(* CODESYS project GraphicalTesting.project
   Company: ifm electronic
   Description: Project template with CR711S configured 2.25MByte Standard 2.25MByte Safety
   Version: 2.4.10.0
   Title: ifmCR711S_TemplateProject

Project tree, tasks and I/O mapping:
  SafetyPLC : CR711S SIL2, ifm electronic, order no. CR711S, version 3.2.0.0
    application Application
      libraries: ifmR360-3, * (ifm electronic)
      task Task (cyclic, interval t#10ms, priority 1, watchdog t#8ms x 1) calls PLC_PRG
      program PLC_PRG [ST]
      global variables EVL
    Communication : Communication, ifm electronic, version 3.2.0.0
      CAN : CAN, ifm electronic, version 3.2.0.0
      Ethernet : Ethernet, ifm electronic, version 3.2.0.0
    HMI : HMI, ifm electronic, version 3.2.0.0
      User_LEDs : User_LEDs, ifm electronic, version 3.2.0.0
          input  UserLED0_I : LED_IEC_B_INPUT_MAPPING_TYPE  // UserLED0_I
          input  UserLED1_I : LED_IEC_B_INPUT_MAPPING_TYPE  // UserLED1_I
          input  UserLED2_I : LED_IEC_B_INPUT_MAPPING_TYPE  // UserLED2_I
          input  UserLED3_I : LED_IEC_B_INPUT_MAPPING_TYPE  // UserLED3_I
          output UserLED0_Q : LED_IEC_B_OUTPUT_MAPPING_TYPE  // User LED 0
          output UserLED1_Q : LED_IEC_B_OUTPUT_MAPPING_TYPE  // User LED 1
          output UserLED2_Q : LED_IEC_B_OUTPUT_MAPPING_TYPE  // User LED 2
          output UserLED3_Q : LED_IEC_B_OUTPUT_MAPPING_TYPE  // User LED 3
    Local_IO : Local_IO, ifm electronic, version 3.2.0.0
      Inputs : Inputs, ifm electronic, version 3.2.0.0
          input  IN0100_I : IN_MULTIFUNCTION_A_INPUT_MAPPING_TYPE  // IN0100_I
          input  IN0101_I : IN_MULTIFUNCTION_A_INPUT_MAPPING_TYPE  // IN0101_I
          input  IN0102_I : IN_MULTIFUNCTION_A_INPUT_MAPPING_TYPE  // IN0102_I
          input  IN0103_I : IN_MULTIFUNCTION_A_INPUT_MAPPING_TYPE  // IN0103_I
          input  IN0200_I : IN_MULTIFUNCTION_A_INPUT_MAPPING_TYPE  // IN0200_I
          input  IN0201_I : IN_MULTIFUNCTION_A_INPUT_MAPPING_TYPE  // IN0201_I
          input  IN0202_I : IN_MULTIFUNCTION_A_INPUT_MAPPING_TYPE  // IN0202_I
          input  IN0203_I : IN_MULTIFUNCTION_A_INPUT_MAPPING_TYPE  // IN0203_I
          input  IN0600_I : IN_MULTIFUNCTION_A_INPUT_MAPPING_TYPE  // IN0600_I
          input  IN0601_I : IN_MULTIFUNCTION_A_INPUT_MAPPING_TYPE  // IN0601_I
          input  IN0602_I : IN_MULTIFUNCTION_A_INPUT_MAPPING_TYPE  // IN0602_I
          input  IN0603_I : IN_MULTIFUNCTION_A_INPUT_MAPPING_TYPE  // IN0603_I
          input  IN0700_I : IN_MULTIFUNCTION_A_INPUT_MAPPING_TYPE  // IN0700_I
          input  IN0701_I : IN_MULTIFUNCTION_A_INPUT_MAPPING_TYPE  // IN0701_I
          input  IN0702_I : IN_MULTIFUNCTION_A_INPUT_MAPPING_TYPE  // IN0702_I
          input  IN0703_I : IN_MULTIFUNCTION_A_INPUT_MAPPING_TYPE  // IN0703_I
          input  IN0400_I : IN_RESISTOR_A_INPUT_MAPPING_TYPE  // IN0400_I
          input  IN0401_I : IN_RESISTOR_A_INPUT_MAPPING_TYPE  // IN0401_I
          input  IN0900_I : IN_RESISTOR_A_INPUT_MAPPING_TYPE  // IN0900_I
          input  IN0901_I : IN_RESISTOR_A_INPUT_MAPPING_TYPE  // IN0901_I
          input  IN0300_I : IN_DIGITAL_B_INPUT_MAPPING_TYPE  // IN0300_I
          input  IN0301_I : IN_DIGITAL_B_INPUT_MAPPING_TYPE  // IN0301_I
          input  IN0800_I : IN_DIGITAL_B_INPUT_MAPPING_TYPE  // IN0800_I
          input  IN0801_I : IN_DIGITAL_B_INPUT_MAPPING_TYPE  // IN0801_I
          input  COM_RESET_I : IN_COMMUNICATION_RESET_INPUT_MAPPING_TYPE  // COM_RESET_I
          input  IN0000_I : IN_FREQUENCY_B_CHANNEL_A_INPUT_MAPPING_TYPE  // IN0000_I
          input  IN0002_I : IN_FREQUENCY_B_CHANNEL_A_INPUT_MAPPING_TYPE  // IN0002_I
          input  IN0500_I : IN_FREQUENCY_B_CHANNEL_A_INPUT_MAPPING_TYPE  // IN0500_I
          input  IN0502_I : IN_FREQUENCY_B_CHANNEL_A_INPUT_MAPPING_TYPE  // IN0502_I
          input  IN0001_I : IN_FREQUENCY_B_CHANNEL_B_INPUT_MAPPING_TYPE  // IN0001_I
          input  IN0003_I : IN_FREQUENCY_B_CHANNEL_B_INPUT_MAPPING_TYPE  // IN0003_I
          input  IN0501_I : IN_FREQUENCY_B_CHANNEL_B_INPUT_MAPPING_TYPE  // IN0501_I
          input  IN0503_I : IN_FREQUENCY_B_CHANNEL_B_INPUT_MAPPING_TYPE  // IN0503_I
      Outputs : Outputs, ifm electronic, version 3.2.0.0
          input  OUT0006_I : OUT_PWM_40_BRIDGE_A_INPUT_MAPPING_TYPE  // OUT0006_I
          input  OUT0106_I : OUT_PWM_40_BRIDGE_A_INPUT_MAPPING_TYPE  // OUT0106_I
          input  OUT0206_I : OUT_PWM_40_BRIDGE_A_INPUT_MAPPING_TYPE  // OUT0206_I
          input  OUT0008_I : OUT_PWM_40_A_INPUT_MAPPING_TYPE  // OUT0008_I
          input  OUT0108_I : OUT_PWM_40_A_INPUT_MAPPING_TYPE  // OUT0108_I
          input  OUT0208_I : OUT_PWM_40_A_INPUT_MAPPING_TYPE  // OUT0208_I
          input  OUT0000_I : OUT_PWM_25_A_INPUT_MAPPING_TYPE  // OUT0000_I
          input  OUT0002_I : OUT_PWM_25_A_INPUT_MAPPING_TYPE  // OUT0002_I
          input  OUT0004_I : OUT_PWM_25_A_INPUT_MAPPING_TYPE  // OUT0004_I
          input  OUT0100_I : OUT_PWM_25_A_INPUT_MAPPING_TYPE  // OUT0100_I
          input  OUT0102_I : OUT_PWM_25_A_INPUT_MAPPING_TYPE  // OUT0102_I
          input  OUT0104_I : OUT_PWM_25_A_INPUT_MAPPING_TYPE  // OUT0104_I
          input  OUT0200_I : OUT_PWM_25_A_INPUT_MAPPING_TYPE  // OUT0200_I
          input  OUT0202_I : OUT_PWM_25_A_INPUT_MAPPING_TYPE  // OUT0202_I
          input  OUT0204_I : OUT_PWM_25_A_INPUT_MAPPING_TYPE  // OUT0204_I
          input  OUT3001_I : OUT_VOLTAGE_A_INPUT_MAPPING_TYPE  // OUT3001_I
          input  OUT3000_I : OUT_SUPPLY_A_INPUT_MAPPING_TYPE  // OUT3000_I
          input  OUT0001_I : OUT_PWM_25_B_INPUT_MAPPING_TYPE  // OUT0001_I
          input  OUT0003_I : OUT_PWM_25_B_INPUT_MAPPING_TYPE  // OUT0003_I
          input  OUT0005_I : OUT_PWM_25_B_INPUT_MAPPING_TYPE  // OUT0005_I
          input  OUT0101_I : OUT_PWM_25_B_INPUT_MAPPING_TYPE  // OUT0101_I
          input  OUT0103_I : OUT_PWM_25_B_INPUT_MAPPING_TYPE  // OUT0103_I
          input  OUT0105_I : OUT_PWM_25_B_INPUT_MAPPING_TYPE  // OUT0105_I
          input  OUT0201_I : OUT_PWM_25_B_INPUT_MAPPING_TYPE  // OUT0201_I
          input  OUT0203_I : OUT_PWM_25_B_INPUT_MAPPING_TYPE  // OUT0203_I
          input  OUT0205_I : OUT_PWM_25_B_INPUT_MAPPING_TYPE  // OUT0205_I
          input  OUT0007_I : OUT_PWM_40_BRIDGE_A_INPUT_MAPPING_TYPE  // OUT0007_I
          input  OUT0107_I : OUT_PWM_40_BRIDGE_A_INPUT_MAPPING_TYPE  // OUT0107_I
          input  OUT0207_I : OUT_PWM_40_BRIDGE_A_INPUT_MAPPING_TYPE  // OUT0207_I
          output OUT0006_Q : OUT_PWM_40_BRIDGE_A_OUTPUT_MAPPING_TYPE  // OUT0006_Q
          output OUT0106_Q : OUT_PWM_40_BRIDGE_A_OUTPUT_MAPPING_TYPE  // OUT0106_Q
          output OUT0206_Q : OUT_PWM_40_BRIDGE_A_OUTPUT_MAPPING_TYPE  // OUT0206_Q
          output OUT0008_Q : OUT_PWM_40_A_OUTPUT_MAPPING_TYPE  // OUT0008_Q
          output OUT0108_Q : OUT_PWM_40_A_OUTPUT_MAPPING_TYPE  // OUT0108_Q
          output OUT0208_Q : OUT_PWM_40_A_OUTPUT_MAPPING_TYPE  // OUT0208_Q
          output OUT0000_Q : OUT_PWM_25_A_OUTPUT_MAPPING_TYPE  // OUT0000_Q
          output OUT0002_Q : OUT_PWM_25_A_OUTPUT_MAPPING_TYPE  // OUT0002_Q
          output OUT0004_Q : OUT_PWM_25_A_OUTPUT_MAPPING_TYPE  // OUT0004_Q
          output OUT0100_Q : OUT_PWM_25_A_OUTPUT_MAPPING_TYPE  // OUT0100_Q
          output OUT0102_Q : OUT_PWM_25_A_OUTPUT_MAPPING_TYPE  // OUT0102_Q
          output OUT0104_Q : OUT_PWM_25_A_OUTPUT_MAPPING_TYPE  // OUT0104_Q
          output OUT0200_Q : OUT_PWM_25_A_OUTPUT_MAPPING_TYPE  // OUT0200_Q
          output OUT0202_Q : OUT_PWM_25_A_OUTPUT_MAPPING_TYPE  // OUT0202_Q
          output OUT0204_Q : OUT_PWM_25_A_OUTPUT_MAPPING_TYPE  // OUT0204_Q
          output OUT3001_Q : OUT_VOLTAGE_A_OUTPUT_MAPPING_TYPE  // OUT3001_Q
          output OUT3000_Q : OUT_SUPPLY_A_OUTPUT_MAPPING_TYPE  // OUT3000_Q
          output OUT0001_Q : OUT_PWM_25_B_OUTPUT_MAPPING_TYPE  // OUT0001_Q
          output OUT0003_Q : OUT_PWM_25_B_OUTPUT_MAPPING_TYPE  // OUT0003_Q
          output OUT0005_Q : OUT_PWM_25_B_OUTPUT_MAPPING_TYPE  // OUT0005_Q
          output OUT0101_Q : OUT_PWM_25_B_OUTPUT_MAPPING_TYPE  // OUT0101_Q
          output OUT0103_Q : OUT_PWM_25_B_OUTPUT_MAPPING_TYPE  // OUT0103_Q
          output OUT0105_Q : OUT_PWM_25_B_OUTPUT_MAPPING_TYPE  // OUT0105_Q
          output OUT0201_Q : OUT_PWM_25_B_OUTPUT_MAPPING_TYPE  // OUT0201_Q
          output OUT0203_Q : OUT_PWM_25_B_OUTPUT_MAPPING_TYPE  // OUT0203_Q
          output OUT0205_Q : OUT_PWM_25_B_OUTPUT_MAPPING_TYPE  // OUT0205_Q
          output OUT0007_Q : OUT_PWM_40_BRIDGE_A_OUTPUT_MAPPING_TYPE  // OUT0007_Q
          output OUT0107_Q : OUT_PWM_40_BRIDGE_A_OUTPUT_MAPPING_TYPE  // OUT0107_Q
          output OUT0207_Q : OUT_PWM_40_BRIDGE_A_OUTPUT_MAPPING_TYPE  // OUT0207_Q
      System_Inputs : System_Inputs, ifm electronic, version 3.2.0.0
          input  VBB30 : IN_SYSTEM_VOLTAGE_INPUT_MAPPING_TYPE  // VBB30
          input  VBB15 : IN_SYSTEM_VOLTAGE_INPUT_MAPPING_TYPE  // VBB15
          input  TemperatureBoard0 : IN_TEMPERATURE_INPUT_MAPPING_TYPE  // TemperatureBoard0
          input  TemperatureChip0 : IN_TEMPERATURE_INPUT_MAPPING_TYPE  // TemperatureChip0
      System_Outputs : System_Outputs, ifm electronic, version 3.2.0.0
          input  VBB0_SW_I : OUT_GROUP_SWITCH_INPUT_MAPPING_TYPE  // VBB0_SW_I
          input  VBB1_SW_I : OUT_GROUP_SWITCH_INPUT_MAPPING_TYPE  // VBB1_SW_I
          input  VBB2_SW_I : OUT_GROUP_SWITCH_INPUT_MAPPING_TYPE  // VBB2_SW_I
          output VBB0_SW_Q : OUT_GROUP_SWITCH_OUTPUT_MAPPING_TYPE  // VBB0_SW_Q
          output VBB1_SW_Q : OUT_GROUP_SWITCH_OUTPUT_MAPPING_TYPE  // VBB1_SW_Q
          output VBB2_SW_Q : OUT_GROUP_SWITCH_OUTPUT_MAPPING_TYPE  // VBB2_SW_Q
          output SUPPLY_SWITCH_Q : OUT_SYS_SWITCH_OUTPUT_MAPPING_TYPE  // SUPPLY_SWITCH_Q
  StandardPLC : CR711S Standard, ifm electronic, order no. CR711S, version 3.2.0.0
    application Application
      libraries: ifmR360-3, 1.1.1.0 (ifm electronic); Util, * (System); Standard, * (System); CR711S IOWrapper, 1.0.4.9 (ifm electronic); CAA CiA 405, 3.5.8.0 (CAA Technical Workgroup)
      task Main (cyclic, interval t#20ms, priority 1, watchdog t#18ms x 1) calls PLC_PRG, _CAN_MAIN
      EVC
      global variables PersistentVars
      program SFC_TEST [SFC]
      program FB_TESTING [FBD]: PleaseIhaveKids
      program LD_TEST [LD]
      visualisation Visualization
    Communication : Communication, ifm electronic, version 3.2.0.0
      CAN : CAN, ifm electronic, version 3.2.0.0
        CANbus_1 : CANbus, ifm electronic, version 1.0.1.1
            settings: NetID = 1
          J1939_Manager : J1939_Manager, 3S - Smart Software Solutions GmbH, order no. 
      , version 3.5.16.0
            Engine_Receiver : J1939_ECU, 3S - Smart Software Solutions GmbH, version 3.5.9.0
                settings: NAME = 16#0000000000000000; Communication Watchog Enabled = TRUE; Communication Watchdog Timeout Period = 16#05DC ms; Activated PGs = 13; PG Offline Data.Name = "EEC2"; PG Offline Data.Description = "Electronic Engine Controller 2"; PG Online Data.PGN = 61443; PG Online Data.Length (Bytes) = 8; PG Transmission Settings.Destination Address = 255; PG Transmission Settings.CycleTimeFactor = 1; Signal Offline Data.SPN = 558; Signal Offline Data.Name = "Accelerator Pedal 1 Low Idle Switch"; Signal Offline Data.Unit = "bit"; Signal Offline Data.Min = 0; Signal Offline Data.Max = 3; Signal Online Data.BitSize = 2; Signal Online Data.BitPosition = 0; Convert Data.Flags = 3; Convert Data.pSigValue = 0; Convert Data.Scaling = 4607182418800017408; Convert Data.Offset = 0; Signal Offline Data.SPN = 559; Signal Offline Data.Name = "Accelerator Pedal Kickdown Switch"; Signal Offline Data.Unit = "bit"; Signal Offline Data.Min = 0; Signal Offline Data.Max = 3; Signal Online Data.BitSize = 2; Signal Online Data.BitPosition = 2; Convert Data.Flags = 3; Convert Data.pSigValue = 0; Convert Data.Scaling = 4607182418800017408; Convert Data.Offset = 0; Signal Offline Data.SPN = 1437; Signal Offline Data.Name = "Road Speed Limit Status"; Signal Offline Data.Unit = "bit"; Signal Offline Data.Min = 0; Signal Offline Data.Max = 3; Signal Online Data.BitSize = 2; Signal Online Data.BitPosition = 4; Convert Data.Flags = 3;
                  Convert Data.pSigValue = 0; Convert Data.Scaling = 4607182418800017408; Convert Data.Offset = 0; Signal Offline Data.SPN = 2970; Signal Offline Data.Name = "Accelerator Pedal 2 Low Idle Switch"; Signal Offline Data.Unit = "bit"; Signal Offline Data.Min = 0; Signal Offline Data.Max = 3; Signal Online Data.BitSize = 2; Signal Online Data.BitPosition = 6; Convert Data.Flags = 3; Convert Data.pSigValue = 0; Convert Data.Scaling = 4607182418800017408; Convert Data.Offset = 0; Signal Offline Data.SPN = 91; Signal Offline Data.Name = "Accelerator Pedal Position 1"; Signal Offline Data.Unit = "%"; Signal Offline Data.Min = 0; Signal Offline Data.Max = 100; Signal Online Data.BitSize = 8; Signal Online Data.BitPosition = 8; Convert Data.Flags = 3; Convert Data.pSigValue = 0; Convert Data.Scaling = 4600877379321698714; Convert Data.Offset = 0; Signal Offline Data.SPN = 92; Signal Offline Data.Name = "Engine Percent Load At Current Speed"; Signal Offline Data.Unit = "%"; Signal Offline Data.Min = 0; Signal Offline Data.Max = 250; Signal Online Data.BitSize = 8; Signal Online Data.BitPosition = 16; Convert Data.Flags = 3; Convert Data.pSigValue = 0; Convert Data.Scaling = 4607182418800017408; Convert Data.Offset = 0; Signal Offline Data.SPN = 974; Signal Offline Data.Name = "Remote Accelerator Pedal Position"; Signal Offline Data.Unit = "%"; Signal Offline Data.Min = 0;
                  Signal Offline Data.Max = 100; Signal Online Data.BitSize = 8; Signal Online Data.BitPosition = 24; Convert Data.Flags = 3; Convert Data.pSigValue = 0; Convert Data.Scaling = 4600877379321698714; Convert Data.Offset = 0; Signal Offline Data.SPN = 29; Signal Offline Data.Name = "Accelerator Pedal Position 2"; Signal Offline Data.Unit = "%"; Signal Offline Data.Min = 0; Signal Offline Data.Max = 100; Signal Online Data.BitSize = 8; Signal Online Data.BitPosition = 32; Convert Data.Flags = 3; Convert Data.pSigValue = 0; Convert Data.Scaling = 4600877379321698714; Convert Data.Offset = 0; Signal Offline Data.SPN = 2979; Signal Offline Data.Name = "Vehicle Acceleration Rate Limit Status"; Signal Offline Data.Unit = "bit"; Signal Offline Data.Min = 0; Signal Offline Data.Max = 3; Signal Online Data.BitSize = 2; Signal Online Data.BitPosition = 40; Convert Data.Flags = 3; Convert Data.pSigValue = 0; Convert Data.Scaling = 4607182418800017408; Convert Data.Offset = 0; Signal Offline Data.SPN = 5021; Signal Offline Data.Name = "Momentary Engine Maximum Power Enable Feedback"; Signal Offline Data.Unit = "bit"; Signal Offline Data.Min = 0; Signal Offline Data.Max = 3; Signal Online Data.BitSize = 2; Signal Online Data.BitPosition = 42; Convert Data.Flags = 3; Convert Data.pSigValue = 0; Convert Data.Scaling = 4607182418800017408; Convert Data.Offset = 0;
                  Signal Offline Data.SPN = 5399; Signal Offline Data.Name = "DPF Thermal Management Active"; Signal Offline Data.Unit = "bit"; Signal Offline Data.Min = 0; Signal Offline Data.Max = 3; Signal Online Data.BitSize = 2; Signal Online Data.BitPosition = 44; Convert Data.Flags = 3; Convert Data.pSigValue = 0; Convert Data.Scaling = 4607182418800017408; Convert Data.Offset = 0; Signal Offline Data.SPN = 5400; Signal Offline Data.Name = "SCR Thermal Management Active"; Signal Offline Data.Unit = "bit"; Signal Offline Data.Min = 0; Signal Offline Data.Max = 3; Signal Online Data.BitSize = 2; Signal Online Data.BitPosition = 46; Convert Data.Flags = 3; Convert Data.pSigValue = 0; Convert Data.Scaling = 4607182418800017408; Convert Data.Offset = 0; Signal Offline Data.SPN = 3357; Signal Offline Data.Name = "Actual Maximum Available Engine - Percent Torque"; Signal Offline Data.Unit = "%"; Signal Offline Data.Min = 0; Signal Offline Data.Max = 100; Signal Online Data.BitSize = 8; Signal Online Data.BitPosition = 48; Convert Data.Flags = 3; Convert Data.pSigValue = 0; Convert Data.Scaling = 4600877379321698714; Convert Data.Offset = 0; Signal Offline Data.SPN = 5398; Signal Offline Data.Name = "Estimated Pumping - Percent Torque"; Signal Offline Data.Unit = "%"; Signal Offline Data.Min = -125; Signal Offline Data.Max = 125; Signal Online Data.BitSize = 8; Signal Online Data.BitPosition = 56;
                  Convert Data.Flags = 3; Convert Data.pSigValue = 0; Convert Data.Scaling = 4607182418800017408; Convert Data.Offset = 13861868546813853696; PG Offline Data.Name = "EEC1"; PG Offline Data.Description = "Electronic Engine Controller 1"; PG Online Data.PGN = 61444; PG Online Data.Length (Bytes) = 8; PG Transmission Settings.Destination Address = 255; PG Transmission Settings.CycleTimeFactor = 1; Signal Offline Data.SPN = 899; Signal Offline Data.Name = "Engine Torque Mode"; Signal Offline Data.Unit = "bit"; Signal Offline Data.Min = 0; Signal Offline Data.Max = 15; Signal Online Data.BitSize = 4; Signal Online Data.BitPosition = 0; Convert Data.Flags = 3; Convert Data.pSigValue = 0; Convert Data.Scaling = 4607182418800017408; Convert Data.Offset = 0; Signal Offline Data.SPN = 4154; Signal Offline Data.Name = "Actual Engine - Percent Torque High Resolution"; Signal Offline Data.Unit = "%"; Signal Offline Data.Min = 0; Signal Offline Data.Max = 0.875; Signal Online Data.BitSize = 4; Signal Online Data.BitPosition = 4; Convert Data.Flags = 3; Convert Data.pSigValue = 0; Convert Data.Scaling = 4593671619917905920; Convert Data.Offset = 0; Signal Offline Data.SPN = 512; Signal Offline Data.Name = "Driver$'s Demand Engine - Percent Torque"; Signal Offline Data.Unit = "%"; Signal Offline Data.Min = -125; Signal Offline Data.Max = 125; Signal Online Data.BitSize = 8; Signal Online Data.BitPosition = 8; Convert Data.Flags = 3;
                  Convert Data.pSigValue = 0; Convert Data.Scaling = 4607182418800017408; Convert Data.Offset = 13861868546813853696; Signal Offline Data.SPN = 513; Signal Offline Data.Name = "Actual Engine - Percent Torque"; Signal Offline Data.Unit = "%"; Signal Offline Data.Min = -125; Signal Offline Data.Max = 125; Signal Online Data.BitSize = 8; Signal Online Data.BitPosition = 16; Convert Data.Flags = 3; Convert Data.pSigValue = 0; Convert Data.Scaling = 4607182418800017408; Convert Data.Offset = 13861868546813853696; Signal Offline Data.SPN = 190; Signal Offline Data.Name = "Engine Speed"; Signal Offline Data.Unit = "rpm"; Signal Offline Data.Min = 0; Signal Offline Data.Max = 8031.875; Signal Online Data.BitSize = 16; Signal Online Data.BitPosition = 24; Convert Data.Flags = 3; Convert Data.pSigValue = 0; Convert Data.Scaling = 4593671619917905920; Convert Data.Offset = 0; Signal Offline Data.SPN = 1483; Signal Offline Data.Name = "Source Address of Controlling Device for Engine Control"; Signal Offline Data.Unit = "SA"; Signal Offline Data.Min = 0; Signal Offline Data.Max = 255; Signal Online Data.BitSize = 8; Signal Online Data.BitPosition = 40; Convert Data.Flags = 3; Convert Data.pSigValue = 0; Convert Data.Scaling = 4607182418800017408; Convert Data.Offset = 0; Signal Offline Data.SPN = 1675; Signal Offline Data.Name = "Engine Starter Mode"; Signal Offline Data.Unit = "bit"; Signal Offline Data.Min = 0;
                  Signal Offline Data.Max = 15; Signal Online Data.BitSize = 4; Signal Online Data.BitPosition = 48; Convert Data.Flags = 3; Convert Data.pSigValue = 0; Convert Data.Scaling = 4607182418800017408; Convert Data.Offset = 0; Signal Offline Data.SPN = 2432; Signal Offline Data.Name = "Engine Demand – Percent Torque"; Signal Offline Data.Unit = "%"; Signal Offline Data.Min = -125; Signal Offline Data.Max = 125; Signal Online Data.BitSize = 8; Signal Online Data.BitPosition = 56; Convert Data.Flags = 3; Convert Data.pSigValue = 0; Convert Data.Scaling = 4607182418800017408; Convert Data.Offset = 13861868546813853696; PG Offline Data.Name = "HOURS"; PG Offline Data.Description = "Engine Hours, Revolutions"; PG Online Data.PGN = 65253; PG Online Data.Length (Bytes) = 8; PG Transmission Settings.Destination Address = 255; PG Transmission Settings.CycleTimeFactor = 1; Signal Offline Data.SPN = 247; Signal Offline Data.Name = "Engine Total Hours of Operation"; Signal Offline Data.Description = "Accumulated time of operation of engine."; Signal Offline Data.Unit = "hr"; Signal Offline Data.Min = 0; Signal Offline Data.Max = 210554060.75; Signal Online Data.BitSize = 32; Signal Online Data.BitPosition = 0; Convert Data.Flags = 3; Convert Data.pSigValue = 0; Convert Data.Scaling = 4587366580439587226; Convert Data.Offset = 0; Signal Offline Data.SPN = 249; Signal Offline Data.Name = "Engine Total Revolutions"; Signal Offline Data.Description = "Accumulated number of revolutions of engine crankshaft during its operation."; Signal Offline Data.Unit = "r";
                  Signal Offline Data.Min = 0; Signal Offline Data.Max = 4211081215000; Signal Online Data.BitSize = 32; Signal Online Data.BitPosition = 32; Convert Data.Flags = 3; Convert Data.pSigValue = 0; Convert Data.Scaling = 4652007308841189376; Convert Data.Offset = 0; PG Offline Data.Name = "ET1"; PG Offline Data.Description = "Engine Temperature 1"; PG Online Data.PGN = 65262; PG Online Data.Length (Bytes) = 8; PG Transmission Settings.Destination Address = 255; PG Transmission Settings.CycleTimeFactor = 1; Signal Offline Data.SPN = 110; Signal Offline Data.Name = "Engine Coolant Temperature"; Signal Offline Data.Description = "Temperature of liquid found in engine cooling system."; Signal Offline Data.Unit = "C"; Signal Offline Data.Min = -40; Signal Offline Data.Max = 210; Signal Online Data.BitSize = 8; Signal Online Data.BitPosition = 0; Convert Data.Flags = 3; Convert Data.pSigValue = 0; Convert Data.Scaling = 4607182418800017408; Convert Data.Offset = 13854198353698488320; Signal Offline Data.SPN = 174; Signal Offline Data.Name = "Engine Fuel Temperature 1"; Signal Offline Data.Unit = "C"; Signal Offline Data.Min = -40; Signal Offline Data.Max = 210; Signal Online Data.BitSize = 8; Signal Online Data.BitPosition = 8; Convert Data.Flags = 3; Convert Data.pSigValue = 0; Convert Data.Scaling = 4607182418800017408; Convert Data.Offset = 13854198353698488320; Signal Offline Data.SPN = 175; Signal Offline Data.Name = "Engine Oil Temperature 1"; Signal Offline Data.Description = "Temperature of the engine lubricant.";
                  Signal Offline Data.Unit = "C"; Signal Offline Data.Min = -273; Signal Offline Data.Max = 1734.96875; Signal Online Data.BitSize = 16; Signal Online Data.BitPosition = 16; Convert Data.Flags = 3; Convert Data.pSigValue = 0; Convert Data.Scaling = 4584664420663164928; Convert Data.Offset = 13866882319836512256; Signal Offline Data.SPN = 176; Signal Offline Data.Name = "Engine Turbocharger Oil Temperature"; Signal Offline Data.Description = "Temperature of the turbocharger lubricant."; Signal Offline Data.Unit = "C"; Signal Offline Data.Min = -273; Signal Offline Data.Max = 1734.96875; Signal Online Data.BitSize = 16; Signal Online Data.BitPosition = 32; Convert Data.Flags = 3; Convert Data.pSigValue = 0; Convert Data.Scaling = 4584664420663164928; Convert Data.Offset = 13866882319836512256; Signal Offline Data.SPN = 52; Signal Offline Data.Name = "Engine Intercooler Temperature"; Signal Offline Data.Description = "Temperature of liquid found in the intercooler located after the turbocharger."; Signal Offline Data.Unit = "C"; Signal Offline Data.Min = -40; Signal Offline Data.Max = 210; Signal Online Data.BitSize = 8; Signal Online Data.BitPosition = 48; Convert Data.Flags = 3; Convert Data.pSigValue = 0; Convert Data.Scaling = 4607182418800017408; Convert Data.Offset = 13854198353698488320; Signal Offline Data.SPN = 1134; Signal Offline Data.Name = "Engine Intercooler Thermostat Opening"; Signal Offline Data.Unit = "%"; Signal Offline Data.Min = 0; Signal Offline Data.Max = 100; Signal Online Data.BitSize = 8; Signal Online Data.BitPosition = 56;
                  Convert Data.Flags = 3; Convert Data.pSigValue = 0; Convert Data.Scaling = 4600877379321698714; Convert Data.Offset = 0; PG Offline Data.Name = "EFL/P1"; PG Offline Data.Description = "Engine Fluid Level/Pressure 1"; PG Online Data.PGN = 65263; PG Online Data.Length (Bytes) = 8; PG Transmission Settings.Destination Address = 255; PG Transmission Settings.CycleTimeFactor = 1; Signal Offline Data.SPN = 94; Signal Offline Data.Name = "Engine Fuel Delivery Pressure"; Signal Offline Data.Unit = "kPa"; Signal Offline Data.Min = 0; Signal Offline Data.Max = 1000; Signal Online Data.BitSize = 8; Signal Online Data.BitPosition = 0; Convert Data.Flags = 3; Convert Data.pSigValue = 0; Convert Data.Scaling = 4616189618054758400; Convert Data.Offset = 0; Signal Offline Data.SPN = 22; Signal Offline Data.Name = "Engine Extended Crankcase Blow-by Pressure"; Signal Offline Data.Unit = "kPa"; Signal Offline Data.Min = 0; Signal Offline Data.Max = 12.5; Signal Online Data.BitSize = 8; Signal Online Data.BitPosition = 8; Convert Data.Flags = 3; Convert Data.pSigValue = 0; Convert Data.Scaling = 4587366580439587226; Convert Data.Offset = 0; Signal Offline Data.SPN = 98; Signal Offline Data.Name = "Engine Oil Level"; Signal Offline Data.Description = "Ratio of current volume of engine sump oil to maximum required volume."; Signal Offline Data.Unit = "%"; Signal Offline Data.Min = 0; Signal Offline Data.Max = 100; Signal Online Data.BitSize = 8; Signal Online Data.BitPosition = 16;
                  Convert Data.Flags = 3; Convert Data.pSigValue = 0; Convert Data.Scaling = 4600877379321698714; Convert Data.Offset = 0; Signal Offline Data.SPN = 100; Signal Offline Data.Name = "Engine Oil Pressure"; Signal Offline Data.Description = "Gage pressure of oil in engine lubrication system as provided by oil pump."; Signal Offline Data.Unit = "kPa"; Signal Offline Data.Min = 0; Signal Offline Data.Max = 1000; Signal Online Data.BitSize = 8; Signal Online Data.BitPosition = 24; Convert Data.Flags = 3; Convert Data.pSigValue = 0; Convert Data.Scaling = 4616189618054758400; Convert Data.Offset = 0; Signal Offline Data.SPN = 101; Signal Offline Data.Name = "Engine Crankcase Pressure"; Signal Offline Data.Description = "Gage pressure inside engine crankcase."; Signal Offline Data.Unit = "kPa"; Signal Offline Data.Min = -250; Signal Offline Data.Max = 251.99; Signal Online Data.BitSize = 16; Signal Online Data.BitPosition = 32; Convert Data.Flags = 3; Convert Data.pSigValue = 0; Convert Data.Scaling = 4575657221408423936; Convert Data.Offset = 13866372146441224192; Signal Offline Data.SPN = 109; Signal Offline Data.Name = "Engine Coolant Pressure"; Signal Offline Data.Description = "Gage pressure of liquid found in engine cooling system.$r$n$r$nSee SPN 20 for alternate SLOT."; Signal Offline Data.Unit = "kPa"; Signal Offline Data.Min = 0; Signal Offline Data.Max = 500; Signal Online Data.BitSize = 8; Signal Online Data.BitPosition = 48; Convert Data.Flags = 3; Convert Data.pSigValue = 0; Convert Data.Scaling = 4611686018427387904; Convert Data.Offset = 0;
                  Signal Offline Data.SPN = 111; Signal Offline Data.Name = "Engine Coolant Level"; Signal Offline Data.Unit = "%"; Signal Offline Data.Min = 0; Signal Offline Data.Max = 100; Signal Online Data.BitSize = 8; Signal Online Data.BitPosition = 56; Convert Data.Flags = 3; Convert Data.pSigValue = 0; Convert Data.Scaling = 4600877379321698714; Convert Data.Offset = 0; PG Offline Data.Name = "LFE1"; PG Offline Data.Description = "Fuel Economy (Liquid)"; PG Online Data.PGN = 65266; PG Online Data.Length (Bytes) = 8; PG Transmission Settings.Destination Address = 255; PG Transmission Settings.CycleTimeFactor = 1; Signal Offline Data.SPN = 183; Signal Offline Data.Name = "Engine Fuel Rate"; Signal Offline Data.Description = "Amount of fuel consumed by engine per unit of time.$r$n$r$nNOTE - See SPN 1600 for alternate resolution."; Signal Offline Data.Unit = "l/h"; Signal Offline Data.Min = 0; Signal Offline Data.Max = 3212.75; Signal Online Data.BitSize = 16; Signal Online Data.BitPosition = 0; Convert Data.Flags = 3; Convert Data.pSigValue = 0; Convert Data.Scaling = 4587366580439587226; Convert Data.Offset = 0; Signal Offline Data.SPN = 184; Signal Offline Data.Name = "Engine Instantaneous Fuel Economy"; Signal Offline Data.Description = "Current fuel economy at current vehicle velocity.$r$n$r$n0xFB00 = Infinite (for example, during engine motoring)"; Signal Offline Data.Unit = "km/L"; Signal Offline Data.Min = 0; Signal Offline Data.Max = 125.498046875; Signal Online Data.BitSize = 16; Signal Online Data.BitPosition = 16; Convert Data.Flags = 3; Convert Data.pSigValue = 0; Convert Data.Scaling = 4566650022153682944;
                  Convert Data.Offset = 0; Signal Offline Data.SPN = 185; Signal Offline Data.Name = "Engine Average Fuel Economy"; Signal Offline Data.Description = "Average of instantaneous fuel economy for that segment of vehicle operation of interest."; Signal Offline Data.Unit = "km/L"; Signal Offline Data.Min = 0; Signal Offline Data.Max = 125.498046875; Signal Online Data.BitSize = 16; Signal Online Data.BitPosition = 32; Convert Data.Flags = 3; Convert Data.pSigValue = 0; Convert Data.Scaling = 4566650022153682944; Convert Data.Offset = 0; Signal Offline Data.SPN = 51; Signal Offline Data.Name = "Engine Throttle Valve 1 Position"; Signal Offline Data.Unit = "%"; Signal Offline Data.Min = 0; Signal Offline Data.Max = 100; Signal Online Data.BitSize = 8; Signal Online Data.BitPosition = 48; Convert Data.Flags = 3; Convert Data.pSigValue = 0; Convert Data.Scaling = 4600877379321698714; Convert Data.Offset = 0; Signal Offline Data.SPN = 3673; Signal Offline Data.Name = "Engine Throttle Valve 2 Position"; Signal Offline Data.Unit = "%"; Signal Offline Data.Min = 0; Signal Offline Data.Max = 100; Signal Online Data.BitSize = 8; Signal Online Data.BitPosition = 56; Convert Data.Flags = 3; Convert Data.pSigValue = 0; Convert Data.Scaling = 4600877379321698714; Convert Data.Offset = 0; PG Offline Data.Name = "IC1"; PG Offline Data.Description = "Intake/Exhaust Conditions 1"; PG Online Data.PGN = 65270; PG Online Data.Length (Bytes) = 8; PG Transmission Settings.Destination Address = 255;
                  PG Transmission Settings.CycleTimeFactor = 1; Signal Offline Data.SPN = 81; Signal Offline Data.Name = "Engine Diesel Particulate Filter Intake Pressure"; Signal Offline Data.Unit = "kPa"; Signal Offline Data.Min = 0; Signal Offline Data.Max = 125; Signal Online Data.BitSize = 8; Signal Online Data.BitPosition = 0; Convert Data.Flags = 3; Convert Data.pSigValue = 0; Convert Data.Scaling = 4602678819172646912; Convert Data.Offset = 0; Signal Offline Data.SPN = 102; Signal Offline Data.Name = "Engine Intake Manifold #1 Pressure"; Signal Offline Data.Unit = "kPa"; Signal Offline Data.Min = 0; Signal Offline Data.Max = 500; Signal Online Data.BitSize = 8; Signal Online Data.BitPosition = 8; Convert Data.Flags = 3; Convert Data.pSigValue = 0; Convert Data.Scaling = 4611686018427387904; Convert Data.Offset = 0; Signal Offline Data.SPN = 105; Signal Offline Data.Name = "Engine Intake Manifold 1 Temperature"; Signal Offline Data.Description = "Temperature of pre-combustion air found in intake manifold of engine air supply system."; Signal Offline Data.Unit = "C"; Signal Offline Data.Min = -40; Signal Offline Data.Max = 210; Signal Online Data.BitSize = 8; Signal Online Data.BitPosition = 16; Convert Data.Flags = 3; Convert Data.pSigValue = 0; Convert Data.Scaling = 4607182418800017408; Convert Data.Offset = 13854198353698488320; Signal Offline Data.SPN = 106; Signal Offline Data.Name = "Engine Air Intake Pressure"; Signal Offline Data.Description = "Absolute air pressure at input port to intake manifold or air box."; Signal Offline Data.Unit = "kPa"; Signal Offline Data.Min = 0;
                  Signal Offline Data.Max = 500; Signal Online Data.BitSize = 8; Signal Online Data.BitPosition = 24; Convert Data.Flags = 3; Convert Data.pSigValue = 0; Convert Data.Scaling = 4611686018427387904; Convert Data.Offset = 0; Signal Offline Data.SPN = 107; Signal Offline Data.Name = "Engine Air Filter 1 Differential Pressure"; Signal Offline Data.Unit = "kPa"; Signal Offline Data.Min = 0; Signal Offline Data.Max = 12.5; Signal Online Data.BitSize = 8; Signal Online Data.BitPosition = 32; Convert Data.Flags = 3; Convert Data.pSigValue = 0; Convert Data.Scaling = 4587366580439587226; Convert Data.Offset = 0; Signal Offline Data.SPN = 173; Signal Offline Data.Name = "Engine Exhaust Gas Temperature"; Signal Offline Data.Unit = "C"; Signal Offline Data.Min = -273; Signal Offline Data.Max = 1734.96875; Signal Online Data.BitSize = 16; Signal Online Data.BitPosition = 40; Convert Data.Flags = 3; Convert Data.pSigValue = 0; Convert Data.Scaling = 4584664420663164928; Convert Data.Offset = 13866882319836512256; Signal Offline Data.SPN = 112; Signal Offline Data.Name = "Engine Coolant Filter Differential Pressure"; Signal Offline Data.Unit = "kPa"; Signal Offline Data.Min = 0; Signal Offline Data.Max = 125; Signal Online Data.BitSize = 8; Signal Online Data.BitPosition = 56; Convert Data.Flags = 3; Convert Data.pSigValue = 0; Convert Data.Scaling = 4602678819172646912; Convert Data.Offset = 0;
                  PG Offline Data.Name = "VEP1"; PG Offline Data.Description = "Vehicle Electrical Power 1"; PG Online Data.PGN = 65271; PG Online Data.Length (Bytes) = 8; PG Transmission Settings.Destination Address = 255; PG Transmission Settings.CycleTimeFactor = 1; Signal Offline Data.SPN = 114; Signal Offline Data.Name = "Net Battery Current"; Signal Offline Data.Description = "Net flow of electrical current into/out of the battery or batteries."; Signal Offline Data.Unit = "Amps"; Signal Offline Data.Min = -125; Signal Offline Data.Max = 125; Signal Online Data.BitSize = 8; Signal Online Data.BitPosition = 0; Convert Data.Flags = 3; Convert Data.pSigValue = 0; Convert Data.Scaling = 4607182418800017408; Convert Data.Offset = 13861868546813853696; Signal Offline Data.SPN = 115; Signal Offline Data.Name = "Alternator Current"; Signal Offline Data.Unit = "Amps"; Signal Offline Data.Min = 0; Signal Offline Data.Max = 250; Signal Online Data.BitSize = 8; Signal Online Data.BitPosition = 8; Convert Data.Flags = 3; Convert Data.pSigValue = 0; Convert Data.Scaling = 4607182418800017408; Convert Data.Offset = 0; Signal Offline Data.SPN = 167; Signal Offline Data.Name = "Charging System Potential (Voltage)"; Signal Offline Data.Unit = "Volts"; Signal Offline Data.Min = 0; Signal Offline Data.Max = 3212.75; Signal Online Data.BitSize = 16; Signal Online Data.BitPosition = 16; Convert Data.Flags = 3; Convert Data.pSigValue = 0; Convert Data.Scaling = 4587366580439587226; Convert Data.Offset = 0;
                  Signal Offline Data.SPN = 168; Signal Offline Data.Name = "Battery Potential / Power Input 1"; Signal Offline Data.Unit = "Volts"; Signal Offline Data.Min = 0; Signal Offline Data.Max = 3212.75; Signal Online Data.BitSize = 16; Signal Online Data.BitPosition = 32; Convert Data.Flags = 3; Convert Data.pSigValue = 0; Convert Data.Scaling = 4587366580439587226; Convert Data.Offset = 0; Signal Offline Data.SPN = 158; Signal Offline Data.Name = "Keyswitch Battery Potential"; Signal Offline Data.Unit = "Volts"; Signal Offline Data.Min = 0; Signal Offline Data.Max = 3212.75; Signal Online Data.BitSize = 16; Signal Online Data.BitPosition = 48; Convert Data.Flags = 3; Convert Data.pSigValue = 0; Convert Data.Scaling = 4587366580439587226; Convert Data.Offset = 0; PG Offline Data.Name = "EC1"; PG Offline Data.Description = "Engine Configuration 1"; PG Online Data.PGN = 65251; PG Online Data.Length (Bytes) = 39; PG Transmission Settings.Destination Address = 255; PG Transmission Settings.CycleTimeFactor = 1; Signal Offline Data.SPN = 188; Signal Offline Data.Name = "Engine Speed At Idle, Point 1 (Engine Configuration)"; Signal Offline Data.Unit = "rpm"; Signal Offline Data.Min = 0; Signal Offline Data.Max = 8031.875; Signal Online Data.BitSize = 16; Signal Online Data.BitPosition = 0; Convert Data.Flags = 3; Convert Data.pSigValue = 0; Convert Data.Scaling = 4593671619917905920; Convert Data.Offset = 0; Signal Offline Data.SPN = 539;
                  Signal Offline Data.Name = "Engine Percent Torque At Idle, Point 1 (Engine Configuration)"; Signal Offline Data.Unit = "%"; Signal Offline Data.Min = -125; Signal Offline Data.Max = 125; Signal Online Data.BitSize = 8; Signal Online Data.BitPosition = 16; Convert Data.Flags = 3; Convert Data.pSigValue = 0; Convert Data.Scaling = 4607182418800017408; Convert Data.Offset = 13861868546813853696; Signal Offline Data.SPN = 528; Signal Offline Data.Name = "Engine Speed At Point 2 (Engine Configuration)"; Signal Offline Data.Unit = "rpm"; Signal Offline Data.Min = 0; Signal Offline Data.Max = 8031.875; Signal Online Data.BitSize = 16; Signal Online Data.BitPosition = 24; Convert Data.Flags = 3; Convert Data.pSigValue = 0; Convert Data.Scaling = 4593671619917905920; Convert Data.Offset = 0; Signal Offline Data.SPN = 540; Signal Offline Data.Name = "Engine Percent Torque At Point 2 (Engine Configuration)"; Signal Offline Data.Unit = "%"; Signal Offline Data.Min = -125; Signal Offline Data.Max = 125; Signal Online Data.BitSize = 8; Signal Online Data.BitPosition = 40; Convert Data.Flags = 3; Convert Data.pSigValue = 0; Convert Data.Scaling = 4607182418800017408; Convert Data.Offset = 13861868546813853696; Signal Offline Data.SPN = 529; Signal Offline Data.Name = "Engine Speed At Point 3 (Engine Configuration)"; Signal Offline Data.Unit = "rpm"; Signal Offline Data.Min = 0; Signal Offline Data.Max = 8031.875; Signal Online Data.BitSize = 16; Signal Online Data.BitPosition = 48; Convert Data.Flags = 3;
                  Convert Data.pSigValue = 0; Convert Data.Scaling = 4593671619917905920; Convert Data.Offset = 0; Signal Offline Data.SPN = 541; Signal Offline Data.Name = "Engine Percent Torque At Point 3 (Engine Configuration)"; Signal Offline Data.Unit = "%"; Signal Offline Data.Min = -125; Signal Offline Data.Max = 125; Signal Online Data.BitSize = 8; Signal Online Data.BitPosition = 64; Convert Data.Flags = 3; Convert Data.pSigValue = 0; Convert Data.Scaling = 4607182418800017408; Convert Data.Offset = 13861868546813853696; Signal Offline Data.SPN = 530; Signal Offline Data.Name = "Engine Speed At Point 4 (Engine Configuration)"; Signal Offline Data.Unit = "rpm"; Signal Offline Data.Min = 0; Signal Offline Data.Max = 8031.875; Signal Online Data.BitSize = 16; Signal Online Data.BitPosition = 72; Convert Data.Flags = 3; Convert Data.pSigValue = 0; Convert Data.Scaling = 4593671619917905920; Convert Data.Offset = 0; Signal Offline Data.SPN = 542; Signal Offline Data.Name = "Engine Percent Torque At Point 4 (Engine Configuration)"; Signal Offline Data.Unit = "%"; Signal Offline Data.Min = -125; Signal Offline Data.Max = 125; Signal Online Data.BitSize = 8; Signal Online Data.BitPosition = 88; Convert Data.Flags = 3; Convert Data.pSigValue = 0; Convert Data.Scaling = 4607182418800017408; Convert Data.Offset = 13861868546813853696; Signal Offline Data.SPN = 531; Signal Offline Data.Name = "Engine Speed At Point 5 (Engine Configuration)"; Signal Offline Data.Unit = "rpm"; Signal Offline Data.Min = 0;
                  Signal Offline Data.Max = 8031.875; Signal Online Data.BitSize = 16; Signal Online Data.BitPosition = 96; Convert Data.Flags = 3; Convert Data.pSigValue = 0; Convert Data.Scaling = 4593671619917905920; Convert Data.Offset = 0; Signal Offline Data.SPN = 543; Signal Offline Data.Name = "Engine Percent Torque At Point 5 (Engine Configuration)"; Signal Offline Data.Unit = "%"; Signal Offline Data.Min = -125; Signal Offline Data.Max = 125; Signal Online Data.BitSize = 8; Signal Online Data.BitPosition = 112; Convert Data.Flags = 3; Convert Data.pSigValue = 0; Convert Data.Scaling = 4607182418800017408; Convert Data.Offset = 13861868546813853696; Signal Offline Data.SPN = 532; Signal Offline Data.Name = "Engine Speed At High Idle, Point 6 (Engine Configuration)"; Signal Offline Data.Unit = "rpm"; Signal Offline Data.Min = 0; Signal Offline Data.Max = 8031.875; Signal Online Data.BitSize = 16; Signal Online Data.BitPosition = 120; Convert Data.Flags = 3; Convert Data.pSigValue = 0; Convert Data.Scaling = 4593671619917905920; Convert Data.Offset = 0; Signal Offline Data.SPN = 545; Signal Offline Data.Name = "Engine Gain (Kp) Of The Endspeed Governor (Engine Configuration)"; Signal Offline Data.Unit = "%/rpm"; Signal Offline Data.Min = 0; Signal Offline Data.Max = 50.2; Signal Online Data.BitSize = 16; Signal Online Data.BitPosition = 136; Convert Data.Flags = 3; Convert Data.pSigValue = 0; Convert Data.Scaling = 4560344982675364250; Convert Data.Offset = 0;
                  Signal Offline Data.SPN = 544; Signal Offline Data.Name = "Engine Reference Torque (Engine Configuration)"; Signal Offline Data.Unit = "Nm"; Signal Offline Data.Min = 0; Signal Offline Data.Max = 64255; Signal Online Data.BitSize = 16; Signal Online Data.BitPosition = 152; Convert Data.Flags = 3; Convert Data.pSigValue = 0; Convert Data.Scaling = 4607182418800017408; Convert Data.Offset = 0; Signal Offline Data.SPN = 533; Signal Offline Data.Name = "Engine Maximum Momentary Override Speed, Point 7 (Engine Configuration)"; Signal Offline Data.Unit = "rpm"; Signal Offline Data.Min = 0; Signal Offline Data.Max = 8031.875; Signal Online Data.BitSize = 16; Signal Online Data.BitPosition = 168; Convert Data.Flags = 3; Convert Data.pSigValue = 0; Convert Data.Scaling = 4593671619917905920; Convert Data.Offset = 0; Signal Offline Data.SPN = 534; Signal Offline Data.Name = "Engine Maximum Momentary Override Time Limit (Engine Configuration)"; Signal Offline Data.Description = "The maximum time limit allowed to override the engine$'s high idle speed."; Signal Offline Data.Unit = "Seconds"; Signal Offline Data.Min = 0; Signal Offline Data.Max = 25; Signal Online Data.BitSize = 8; Signal Online Data.BitPosition = 184; Convert Data.Flags = 3; Convert Data.pSigValue = 0; Convert Data.Scaling = 4591870180066957722; Convert Data.Offset = 0; Signal Offline Data.SPN = 535; Signal Offline Data.Name = "Engine Requested Speed Control Range Lower Limit (Engine Configuration)"; Signal Offline Data.Description = "The minimum engine speed that the engine will allow when operating in a speed control/limit mode."; Signal Offline Data.Unit = "rpm"; Signal Offline Data.Min = 0; Signal Offline Data.Max = 2500;
                  Signal Online Data.BitSize = 8; Signal Online Data.BitPosition = 192; Convert Data.Flags = 3; Convert Data.pSigValue = 0; Convert Data.Scaling = 4621819117588971520; Convert Data.Offset = 0; Signal Offline Data.SPN = 536; Signal Offline Data.Name = "Engine Requested Speed Control Range Upper Limit (Engine Configuration)"; Signal Offline Data.Unit = "rpm"; Signal Offline Data.Min = 0; Signal Offline Data.Max = 2500; Signal Online Data.BitSize = 8; Signal Online Data.BitPosition = 200; Convert Data.Flags = 3; Convert Data.pSigValue = 0; Convert Data.Scaling = 4621819117588971520; Convert Data.Offset = 0; Signal Offline Data.SPN = 537; Signal Offline Data.Name = "Engine Requested Torque Control Range Lower Limit (Engine Configuration)"; Signal Offline Data.Description = "The minimum engine torque that the engine will allow when operating in a torque control/limit mode."; Signal Offline Data.Unit = "%"; Signal Offline Data.Min = -125; Signal Offline Data.Max = 125; Signal Online Data.BitSize = 8; Signal Online Data.BitPosition = 208; Convert Data.Flags = 3; Convert Data.pSigValue = 0; Convert Data.Scaling = 4607182418800017408; Convert Data.Offset = 13861868546813853696; Signal Offline Data.SPN = 538; Signal Offline Data.Name = "Engine Requested Torque Control Range Upper Limit (Engine Configuration)"; Signal Offline Data.Description = "The maximum engine torque that the engine will allow when operating in a torque control/limit mode."; Signal Offline Data.Unit = "%"; Signal Offline Data.Min = -125; Signal Offline Data.Max = 125; Signal Online Data.BitSize = 8; Signal Online Data.BitPosition = 216; Convert Data.Flags = 3; Convert Data.pSigValue = 0; Convert Data.Scaling = 4607182418800017408;
                  Convert Data.Offset = 13861868546813853696; Signal Offline Data.SPN = 1712; Signal Offline Data.Name = "Engine Extended Range Requested Speed Control Range Upper Limit (Engine configuration)"; Signal Offline Data.Unit = "rpm"; Signal Offline Data.Min = 0; Signal Offline Data.Max = 8031.875; Signal Online Data.BitSize = 16; Signal Online Data.BitPosition = 224; Convert Data.Flags = 3; Convert Data.pSigValue = 0; Convert Data.Scaling = 4593671619917905920; Convert Data.Offset = 0; Signal Offline Data.SPN = 1794; Signal Offline Data.Name = "Engine Moment of Inertia"; Signal Offline Data.Unit = "kg/m²"; Signal Offline Data.Min = 0; Signal Offline Data.Max = 257.02; Signal Online Data.BitSize = 16; Signal Online Data.BitPosition = 240; Convert Data.Flags = 3; Convert Data.pSigValue = 0; Convert Data.Scaling = 4571261708172110332; Convert Data.Offset = 0; Signal Offline Data.SPN = 1846; Signal Offline Data.Name = "Engine Default Torque Limit"; Signal Offline Data.Unit = "Nm"; Signal Offline Data.Min = 0; Signal Offline Data.Max = 64255; Signal Online Data.BitSize = 16; Signal Online Data.BitPosition = 256; Convert Data.Flags = 3; Convert Data.pSigValue = 0; Convert Data.Scaling = 4607182418800017408; Convert Data.Offset = 0; Signal Offline Data.SPN = 3344; Signal Offline Data.Name = "Support Variable Rate TSC1 Message"; Signal Offline Data.Unit = "bit"; Signal Offline Data.Min = 0; Signal Offline Data.Max = 255; Signal Online Data.BitSize = 8;
                  Signal Online Data.BitPosition = 272; Convert Data.Flags = 3; Convert Data.pSigValue = 0; Convert Data.Scaling = 4607182418800017408; Convert Data.Offset = 0; Signal Offline Data.SPN = 3345; Signal Offline Data.Name = "Support TSC1 Control Purpose Group 1"; Signal Offline Data.Unit = "bit"; Signal Offline Data.Min = 0; Signal Offline Data.Max = 255; Signal Online Data.BitSize = 8; Signal Online Data.BitPosition = 280; Convert Data.Flags = 3; Convert Data.pSigValue = 0; Convert Data.Scaling = 4607182418800017408; Convert Data.Offset = 0; Signal Offline Data.SPN = 3346; Signal Offline Data.Name = "Support TSC1 Control Purpose Group 2"; Signal Offline Data.Unit = "bit"; Signal Offline Data.Min = 0; Signal Offline Data.Max = 255; Signal Online Data.BitSize = 8; Signal Online Data.BitPosition = 288; Convert Data.Flags = 3; Convert Data.pSigValue = 0; Convert Data.Scaling = 4607182418800017408; Convert Data.Offset = 0; Signal Offline Data.SPN = 3347; Signal Offline Data.Name = "Support TSC1 Control Purpose Group 3"; Signal Offline Data.Unit = "bit"; Signal Offline Data.Min = 0; Signal Offline Data.Max = 255; Signal Online Data.BitSize = 8; Signal Online Data.BitPosition = 296; Convert Data.Flags = 3; Convert Data.pSigValue = 0; Convert Data.Scaling = 4607182418800017408; Convert Data.Offset = 0; Signal Offline Data.SPN = 3348; Signal Offline Data.Name = "Support TSC1 Control Purpose Group 4";
                  Signal Offline Data.Unit = "bit"; Signal Offline Data.Min = 0; Signal Offline Data.Max = 255; Signal Online Data.BitSize = 8; Signal Online Data.BitPosition = 304; Convert Data.Flags = 3; Convert Data.pSigValue = 0; Convert Data.Scaling = 4607182418800017408; Convert Data.Offset = 0; PG Offline Data.Name = "EEC3"; PG Offline Data.Description = "Electronic Engine Controller 3"; PG Online Data.PGN = 65247; PG Online Data.Length (Bytes) = 8; PG Transmission Settings.Destination Address = 255; PG Transmission Settings.CycleTimeFactor = 1; Signal Offline Data.SPN = 514; Signal Offline Data.Name = "Nominal Friction - Percent Torque"; Signal Offline Data.Unit = "%"; Signal Offline Data.Min = -125; Signal Offline Data.Max = 125; Signal Online Data.BitSize = 8; Signal Online Data.BitPosition = 0; Convert Data.Flags = 3; Convert Data.pSigValue = 0; Convert Data.Scaling = 4607182418800017408; Convert Data.Offset = 13861868546813853696; Signal Offline Data.SPN = 515; Signal Offline Data.Name = "Engine$'s Desired Operating Speed"; Signal Offline Data.Unit = "rpm"; Signal Offline Data.Min = 0; Signal Offline Data.Max = 8031.875; Signal Online Data.BitSize = 16; Signal Online Data.BitPosition = 8; Convert Data.Flags = 3; Convert Data.pSigValue = 0; Convert Data.Scaling = 4593671619917905920; Convert Data.Offset = 0; Signal Offline Data.SPN = 519; Signal Offline Data.Name = "Engine$'s Desired Operating Speed Asymmetry Adjustment"; Signal Offline Data.Unit = "Ratio";
                  Signal Offline Data.Min = 0; Signal Offline Data.Max = 250; Signal Online Data.BitSize = 8; Signal Online Data.BitPosition = 24; Convert Data.Flags = 3; Convert Data.pSigValue = 0; Convert Data.Scaling = 4607182418800017408; Convert Data.Offset = 0; Signal Offline Data.SPN = 2978; Signal Offline Data.Name = "Estimated Engine Parasitic Losses - Percent Torque"; Signal Offline Data.Unit = "%"; Signal Offline Data.Min = -125; Signal Offline Data.Max = 125; Signal Online Data.BitSize = 8; Signal Online Data.BitPosition = 32; Convert Data.Flags = 3; Convert Data.pSigValue = 0; Convert Data.Scaling = 4607182418800017408; Convert Data.Offset = 13861868546813853696; Signal Offline Data.SPN = 3236; Signal Offline Data.Name = "Aftertreatment 1 Exhaust Gas Mass Flow"; Signal Offline Data.Description = "Measured/calculated exhaust gas mass upstream of the aftertreatment system in exhaust bank 1 and 2."; Signal Offline Data.Unit = "kg/h"; Signal Offline Data.Min = 0; Signal Offline Data.Max = 12851; Signal Online Data.BitSize = 16; Signal Online Data.BitPosition = 40; Convert Data.Flags = 3; Convert Data.pSigValue = 0; Convert Data.Scaling = 4596373779694328218; Convert Data.Offset = 0; Signal Offline Data.SPN = 3237; Signal Offline Data.Name = "Aftertreatment 1 Intake Dew Point"; Signal Offline Data.Unit = "bit"; Signal Offline Data.Min = 0; Signal Offline Data.Max = 3; Signal Online Data.BitSize = 2; Signal Online Data.BitPosition = 56; Convert Data.Flags = 3; Convert Data.pSigValue = 0;
                  Convert Data.Scaling = 4607182418800017408; Convert Data.Offset = 0; Signal Offline Data.SPN = 3238; Signal Offline Data.Name = "Aftertreatment 1 Exhaust Dew Point"; Signal Offline Data.Unit = "bit"; Signal Offline Data.Min = 0; Signal Offline Data.Max = 3; Signal Online Data.BitSize = 2; Signal Online Data.BitPosition = 58; Convert Data.Flags = 3; Convert Data.pSigValue = 0; Convert Data.Scaling = 4607182418800017408; Convert Data.Offset = 0; Signal Offline Data.SPN = 3239; Signal Offline Data.Name = "Aftertreatment 2 Intake Dew Point"; Signal Offline Data.Unit = "bit"; Signal Offline Data.Min = 0; Signal Offline Data.Max = 3; Signal Online Data.BitSize = 2; Signal Online Data.BitPosition = 60; Convert Data.Flags = 3; Convert Data.pSigValue = 0; Convert Data.Scaling = 4607182418800017408; Convert Data.Offset = 0; Signal Offline Data.SPN = 3240; Signal Offline Data.Name = "Aftertreatment 2 Exhaust Dew Point"; Signal Offline Data.Unit = "bit"; Signal Offline Data.Min = 0; Signal Offline Data.Max = 3; Signal Online Data.BitSize = 2; Signal Online Data.BitPosition = 62; Convert Data.Flags = 3; Convert Data.pSigValue = 0; Convert Data.Scaling = 4607182418800017408; Convert Data.Offset = 0; PG Offline Data.Name = "AAI"; PG Offline Data.Description = "Auxiliary Analog Information"; PG Online Data.PGN = 65164; PG Online Data.Length (Bytes) = 8; PG Transmission Settings.Destination Address = 255;
                  PG Transmission Settings.CycleTimeFactor = 1; Signal Offline Data.SPN = 441; Signal Offline Data.Name = "Auxiliary Temperature 1"; Signal Offline Data.Description = "Temperature measured by auxiliary temperature sensor #1.  Not to be used in place of existing SPNs."; Signal Offline Data.Unit = "C"; Signal Offline Data.Min = -40; Signal Offline Data.Max = 210; Signal Online Data.BitSize = 8; Signal Online Data.BitPosition = 0; Convert Data.Flags = 3; Convert Data.pSigValue = 0; Convert Data.Scaling = 4607182418800017408; Convert Data.Offset = 13854198353698488320; Signal Offline Data.SPN = 1387; Signal Offline Data.Name = "Auxiliary Pressure #1"; Signal Offline Data.Description = "Pressure measured by auxiliary pressure sensor #1.  Not to be used in place of existing SPNs."; Signal Offline Data.Unit = "kPa"; Signal Offline Data.Min = 0; Signal Offline Data.Max = 4000; Signal Online Data.BitSize = 8; Signal Online Data.BitPosition = 16; Convert Data.Flags = 3; Convert Data.pSigValue = 0; Convert Data.Scaling = 4625196817309499392; Convert Data.Offset = 0; PG Offline Data.Name = "SHUTDN"; PG Offline Data.Description = "Shutdown"; PG Online Data.PGN = 65252; PG Online Data.Length (Bytes) = 8; PG Transmission Settings.Destination Address = 255; PG Transmission Settings.CycleTimeFactor = 1; Signal Offline Data.SPN = 593; Signal Offline Data.Name = "Engine Idle Shutdown has Shutdown Engine"; Signal Offline Data.Unit = "bit"; Signal Offline Data.Min = 0; Signal Offline Data.Max = 3; Signal Online Data.BitSize = 2; Signal Online Data.BitPosition = 0; Convert Data.Flags = 3; Convert Data.pSigValue = 0;
                  Convert Data.Scaling = 4607182418800017408; Convert Data.Offset = 0; Signal Offline Data.SPN = 594; Signal Offline Data.Name = "Engine Idle Shutdown Driver Alert Mode"; Signal Offline Data.Unit = "bit"; Signal Offline Data.Min = 0; Signal Offline Data.Max = 3; Signal Online Data.BitSize = 2; Signal Online Data.BitPosition = 2; Convert Data.Flags = 3; Convert Data.pSigValue = 0; Convert Data.Scaling = 4607182418800017408; Convert Data.Offset = 0; Signal Offline Data.SPN = 592; Signal Offline Data.Name = "Engine Idle Shutdown Timer Override"; Signal Offline Data.Unit = "bit"; Signal Offline Data.Min = 0; Signal Offline Data.Max = 3; Signal Online Data.BitSize = 2; Signal Online Data.BitPosition = 4; Convert Data.Flags = 3; Convert Data.pSigValue = 0; Convert Data.Scaling = 4607182418800017408; Convert Data.Offset = 0; Signal Offline Data.SPN = 590; Signal Offline Data.Name = "Engine Idle Shutdown Timer State"; Signal Offline Data.Unit = "bit"; Signal Offline Data.Min = 0; Signal Offline Data.Max = 3; Signal Online Data.BitSize = 2; Signal Online Data.BitPosition = 6; Convert Data.Flags = 3; Convert Data.pSigValue = 0; Convert Data.Scaling = 4607182418800017408; Convert Data.Offset = 0; Signal Offline Data.SPN = 591; Signal Offline Data.Name = "Engine Idle Shutdown Timer Function"; Signal Offline Data.Unit = "bit"; Signal Offline Data.Min = 0; Signal Offline Data.Max = 3;
                  Signal Online Data.BitSize = 2; Signal Online Data.BitPosition = 14; Convert Data.Flags = 3; Convert Data.pSigValue = 0; Convert Data.Scaling = 4607182418800017408; Convert Data.Offset = 0; Signal Offline Data.SPN = 985; Signal Offline Data.Name = "A/C High Pressure Fan Switch"; Signal Offline Data.Unit = "bit"; Signal Offline Data.Min = 0; Signal Offline Data.Max = 3; Signal Online Data.BitSize = 2; Signal Online Data.BitPosition = 16; Convert Data.Flags = 3; Convert Data.pSigValue = 0; Convert Data.Scaling = 4607182418800017408; Convert Data.Offset = 0; Signal Offline Data.SPN = 875; Signal Offline Data.Name = "Refrigerant Low Pressure Switch"; Signal Offline Data.Unit = "bit"; Signal Offline Data.Min = 0; Signal Offline Data.Max = 3; Signal Online Data.BitSize = 2; Signal Online Data.BitPosition = 18; Convert Data.Flags = 3; Convert Data.pSigValue = 0; Convert Data.Scaling = 4607182418800017408; Convert Data.Offset = 0; Signal Offline Data.SPN = 605; Signal Offline Data.Name = "Refrigerant High Pressure Switch"; Signal Offline Data.Unit = "bit"; Signal Offline Data.Min = 0; Signal Offline Data.Max = 3; Signal Online Data.BitSize = 2; Signal Online Data.BitPosition = 20; Convert Data.Flags = 3; Convert Data.pSigValue = 0; Convert Data.Scaling = 4607182418800017408; Convert Data.Offset = 0; Signal Offline Data.SPN = 1081;
                  Signal Offline Data.Name = "Engine Wait to Start Lamp"; Signal Offline Data.Unit = "bit"; Signal Offline Data.Min = 0; Signal Offline Data.Max = 3; Signal Online Data.BitSize = 2; Signal Online Data.BitPosition = 24; Convert Data.Flags = 3; Convert Data.pSigValue = 0; Convert Data.Scaling = 4607182418800017408; Convert Data.Offset = 0; Signal Offline Data.SPN = 1110; Signal Offline Data.Name = "Engine Protection System has Shutdown Engine"; Signal Offline Data.Unit = "bit"; Signal Offline Data.Min = 0; Signal Offline Data.Max = 3; Signal Online Data.BitSize = 2; Signal Online Data.BitPosition = 32; Convert Data.Flags = 3; Convert Data.pSigValue = 0; Convert Data.Scaling = 4607182418800017408; Convert Data.Offset = 0; Signal Offline Data.SPN = 1109; Signal Offline Data.Name = "Engine Protection System Approaching Shutdown"; Signal Offline Data.Unit = "bit"; Signal Offline Data.Min = 0; Signal Offline Data.Max = 3; Signal Online Data.BitSize = 2; Signal Online Data.BitPosition = 34; Convert Data.Flags = 3; Convert Data.pSigValue = 0; Convert Data.Scaling = 4607182418800017408; Convert Data.Offset = 0; Signal Offline Data.SPN = 1108; Signal Offline Data.Name = "Engine Protection System Timer Override"; Signal Offline Data.Unit = "bit"; Signal Offline Data.Min = 0; Signal Offline Data.Max = 3; Signal Online Data.BitSize = 2; Signal Online Data.BitPosition = 36; Convert Data.Flags = 3;
                  Convert Data.pSigValue = 0; Convert Data.Scaling = 4607182418800017408; Convert Data.Offset = 0; Signal Offline Data.SPN = 1107; Signal Offline Data.Name = "Engine Protection System Timer State"; Signal Offline Data.Unit = "bit"; Signal Offline Data.Min = 0; Signal Offline Data.Max = 3; Signal Online Data.BitSize = 2; Signal Online Data.BitPosition = 38; Convert Data.Flags = 3; Convert Data.pSigValue = 0; Convert Data.Scaling = 4607182418800017408; Convert Data.Offset = 0; Signal Offline Data.SPN = 1111; Signal Offline Data.Name = "Engine Protection System Configuration"; Signal Offline Data.Unit = "bit"; Signal Offline Data.Min = 0; Signal Offline Data.Max = 3; Signal Online Data.BitSize = 2; Signal Online Data.BitPosition = 46; Convert Data.Flags = 3; Convert Data.pSigValue = 0; Convert Data.Scaling = 4607182418800017408; Convert Data.Offset = 0; Signal Offline Data.SPN = 2815; Signal Offline Data.Name = "Engine Alarm Acknowledge"; Signal Offline Data.Unit = "bit"; Signal Offline Data.Min = 0; Signal Offline Data.Max = 3; Signal Online Data.BitSize = 2; Signal Online Data.BitPosition = 48; Convert Data.Flags = 3; Convert Data.pSigValue = 0; Convert Data.Scaling = 4607182418800017408; Convert Data.Offset = 0; Signal Offline Data.SPN = 2814; Signal Offline Data.Name = "Engine Alarm Output Command Status"; Signal Offline Data.Unit = "bit"; Signal Offline Data.Min = 0;
                  Signal Offline Data.Max = 3; Signal Online Data.BitSize = 2; Signal Online Data.BitPosition = 50; Convert Data.Flags = 3; Convert Data.pSigValue = 0; Convert Data.Scaling = 4607182418800017408; Convert Data.Offset = 0; Signal Offline Data.SPN = 2813; Signal Offline Data.Name = "Engine Air Shutoff Command Status"; Signal Offline Data.Unit = "bit"; Signal Offline Data.Min = 0; Signal Offline Data.Max = 3; Signal Online Data.BitSize = 2; Signal Online Data.BitPosition = 52; Convert Data.Flags = 3; Convert Data.pSigValue = 0; Convert Data.Scaling = 4607182418800017408; Convert Data.Offset = 0; Signal Offline Data.SPN = 2812; Signal Offline Data.Name = "Engine Overspeed Test"; Signal Offline Data.Unit = "bit"; Signal Offline Data.Min = 0; Signal Offline Data.Max = 3; Signal Online Data.BitSize = 2; Signal Online Data.BitPosition = 54; Convert Data.Flags = 3; Convert Data.pSigValue = 0; Convert Data.Scaling = 4607182418800017408; Convert Data.Offset = 0; Signal Offline Data.SPN = 3667; Signal Offline Data.Name = "Engine Air Shutoff Status"; Signal Offline Data.Unit = "bit"; Signal Offline Data.Min = 0; Signal Offline Data.Max = 3; Signal Online Data.BitSize = 2; Signal Online Data.BitPosition = 56; Convert Data.Flags = 3; Convert Data.pSigValue = 0; Convert Data.Scaling = 4607182418800017408; Convert Data.Offset = 0;
                  Signal Offline Data.SPN = 5404; Signal Offline Data.Name = "PTO Shutdown has Shutdown Engine"; Signal Offline Data.Unit = "bit"; Signal Offline Data.Min = 0; Signal Offline Data.Max = 3; Signal Online Data.BitSize = 2; Signal Online Data.BitPosition = 58; Convert Data.Flags = 3; Convert Data.pSigValue = 0; Convert Data.Scaling = 4607182418800017408; Convert Data.Offset = 0; Signal Offline Data.SPN = 5566; Signal Offline Data.Name = "Coolant Level Engine Protection Shutdown Status"; Signal Offline Data.Unit = "bit"; Signal Offline Data.Min = 0; Signal Offline Data.Max = 3; Signal Online Data.BitSize = 2; Signal Online Data.BitPosition = 60; Convert Data.Flags = 3; Convert Data.pSigValue = 0; Convert Data.Scaling = 4607182418800017408; Convert Data.Offset = 0; PG Offline Data.Name = "DM01"; PG Offline Data.Description = "Active Diagnostic Trouble Codes"; PG Online Data.PGN = 65226; PG Online Data.Length (Bytes) = 1785; PG Transmission Settings.Destination Address = 255; PG Transmission Settings.CycleTimeFactor = 1; Signal Offline Data.SPN = 987; Signal Offline Data.Name = "Protect Lamp"; Signal Offline Data.Unit = "bit"; Signal Offline Data.Min = 0; Signal Offline Data.Max = 3; Signal Online Data.BitSize = 2; Signal Online Data.BitPosition = 0; Convert Data.Flags = 3; Convert Data.pSigValue = 0; Convert Data.Scaling = 4607182418800017408; Convert Data.Offset = 0; Signal Offline Data.SPN = 624;
                  Signal Offline Data.Name = "Amber Warning Lamp"; Signal Offline Data.Unit = "bit"; Signal Offline Data.Min = 0; Signal Offline Data.Max = 3; Signal Online Data.BitSize = 2; Signal Online Data.BitPosition = 2; Convert Data.Flags = 3; Convert Data.pSigValue = 0; Convert Data.Scaling = 4607182418800017408; Convert Data.Offset = 0; Signal Offline Data.SPN = 623; Signal Offline Data.Name = "Red Stop Lamp"; Signal Offline Data.Unit = "bit"; Signal Offline Data.Min = 0; Signal Offline Data.Max = 3; Signal Online Data.BitSize = 2; Signal Online Data.BitPosition = 4; Convert Data.Flags = 3; Convert Data.pSigValue = 0; Convert Data.Scaling = 4607182418800017408; Convert Data.Offset = 0; Signal Offline Data.SPN = 1213; Signal Offline Data.Name = "Malfunction Indicator Lamp"; Signal Offline Data.Unit = "bit"; Signal Offline Data.Min = 0; Signal Offline Data.Max = 3; Signal Online Data.BitSize = 2; Signal Online Data.BitPosition = 6; Convert Data.Flags = 3; Convert Data.pSigValue = 0; Convert Data.Scaling = 4607182418800017408; Convert Data.Offset = 0; Signal Offline Data.SPN = 3041; Signal Offline Data.Name = "Flash Protect Lamp"; Signal Offline Data.Unit = "bit"; Signal Offline Data.Min = 0; Signal Offline Data.Max = 3; Signal Online Data.BitSize = 2; Signal Online Data.BitPosition = 8; Convert Data.Flags = 3;
                  Convert Data.pSigValue = 0; Convert Data.Scaling = 4607182418800017408; Convert Data.Offset = 0; Signal Offline Data.SPN = 3040; Signal Offline Data.Name = "Flash Amber Warning Lamp (AWL)"; Signal Offline Data.Unit = "bit"; Signal Offline Data.Min = 0; Signal Offline Data.Max = 3; Signal Online Data.BitSize = 2; Signal Online Data.BitPosition = 10; Convert Data.Flags = 3; Convert Data.pSigValue = 0; Convert Data.Scaling = 4607182418800017408; Convert Data.Offset = 0; Signal Offline Data.SPN = 3039; Signal Offline Data.Name = "Flash Red Stop Lamp (RSL)"; Signal Offline Data.Unit = "bit"; Signal Offline Data.Min = 0; Signal Offline Data.Max = 3; Signal Online Data.BitSize = 2; Signal Online Data.BitPosition = 12; Convert Data.Flags = 3; Convert Data.pSigValue = 0; Convert Data.Scaling = 4607182418800017408; Convert Data.Offset = 0; Signal Offline Data.SPN = 3038; Signal Offline Data.Name = "Flash Malfunction Indicator Lamp (MIL)"; Signal Offline Data.Unit = "bit"; Signal Offline Data.Min = 0; Signal Offline Data.Max = 3; Signal Online Data.BitSize = 2; Signal Online Data.BitPosition = 14; Convert Data.Flags = 3; Convert Data.pSigValue = 0; Convert Data.Scaling = 4607182418800017408; Convert Data.Offset = 0; Signal Offline Data.SPN = 1214; Signal Offline Data.Name = "Suspect Parameter Number"; Signal Offline Data.Unit = "binary"; Signal Offline Data.Min = 0;
                  Signal Offline Data.Max = 524287; Signal Online Data.BitSize = 19; Signal Online Data.BitPosition = 16; Convert Data.Flags = 3; Convert Data.pSigValue = 0; Convert Data.Scaling = 4607182418800017408; Convert Data.Offset = 0; Signal Offline Data.SPN = 1215; Signal Offline Data.Name = "Failure Mode Identifier"; Signal Offline Data.Unit = "binary"; Signal Offline Data.Min = 0; Signal Offline Data.Max = 31; Signal Online Data.BitSize = 5; Signal Online Data.BitPosition = 32; Convert Data.Flags = 3; Convert Data.pSigValue = 0; Convert Data.Scaling = 4607182418800017408; Convert Data.Offset = 0; Signal Offline Data.SPN = 1216; Signal Offline Data.Name = "Occurrence Count"; Signal Offline Data.Unit = "binary"; Signal Offline Data.Min = 0; Signal Offline Data.Max = 127; Signal Online Data.BitSize = 7; Signal Online Data.BitPosition = 40; Convert Data.Flags = 3; Convert Data.pSigValue = 0; Convert Data.Scaling = 4607182418800017408; Convert Data.Offset = 0; Signal Offline Data.SPN = 1706; Signal Offline Data.Name = "SPN Conversion Method"; Signal Offline Data.Unit = "bit"; Signal Offline Data.Min = 0; Signal Offline Data.Max = 1; Signal Online Data.BitSize = 1; Signal Online Data.BitPosition = 47; Convert Data.Flags = 3; Convert Data.pSigValue = 0; Convert Data.Scaling = 4607182418800017408; Convert Data.Offset = 0;
                  Activated PGs = 0
                input  Engine_Load_at_Current_Speed : USINT  // Engine Percent Load At Current Speed
                input  Engine_Speed : REAL  // Engine Speed
                input  Engine_Load_Percent_Torque : BYTE  // Engine Demand – Percent Torque
                input  Engine_Total_Hours_of_Operation : REAL  // Engine Total Hours of Operation
                input  Engine_Total_Revolutions : localTypes:TByteArray4  // Engine Total Revolutions
                input  Engine_Coolant_Temperature : INT  // Engine Coolant Temperature
                input  Engine_Fuel_Temperature : INT  // Engine Fuel Temperature 1
                input  Engine_Oil_Temperature : REAL  // Engine Oil Temperature 1
                input  Eninge_Intercooler_Temperature : INT  // Engine Intercooler Temperature
                input  Engine_Oil_Level : REAL  // Engine Oil Level
                input  Engine_Oil_Pressure : UINT  // Engine Oil Pressure
                input  Engine_Coolant_Pressure : UINT  // Engine Coolant Pressure
                input  Engine_Coolant_Level : REAL  // Engine Coolant Level
                input  Engine_Fuel_Rate : REAL  // Engine Fuel Rate
                input  Engine_Inlet_Temperature : INT  // Engine Intake Manifold 1 Temperature
                input  Engine_Intake_Pressure : UINT  // Engine Air Intake Pressure
                input  Engine_Exhaust_Gas_Temperature : REAL  // Engine Exhaust Gas Temperature
                input  Battery_Potential_Voltage : REAL  // Battery Potential / Power Input 1
                input  Keyswitch_Battery_Potential : REAL  // Keyswitch Battery Potential
                input  Engine_Speed_At_Low_Idle : localTypes:TByteArray2  // Engine Speed At Idle, Point 1 (Engine Configuration)
                input  Engine_Percent_Torque_At_Idle_Point_1_Engine_Configuration_ : BYTE  // Engine Percent Torque At Idle, Point 1 (Engine Configuration)
                input  Engine_Speed_At_Point_2_Engine_Configuration_ : localTypes:TByteArray2  // Engine Speed At Point 2 (Engine Configuration)
                input  Engine_Percent_Torque_At_Point_2_Engine_Configuration_ : BYTE  // Engine Percent Torque At Point 2 (Engine Configuration)
                input  Engine_Speed_At_Point_3_Engine_Configuration_ : localTypes:TByteArray2  // Engine Speed At Point 3 (Engine Configuration)
                input  Engine_Percent_Torque_At_Point_3_Engine_Configuration_ : BYTE  // Engine Percent Torque At Point 3 (Engine Configuration)
                input  Engine_Speed_At_Point_4_Engine_Configuration_ : localTypes:TByteArray2  // Engine Speed At Point 4 (Engine Configuration)
                input  Engine_Percent_Torque_At_Point_4_Engine_Configuration_ : BYTE  // Engine Percent Torque At Point 4 (Engine Configuration)
                input  Engine_Speed_At_Point_5_Engine_Configuration_ : localTypes:TByteArray2  // Engine Speed At Point 5 (Engine Configuration)
                input  Engine_Percent_Torque_At_Point_5_Engine_Configuration_ : BYTE  // Engine Percent Torque At Point 5 (Engine Configuration)
                input  Engine_Speed_At_High_Idle : localTypes:TByteArray2  // Engine Speed At High Idle, Point 6 (Engine Configuration)
                input  Engine_Gain_Kp_Of_The_Endspeed_Governor_Engine_Configuration_ : localTypes:TByteArray2  // Engine Gain (Kp) Of The Endspeed Governor (Engine Configuration)
                input  Engine_Reference_Torque_Engine_Configuration_ : localTypes:TByteArray2  // Engine Reference Torque (Engine Configuration)
                input  Engine_Maximum_Momentary_Override_Speed_Point_7_Engine_Configuration_ : localTypes:TByteArray2  // Engine Maximum Momentary Override Speed, Point 7 (Engine Configuration)
                input  Engine_Maximum_Momentary_Override_Time_Limit_Engine_Configuration_ : BYTE  // Engine Maximum Momentary Override Time Limit (Engine Configuration)
                input  Engine_Requested_Speed_Control_Range_Lower_Limit_Engine_Configuration_ : BYTE  // Engine Requested Speed Control Range Lower Limit (Engine Configuration)
                input  Engine_Requested_Speed_Control_Range_Upper_Limit_Engine_Configuration_ : BYTE  // Engine Requested Speed Control Range Upper Limit (Engine Configuration)
                input  Engine_Requested_Torque_Control_Range_Lower_Limit_Engine_Configuration_ : BYTE  // Engine Requested Torque Control Range Lower Limit (Engine Configuration)
                input  Engine_Requested_Torque_Control_Range_Upper_Limit_Engine_Configuration_ : BYTE  // Engine Requested Torque Control Range Upper Limit (Engine Configuration)
                input  Engine_Extended_Range_Requested_Speed_Control_Range_Upper_Limit_Engine_configuration_ : localTypes:TByteArray2  // Engine Extended Range Requested Speed Control Range Upper Limit (Engine configuration)
                input  Engine_Moment_of_Inertia : localTypes:TByteArray2  // Engine Moment of Inertia
                input  Engine_Default_Torque_Limit : localTypes:TByteArray2  // Engine Default Torque Limit
                input  Support_Variable_Rate_TSC1_Message : BYTE  // Support Variable Rate TSC1 Message
                input  Support_TSC1_Control_Purpose_Group_1 : BYTE  // Support TSC1 Control Purpose Group 1
                input  Support_TSC1_Control_Purpose_Group_2 : BYTE  // Support TSC1 Control Purpose Group 2
                input  Support_TSC1_Control_Purpose_Group_3 : BYTE  // Support TSC1 Control Purpose Group 3
                input  Support_TSC1_Control_Purpose_Group_4 : BYTE  // Support TSC1 Control Purpose Group 4
                input  Nominal_Friction_Percent_Torque : BYTE  // Nominal Friction - Percent Torque
                input  Engine_Desired_Operating_Speed : localTypes:TByteArray2  // Engine's Desired Operating Speed
                input  Auxiliary_Temperature_1 : BYTE  // Auxiliary Temperature 1
                input  Auxiliary_Pressure_1 : BYTE  // Auxiliary Pressure #1
                input  Engine_Idle_Shutdown_has_Shutdown_Engine : BYTE  // Engine Idle Shutdown has Shutdown Engine
                input  Engine_Idle_Shutdown_Driver_Alert_Mode : BYTE  // Engine Idle Shutdown Driver Alert Mode
                input  Engine_Idle_Shutdown_Timer_Override : BYTE  // Engine Idle Shutdown Timer Override
                input  Engine_Idle_Shutdown_Timer_State : BYTE  // Engine Idle Shutdown Timer State
                input  Engine_Idle_Shutdown_Timer_Function : BYTE  // Engine Idle Shutdown Timer Function
                input  A_C_High_Pressure_Fan_Switch : BYTE  // A/C High Pressure Fan Switch
                input  Refrigerant_Low_Pressure_Switch : BYTE  // Refrigerant Low Pressure Switch
                input  Refrigerant_High_Pressure_Switch : BYTE  // Refrigerant High Pressure Switch
                input  Engine_Wait_to_Start_Lamp : USINT  // Engine Wait to Start Lamp
                input  Engine_Protection_System_has_Shutdown_Engine : BYTE  // Engine Protection System has Shutdown Engine
                input  Engine_Protection_System_Approaching_Shutdown : BYTE  // Engine Protection System Approaching Shutdown
                input  Engine_Protection_System_Timer_Override : BYTE  // Engine Protection System Timer Override
                input  Engine_Protection_System_Timer_State : BYTE  // Engine Protection System Timer State
                input  Engine_Protection_System_Configuration : BYTE  // Engine Protection System Configuration
                input  Engine_Alarm_Acknowledge : BYTE  // Engine Alarm Acknowledge
                input  Engine_Alarm_Output_Command_Status : BYTE  // Engine Alarm Output Command Status
                input  Engine_Air_Shutoff_Command_Status : BYTE  // Engine Air Shutoff Command Status
                input  Engine_Overspeed_Test : BYTE  // Engine Overspeed Test
                input  Engine_Air_Shutoff_Status : BYTE  // Engine Air Shutoff Status
                input  PTO_Shutdown_has_Shutdown_Engine : BYTE  // PTO Shutdown has Shutdown Engine
                input  Coolant_Level_Engine_Protection_Shutdown_Status : BYTE  // Coolant Level Engine Protection Shutdown Status
                input  Protect_Lamp_1 : USINT  // Protect Lamp
                input  Amber_Warning_Lamp_1 : USINT  // Amber Warning Lamp
                input  Red_Stop_Lamp_1 : USINT  // Red Stop Lamp
                input  Malfunction_Indicator_Lamp_1 : BYTE  // Malfunction Indicator Lamp
                input  Flash_Protect_Lamp_1 : BYTE  // Flash Protect Lamp
                input  Flash_Amber_Warning_Lamp_AWL_1 : BYTE  // Flash Amber Warning Lamp (AWL)
                input  Flash_Red_Stop_Lamp_RSL_1 : BYTE  // Flash Red Stop Lamp (RSL)
                input  Flash_Malfunction_Indicator_Lamp_MIL_1 : BYTE  // Flash Malfunction Indicator Lamp (MIL)
                input  Suspect_Parameter_Number_1 : UDINT  // Suspect Parameter Number
                input  Failure_Mode_Identifier_1 : USINT  // Failure Mode Identifier
                input  Occurrence_Count_1 : USINT  // Occurrence Count
                input  SPN_Conversion_Method_1 : BIT  // SPN Conversion Method
                unmapped channels: Accelerator Pedal 1 Low Idle Switch, Accelerator Pedal Kickdown Switch, Road Speed Limit Status, Accelerator Pedal 2 Low Idle Switch, Accelerator Pedal Position 1, Remote Accelerator Pedal Position, Accelerator Pedal Position 2, Vehicle Acceleration Rate Limit Status, Momentary Engine Maximum Power Enable Feedback, DPF Thermal Management Active, SCR Thermal Management Active, Actual Maximum Available Engine - Percent Torque, Estimated Pumping - Percent Torque, Engine Torque Mode, Actual Engine - Percent Torque High Resolution, Driver's Demand Engine - Percent Torque, Actual Engine - Percent Torque, Source Address of Controlling Device for Engine Control, Engine Starter Mode, Engine Turbocharger Oil Temperature, Engine Intercooler Thermostat Opening, Engine Fuel Delivery Pressure, Engine Extended Crankcase Blow-by Pressure, Engine Crankcase Pressure, Engine Instantaneous Fuel Economy, Engine Average Fuel Economy, Engine Throttle Valve 1 Position, Engine Throttle Valve 2 Position, Engine Diesel Particulate Filter Intake Pressure, Engine Intake Manifold #1 Pressure, Engine Air Filter 1 Differential Pressure, Engine Coolant Filter Differential Pressure, Net Battery Current, Alternator Current, Charging System Potential (Voltage), Engine's Desired Operating Speed Asymmetry Adjustment, Estimated Engine Parasitic Losses - Percent Torque, Aftertreatment 1 Exhaust Gas Mass Flow, Aftertreatment 1 Intake Dew Point, Aftertreatment 1 Exhaust Dew Point,
                  Aftertreatment 2 Intake Dew Point, Aftertreatment 2 Exhaust Dew Point
        CANbus_0 : CANbus, ifm electronic, version 1.0.1.1
          CANopen_Manager : CANopen_Manager, 3S - Smart Software Solutions GmbH, version 3.5.10.0
              settings: Sync CycleTime in Microseconds = 100000; Enable Sync generation = TRUE; Synchronous Window Length = 120000; Heartbeat Node ID = 1; CANopen NodeID = 1; ConfigVersion = 50659584
            CDJCAN_CO_3_X : CDJCAN_XYZW_AXIS, Frenzel + Berg Elektronik, order no. CO4013, version Revision=16#00000001, FileVersion=1.0, File=CDJCAN_XYZW_AXIS.eds
                settings: General Options.Create all SDOs = TRUE; General Options.Optional Device = TRUE; General Options.Reset Node = FALSE; NODEIDSAVED = 14; SDO Timeout = 1000000; PDO_Autoconfig = FALSE; EXPERTSETTINGS = True; Emergency-General Parameters.Emergency COBID = 16#0000008E; Heartbeat-Producer Time = 200; PDO 16#1400.COBID = 16#0000020E; PDO 16#1400.Transmission Type = 16#00; Process by CANopenManager = TRUE; PDO 16#1800.COBID = 16#0000018E; Process by CANopenManager = TRUE; PDO 16#1801.COBID = 16#0000028E; Process by CANopenManager = TRUE; Write Output Byte_1.Subindex = 16#01; DigInput8_0.Subindex = 16#01; DigInput8_1.Subindex = 16#02; DigInput8_2.Subindex = 16#03; Joystick X Axis.Subindex = 16#01; Joystick Y Axis.Subindex = 16#02; Joystick Z Axis.Subindex = 16#03; SDO List.Set COB-ID sync.Index = 16#1005; SDO List.Set COB-ID sync.Subindex = 16#00; SDO List.Set COB-ID sync.Value = 16#00000080; SDO List.Set COB-ID sync.Size = 32; SDO List.Set COB-ID sync.AbortIfError = FALSE; SDO List.Set COB-ID sync.JumpToLine = FALSE; SDO List.Set COB-ID sync.Line = 0; SDO List.Set Guardtime.Index = 16#100C; SDO List.Set Guardtime.Subindex = 16#00; SDO List.Set Guardtime.Value = 16#00000000; SDO List.Set Guardtime.Size = 16; SDO List.Set Guardtime.AbortIfError = FALSE; SDO List.Set Guardtime.JumpToLine = FALSE; SDO List.Set Guardtime.Line = 0; SDO List.Set Lifetime.Index = 16#100D; SDO List.Set Lifetime.Subindex = 16#00; SDO List.Set Lifetime.Value = 16#00000000;
                  SDO List.Set Lifetime.Size = 8; SDO List.Set Lifetime.AbortIfError = FALSE; SDO List.Set Lifetime.JumpToLine = FALSE; SDO List.Set Lifetime.Line = 0; SDO List.Disable Emcy CobID.Index = 16#1014; SDO List.Disable Emcy CobID.Subindex = 16#00; SDO List.Disable Emcy CobID.Value = 16#8000008E; SDO List.Disable Emcy CobID.Size = 32; SDO List.Disable Emcy CobID.AbortIfError = FALSE; SDO List.Disable Emcy CobID.JumpToLine = FALSE; SDO List.Disable Emcy CobID.Line = 0; SDO List.Set Emcy CobID.Index = 16#1014; SDO List.Set Emcy CobID.Subindex = 16#00; SDO List.Set Emcy CobID.Value = 16#0000008E; SDO List.Set Emcy CobID.Size = 32; SDO List.Set Emcy CobID.AbortIfError = FALSE; SDO List.Set Emcy CobID.JumpToLine = FALSE; SDO List.Set Emcy CobID.Line = 0; SDO List.Set Heartbeat Producer.Index = 16#1017; SDO List.Set Heartbeat Producer.Subindex = 16#00; SDO List.Set Heartbeat Producer.Value = 16#000000C8; SDO List.Set Heartbeat Producer.Size = 16; SDO List.Set Heartbeat Producer.AbortIfError = FALSE; SDO List.Set Heartbeat Producer.JumpToLine = FALSE; SDO List.Set Heartbeat Producer.Line = 0; SDO List.Disable PDO.Index = 16#1400; SDO List.Disable PDO.Subindex = 16#01; SDO List.Disable PDO.Value = 16#8000020E; SDO List.Disable PDO.Size = 32; SDO List.Disable PDO.AbortIfError = FALSE; SDO List.Disable PDO.JumpToLine = FALSE; SDO List.Disable PDO.Line = 0; SDO List.Set transmission type.Index = 16#1400; SDO List.Set transmission type.Subindex = 16#02; SDO List.Set transmission type.Value = 16#00; SDO List.Set transmission type.Size = 8; SDO List.Set transmission type.AbortIfError = FALSE; SDO List.Set transmission type.JumpToLine = FALSE; SDO List.Set transmission type.Line = 0; SDO List.Clear pdo mapping.Index = 16#1600;
                  SDO List.Clear pdo mapping.Subindex = 16#00; SDO List.Clear pdo mapping.Value = 16#0; SDO List.Clear pdo mapping.Size = 8; SDO List.Clear pdo mapping.AbortIfError = FALSE; SDO List.Clear pdo mapping.JumpToLine = FALSE; SDO List.Clear pdo mapping.Line = 0; SDO List.Set Mapping.Index = 16#1600; SDO List.Set Mapping.Subindex = 16#01; SDO List.Set Mapping.Value = 16#62000108; SDO List.Set Mapping.Size = 32; SDO List.Set Mapping.AbortIfError = FALSE; SDO List.Set Mapping.JumpToLine = FALSE; SDO List.Set Mapping.Line = 0; SDO List.Set number of mappings.Index = 16#1600; SDO List.Set number of mappings.Subindex = 16#00; SDO List.Set number of mappings.Value = 16#01; SDO List.Set number of mappings.Size = 8; SDO List.Set number of mappings.AbortIfError = FALSE; SDO List.Set number of mappings.JumpToLine = FALSE; SDO List.Set number of mappings.Line = 0; SDO List.Set and enable COB-ID.Index = 16#1400; SDO List.Set and enable COB-ID.Subindex = 16#01; SDO List.Set and enable COB-ID.Value = 16#0000020E; SDO List.Set and enable COB-ID.Size = 32; SDO List.Set and enable COB-ID.AbortIfError = FALSE; SDO List.Set and enable COB-ID.JumpToLine = FALSE; SDO List.Set and enable COB-ID.Line = 0; SDO List.Disable PDO.Index = 16#1800; SDO List.Disable PDO.Subindex = 16#01; SDO List.Disable PDO.Value = 16#8000018E; SDO List.Disable PDO.Size = 32; SDO List.Disable PDO.AbortIfError = FALSE; SDO List.Disable PDO.JumpToLine = FALSE; SDO List.Disable PDO.Line = 0; SDO List.Set transmission type.Index = 16#1800; SDO List.Set transmission type.Subindex = 16#02; SDO List.Set transmission type.Value = 16#FF; SDO List.Set transmission type.Size = 8; SDO List.Set transmission type.AbortIfError = FALSE; SDO List.Set transmission type.JumpToLine = FALSE;
                  SDO List.Set transmission type.Line = 0; SDO List.Set inhibit time.Index = 16#1800; SDO List.Set inhibit time.Subindex = 16#03; SDO List.Set inhibit time.Value = 16#0000; SDO List.Set inhibit time.Size = 16; SDO List.Set inhibit time.AbortIfError = FALSE; SDO List.Set inhibit time.JumpToLine = FALSE; SDO List.Set inhibit time.Line = 0; SDO List.Set event time.Index = 16#1800; SDO List.Set event time.Subindex = 16#05; SDO List.Set event time.Value = 16#0000; SDO List.Set event time.Size = 16; SDO List.Set event time.AbortIfError = FALSE; SDO List.Set event time.JumpToLine = FALSE; SDO List.Set event time.Line = 0; SDO List.Clear pdo mapping.Index = 16#1A00; SDO List.Clear pdo mapping.Subindex = 16#00; SDO List.Clear pdo mapping.Value = 16#0; SDO List.Clear pdo mapping.Size = 8; SDO List.Clear pdo mapping.AbortIfError = FALSE; SDO List.Clear pdo mapping.JumpToLine = FALSE; SDO List.Clear pdo mapping.Line = 0; SDO List.Set Mapping.Index = 16#1A00; SDO List.Set Mapping.Subindex = 16#01; SDO List.Set Mapping.Value = 16#60000108; SDO List.Set Mapping.Size = 32; SDO List.Set Mapping.AbortIfError = FALSE; SDO List.Set Mapping.JumpToLine = FALSE; SDO List.Set Mapping.Line = 0; SDO List.Set Mapping.Index = 16#1A00; SDO List.Set Mapping.Subindex = 16#02; SDO List.Set Mapping.Value = 16#60000208; SDO List.Set Mapping.Size = 32; SDO List.Set Mapping.AbortIfError = FALSE; SDO List.Set Mapping.JumpToLine = FALSE; SDO List.Set Mapping.Line = 0; SDO List.Set Mapping.Index = 16#1A00; SDO List.Set Mapping.Subindex = 16#03; SDO List.Set Mapping.Value = 16#60000308; SDO List.Set Mapping.Size = 32;
                  SDO List.Set Mapping.AbortIfError = FALSE; SDO List.Set Mapping.JumpToLine = FALSE; SDO List.Set Mapping.Line = 0; SDO List.Set number of mappings.Index = 16#1A00; SDO List.Set number of mappings.Subindex = 16#00; SDO List.Set number of mappings.Value = 16#03; SDO List.Set number of mappings.Size = 8; SDO List.Set number of mappings.AbortIfError = FALSE; SDO List.Set number of mappings.JumpToLine = FALSE; SDO List.Set number of mappings.Line = 0; SDO List.Set and enable COB-ID.Index = 16#1800; SDO List.Set and enable COB-ID.Subindex = 16#01; SDO List.Set and enable COB-ID.Value = 16#0000018E; SDO List.Set and enable COB-ID.Size = 32; SDO List.Set and enable COB-ID.AbortIfError = FALSE; SDO List.Set and enable COB-ID.JumpToLine = FALSE; SDO List.Set and enable COB-ID.Line = 0; SDO List.Disable PDO.Index = 16#1801; SDO List.Disable PDO.Subindex = 16#01; SDO List.Disable PDO.Value = 16#8000028E; SDO List.Disable PDO.Size = 32; SDO List.Disable PDO.AbortIfError = FALSE; SDO List.Disable PDO.JumpToLine = FALSE; SDO List.Disable PDO.Line = 0; SDO List.Set transmission type.Index = 16#1801; SDO List.Set transmission type.Subindex = 16#02; SDO List.Set transmission type.Value = 16#FF; SDO List.Set transmission type.Size = 8; SDO List.Set transmission type.AbortIfError = FALSE; SDO List.Set transmission type.JumpToLine = FALSE; SDO List.Set transmission type.Line = 0; SDO List.Set inhibit time.Index = 16#1801; SDO List.Set inhibit time.Subindex = 16#03; SDO List.Set inhibit time.Value = 16#0000; SDO List.Set inhibit time.Size = 16; SDO List.Set inhibit time.AbortIfError = FALSE; SDO List.Set inhibit time.JumpToLine = FALSE; SDO List.Set inhibit time.Line = 0; SDO List.Set event time.Index = 16#1801; SDO List.Set event time.Subindex = 16#05;
                  SDO List.Set event time.Value = 16#0000; SDO List.Set event time.Size = 16; SDO List.Set event time.AbortIfError = FALSE; SDO List.Set event time.JumpToLine = FALSE; SDO List.Set event time.Line = 0; SDO List.Clear pdo mapping.Index = 16#1A01; SDO List.Clear pdo mapping.Subindex = 16#00; SDO List.Clear pdo mapping.Value = 16#0; SDO List.Clear pdo mapping.Size = 8; SDO List.Clear pdo mapping.AbortIfError = FALSE; SDO List.Clear pdo mapping.JumpToLine = FALSE; SDO List.Clear pdo mapping.Line = 0; SDO List.Set Mapping.Index = 16#1A01; SDO List.Set Mapping.Subindex = 16#01; SDO List.Set Mapping.Value = 16#64010110; SDO List.Set Mapping.Size = 32; SDO List.Set Mapping.AbortIfError = FALSE; SDO List.Set Mapping.JumpToLine = FALSE; SDO List.Set Mapping.Line = 0; SDO List.Set Mapping.Index = 16#1A01; SDO List.Set Mapping.Subindex = 16#02; SDO List.Set Mapping.Value = 16#64010210; SDO List.Set Mapping.Size = 32; SDO List.Set Mapping.AbortIfError = FALSE; SDO List.Set Mapping.JumpToLine = FALSE; SDO List.Set Mapping.Line = 0; SDO List.Set Mapping.Index = 16#1A01; SDO List.Set Mapping.Subindex = 16#03; SDO List.Set Mapping.Value = 16#64010310; SDO List.Set Mapping.Size = 32; SDO List.Set Mapping.AbortIfError = FALSE; SDO List.Set Mapping.JumpToLine = FALSE; SDO List.Set Mapping.Line = 0; SDO List.Set number of mappings.Index = 16#1A01; SDO List.Set number of mappings.Subindex = 16#00; SDO List.Set number of mappings.Value = 16#03; SDO List.Set number of mappings.Size = 8; SDO List.Set number of mappings.AbortIfError = FALSE; SDO List.Set number of mappings.JumpToLine = FALSE; SDO List.Set number of mappings.Line = 0;
                  SDO List.Set and enable COB-ID.Index = 16#1801; SDO List.Set and enable COB-ID.Subindex = 16#01; SDO List.Set and enable COB-ID.Value = 16#0000028E; SDO List.Set and enable COB-ID.Size = 32; SDO List.Set and enable COB-ID.AbortIfError = FALSE; SDO List.Set and enable COB-ID.JumpToLine = FALSE; SDO List.Set and enable COB-ID.Line = 0; SDO List.Global Interrupt Enable Digital In.Index = 16#6005; SDO List.Global Interrupt Enable Digital In.Subindex = 16#00; SDO List.Global Interrupt Enable Digital In.Value = 16#FF; SDO List.Global Interrupt Enable Digital In.Size = 8; SDO List.Global Interrupt Enable Digital In.AbortIfError = FALSE; SDO List.Global Interrupt Enable Digital In.JumpToLine = FALSE; SDO List.Global Interrupt Enable Digital In.Line = 0; SDO List.Analog Input Interrupt Enable.Index = 16#6423; SDO List.Analog Input Interrupt Enable.Subindex = 16#00; SDO List.Analog Input Interrupt Enable.Value = 1; SDO List.Analog Input Interrupt Enable.Size = 8; SDO List.Analog Input Interrupt Enable.AbortIfError = FALSE; SDO List.Analog Input Interrupt Enable.JumpToLine = FALSE; SDO List.Analog Input Interrupt Enable.Line = 0; SDO List.CAN Restart Delay.Index = 16#2180; SDO List.CAN Restart Delay.Subindex = 16#00; SDO List.CAN Restart Delay.Value = 0; SDO List.CAN Restart Delay.Size = 16; SDO List.CAN Restart Delay.AbortIfError = FALSE; SDO List.CAN Restart Delay.JumpToLine = FALSE; SDO List.CAN Restart Delay.Line = 0; SDO List.Debounce Time digital Input1.Index = 16#5003; SDO List.Debounce Time digital Input1.Subindex = 16#01; SDO List.Debounce Time digital Input1.Value = 40; SDO List.Debounce Time digital Input1.Size = 8; SDO List.Debounce Time digital Input1.AbortIfError = FALSE; SDO List.Debounce Time digital Input1.JumpToLine = FALSE; SDO List.Debounce Time digital Input1.Line = 0; SDO List.Debounce Time digital Input2.Index = 16#5003; SDO List.Debounce Time digital Input2.Subindex = 16#02; SDO List.Debounce Time digital Input2.Value = 40; SDO List.Debounce Time digital Input2.Size = 8; SDO List.Debounce Time digital Input2.AbortIfError = FALSE;
                  SDO List.Debounce Time digital Input2.JumpToLine = FALSE; SDO List.Debounce Time digital Input2.Line = 0; SDO List.Debounce Time digital Input3.Index = 16#5003; SDO List.Debounce Time digital Input3.Subindex = 16#03; SDO List.Debounce Time digital Input3.Value = 40; SDO List.Debounce Time digital Input3.Size = 8; SDO List.Debounce Time digital Input3.AbortIfError = FALSE; SDO List.Debounce Time digital Input3.JumpToLine = FALSE; SDO List.Debounce Time digital Input3.Line = 0; SDO List.Debounce Time digital Input4.Index = 16#5003; SDO List.Debounce Time digital Input4.Subindex = 16#04; SDO List.Debounce Time digital Input4.Value = 40; SDO List.Debounce Time digital Input4.Size = 8; SDO List.Debounce Time digital Input4.AbortIfError = FALSE; SDO List.Debounce Time digital Input4.JumpToLine = FALSE; SDO List.Debounce Time digital Input4.Line = 0; SDO List.Debounce Time digital Input5.Index = 16#5003; SDO List.Debounce Time digital Input5.Subindex = 16#05; SDO List.Debounce Time digital Input5.Value = 40; SDO List.Debounce Time digital Input5.Size = 8; SDO List.Debounce Time digital Input5.AbortIfError = FALSE; SDO List.Debounce Time digital Input5.JumpToLine = FALSE; SDO List.Debounce Time digital Input5.Line = 0; SDO List.Debounce Time digital Input6.Index = 16#5003; SDO List.Debounce Time digital Input6.Subindex = 16#06; SDO List.Debounce Time digital Input6.Value = 40; SDO List.Debounce Time digital Input6.Size = 8; SDO List.Debounce Time digital Input6.AbortIfError = FALSE; SDO List.Debounce Time digital Input6.JumpToLine = FALSE; SDO List.Debounce Time digital Input6.Line = 0; SDO List.Debounce Time digital Input7.Index = 16#5003; SDO List.Debounce Time digital Input7.Subindex = 16#07; SDO List.Debounce Time digital Input7.Value = 40; SDO List.Debounce Time digital Input7.Size = 8; SDO List.Debounce Time digital Input7.AbortIfError = FALSE; SDO List.Debounce Time digital Input7.JumpToLine = FALSE; SDO List.Debounce Time digital Input7.Line = 0; SDO List.Debounce Time digital Input8.Index = 16#5003; SDO List.Debounce Time digital Input8.Subindex = 16#08; SDO List.Debounce Time digital Input8.Value = 40;
                  SDO List.Debounce Time digital Input8.Size = 8; SDO List.Debounce Time digital Input8.AbortIfError = FALSE; SDO List.Debounce Time digital Input8.JumpToLine = FALSE; SDO List.Debounce Time digital Input8.Line = 0; SDO List.Debounce Time digital Input9.Index = 16#5003; SDO List.Debounce Time digital Input9.Subindex = 16#09; SDO List.Debounce Time digital Input9.Value = 40; SDO List.Debounce Time digital Input9.Size = 8; SDO List.Debounce Time digital Input9.AbortIfError = FALSE; SDO List.Debounce Time digital Input9.JumpToLine = FALSE; SDO List.Debounce Time digital Input9.Line = 0; SDO List.Debounce Time digital Input10.Index = 16#5003; SDO List.Debounce Time digital Input10.Subindex = 16#0A; SDO List.Debounce Time digital Input10.Value = 40; SDO List.Debounce Time digital Input10.Size = 8; SDO List.Debounce Time digital Input10.AbortIfError = FALSE; SDO List.Debounce Time digital Input10.JumpToLine = FALSE; SDO List.Debounce Time digital Input10.Line = 0; SDO List.Debounce Time digital Input11.Index = 16#5003; SDO List.Debounce Time digital Input11.Subindex = 16#0B; SDO List.Debounce Time digital Input11.Value = 40; SDO List.Debounce Time digital Input11.Size = 8; SDO List.Debounce Time digital Input11.AbortIfError = FALSE; SDO List.Debounce Time digital Input11.JumpToLine = FALSE; SDO List.Debounce Time digital Input11.Line = 0; SDO List.Debounce Time digital Input12.Index = 16#5003; SDO List.Debounce Time digital Input12.Subindex = 16#0C; SDO List.Debounce Time digital Input12.Value = 40; SDO List.Debounce Time digital Input12.Size = 8; SDO List.Debounce Time digital Input12.AbortIfError = FALSE; SDO List.Debounce Time digital Input12.JumpToLine = FALSE; SDO List.Debounce Time digital Input12.Line = 0; SDO List.Debounce Time digital Input13.Index = 16#5003; SDO List.Debounce Time digital Input13.Subindex = 16#0D; SDO List.Debounce Time digital Input13.Value = 40; SDO List.Debounce Time digital Input13.Size = 8; SDO List.Debounce Time digital Input13.AbortIfError = FALSE; SDO List.Debounce Time digital Input13.JumpToLine = FALSE; SDO List.Debounce Time digital Input13.Line = 0; SDO List.Debounce Time digital Input14.Index = 16#5003;
                  SDO List.Debounce Time digital Input14.Subindex = 16#0E; SDO List.Debounce Time digital Input14.Value = 40; SDO List.Debounce Time digital Input14.Size = 8; SDO List.Debounce Time digital Input14.AbortIfError = FALSE; SDO List.Debounce Time digital Input14.JumpToLine = FALSE; SDO List.Debounce Time digital Input14.Line = 0; SDO List.Debounce Time digital Input15.Index = 16#5003; SDO List.Debounce Time digital Input15.Subindex = 16#0F; SDO List.Debounce Time digital Input15.Value = 40; SDO List.Debounce Time digital Input15.Size = 8; SDO List.Debounce Time digital Input15.AbortIfError = FALSE; SDO List.Debounce Time digital Input15.JumpToLine = FALSE; SDO List.Debounce Time digital Input15.Line = 0; SDO List.Debounce Time digital Input16.Index = 16#5003; SDO List.Debounce Time digital Input16.Subindex = 16#10; SDO List.Debounce Time digital Input16.Value = 40; SDO List.Debounce Time digital Input16.Size = 8; SDO List.Debounce Time digital Input16.AbortIfError = FALSE; SDO List.Debounce Time digital Input16.JumpToLine = FALSE; SDO List.Debounce Time digital Input16.Line = 0; SDO List.Debounce Time digital Input17.Index = 16#5003; SDO List.Debounce Time digital Input17.Subindex = 16#11; SDO List.Debounce Time digital Input17.Value = 40; SDO List.Debounce Time digital Input17.Size = 8; SDO List.Debounce Time digital Input17.AbortIfError = FALSE; SDO List.Debounce Time digital Input17.JumpToLine = FALSE; SDO List.Debounce Time digital Input17.Line = 0; SDO List.Debounce Time digital Input18.Index = 16#5003; SDO List.Debounce Time digital Input18.Subindex = 16#12; SDO List.Debounce Time digital Input18.Value = 40; SDO List.Debounce Time digital Input18.Size = 8; SDO List.Debounce Time digital Input18.AbortIfError = FALSE; SDO List.Debounce Time digital Input18.JumpToLine = FALSE; SDO List.Debounce Time digital Input18.Line = 0; SDO List.Debounce Time digital Input19.Index = 16#5003; SDO List.Debounce Time digital Input19.Subindex = 16#13; SDO List.Debounce Time digital Input19.Value = 40; SDO List.Debounce Time digital Input19.Size = 8; SDO List.Debounce Time digital Input19.AbortIfError = FALSE; SDO List.Debounce Time digital Input19.JumpToLine = FALSE;
                  SDO List.Debounce Time digital Input19.Line = 0; SDO List.Debounce Time digital Input20.Index = 16#5003; SDO List.Debounce Time digital Input20.Subindex = 16#14; SDO List.Debounce Time digital Input20.Value = 40; SDO List.Debounce Time digital Input20.Size = 8; SDO List.Debounce Time digital Input20.AbortIfError = FALSE; SDO List.Debounce Time digital Input20.JumpToLine = FALSE; SDO List.Debounce Time digital Input20.Line = 0; SDO List.Debounce Time digital Input21.Index = 16#5003; SDO List.Debounce Time digital Input21.Subindex = 16#15; SDO List.Debounce Time digital Input21.Value = 40; SDO List.Debounce Time digital Input21.Size = 8; SDO List.Debounce Time digital Input21.AbortIfError = FALSE; SDO List.Debounce Time digital Input21.JumpToLine = FALSE; SDO List.Debounce Time digital Input21.Line = 0; SDO List.Debounce Time digital Input22.Index = 16#5003; SDO List.Debounce Time digital Input22.Subindex = 16#16; SDO List.Debounce Time digital Input22.Value = 40; SDO List.Debounce Time digital Input22.Size = 8; SDO List.Debounce Time digital Input22.AbortIfError = FALSE; SDO List.Debounce Time digital Input22.JumpToLine = FALSE; SDO List.Debounce Time digital Input22.Line = 0; SDO List.Debounce Time digital Input23.Index = 16#5003; SDO List.Debounce Time digital Input23.Subindex = 16#17; SDO List.Debounce Time digital Input23.Value = 40; SDO List.Debounce Time digital Input23.Size = 8; SDO List.Debounce Time digital Input23.AbortIfError = FALSE; SDO List.Debounce Time digital Input23.JumpToLine = FALSE; SDO List.Debounce Time digital Input23.Line = 0; SDO List.Debounce Time digital Input24.Index = 16#5003; SDO List.Debounce Time digital Input24.Subindex = 16#18; SDO List.Debounce Time digital Input24.Value = 40; SDO List.Debounce Time digital Input24.Size = 8; SDO List.Debounce Time digital Input24.AbortIfError = FALSE; SDO List.Debounce Time digital Input24.JumpToLine = FALSE; SDO List.Debounce Time digital Input24.Line = 0; SDO List.Debounce Time digital Input25.Index = 16#5003; SDO List.Debounce Time digital Input25.Subindex = 16#19; SDO List.Debounce Time digital Input25.Value = 40; SDO List.Debounce Time digital Input25.Size = 8;
                  SDO List.Debounce Time digital Input25.AbortIfError = FALSE; SDO List.Debounce Time digital Input25.JumpToLine = FALSE; SDO List.Debounce Time digital Input25.Line = 0; SDO List.Debounce Time digital Input26.Index = 16#5003; SDO List.Debounce Time digital Input26.Subindex = 16#1A; SDO List.Debounce Time digital Input26.Value = 40; SDO List.Debounce Time digital Input26.Size = 8; SDO List.Debounce Time digital Input26.AbortIfError = FALSE; SDO List.Debounce Time digital Input26.JumpToLine = FALSE; SDO List.Debounce Time digital Input26.Line = 0; SDO List.Debounce Time digital Input27.Index = 16#5003; SDO List.Debounce Time digital Input27.Subindex = 16#1B; SDO List.Debounce Time digital Input27.Value = 40; SDO List.Debounce Time digital Input27.Size = 8; SDO List.Debounce Time digital Input27.AbortIfError = FALSE; SDO List.Debounce Time digital Input27.JumpToLine = FALSE; SDO List.Debounce Time digital Input27.Line = 0; SDO List.Debounce Time digital Input28.Index = 16#5003; SDO List.Debounce Time digital Input28.Subindex = 16#1C; SDO List.Debounce Time digital Input28.Value = 40; SDO List.Debounce Time digital Input28.Size = 8; SDO List.Debounce Time digital Input28.AbortIfError = FALSE; SDO List.Debounce Time digital Input28.JumpToLine = FALSE; SDO List.Debounce Time digital Input28.Line = 0; SDO List.Debounce Time digital Input29.Index = 16#5003; SDO List.Debounce Time digital Input29.Subindex = 16#1D; SDO List.Debounce Time digital Input29.Value = 40; SDO List.Debounce Time digital Input29.Size = 8; SDO List.Debounce Time digital Input29.AbortIfError = FALSE; SDO List.Debounce Time digital Input29.JumpToLine = FALSE; SDO List.Debounce Time digital Input29.Line = 0; SDO List.Debounce Time digital Input30.Index = 16#5003; SDO List.Debounce Time digital Input30.Subindex = 16#1E; SDO List.Debounce Time digital Input30.Value = 40; SDO List.Debounce Time digital Input30.Size = 8; SDO List.Debounce Time digital Input30.AbortIfError = FALSE; SDO List.Debounce Time digital Input30.JumpToLine = FALSE; SDO List.Debounce Time digital Input30.Line = 0; SDO List.Debounce Time digital Input31.Index = 16#5003; SDO List.Debounce Time digital Input31.Subindex = 16#1F;
                  SDO List.Debounce Time digital Input31.Value = 40; SDO List.Debounce Time digital Input31.Size = 8; SDO List.Debounce Time digital Input31.AbortIfError = FALSE; SDO List.Debounce Time digital Input31.JumpToLine = FALSE; SDO List.Debounce Time digital Input31.Line = 0; SDO List.Debounce Time digital Input32.Index = 16#5003; SDO List.Debounce Time digital Input32.Subindex = 16#20; SDO List.Debounce Time digital Input32.Value = 40; SDO List.Debounce Time digital Input32.Size = 8; SDO List.Debounce Time digital Input32.AbortIfError = FALSE; SDO List.Debounce Time digital Input32.JumpToLine = FALSE; SDO List.Debounce Time digital Input32.Line = 0; SDO List.Minimum Value Axis1.Index = 16#5401; SDO List.Minimum Value Axis1.Subindex = 16#01; SDO List.Minimum Value Axis1.Value = 16#00001000; SDO List.Minimum Value Axis1.Size = 16; SDO List.Minimum Value Axis1.AbortIfError = FALSE; SDO List.Minimum Value Axis1.JumpToLine = FALSE; SDO List.Minimum Value Axis1.Line = 0; SDO List.Minimum Value Axis2.Index = 16#5401; SDO List.Minimum Value Axis2.Subindex = 16#02; SDO List.Minimum Value Axis2.Value = 16#00001000; SDO List.Minimum Value Axis2.Size = 16; SDO List.Minimum Value Axis2.AbortIfError = FALSE; SDO List.Minimum Value Axis2.JumpToLine = FALSE; SDO List.Minimum Value Axis2.Line = 0; SDO List.Minimum Value Axis3.Index = 16#5401; SDO List.Minimum Value Axis3.Subindex = 16#03; SDO List.Minimum Value Axis3.Value = 16#00001000; SDO List.Minimum Value Axis3.Size = 16; SDO List.Minimum Value Axis3.AbortIfError = FALSE; SDO List.Minimum Value Axis3.JumpToLine = FALSE; SDO List.Minimum Value Axis3.Line = 0; SDO List.Minimum Value Axis4.Index = 16#5401; SDO List.Minimum Value Axis4.Subindex = 16#04; SDO List.Minimum Value Axis4.Value = 16#00001000; SDO List.Minimum Value Axis4.Size = 16; SDO List.Minimum Value Axis4.AbortIfError = FALSE; SDO List.Minimum Value Axis4.JumpToLine = FALSE; SDO List.Minimum Value Axis4.Line = 0;
                  SDO List.Polarity Input 8 bit Byte_0.Index = 16#6002; SDO List.Polarity Input 8 bit Byte_0.Subindex = 16#01; SDO List.Polarity Input 8 bit Byte_0.Value = 0; SDO List.Polarity Input 8 bit Byte_0.Size = 8; SDO List.Polarity Input 8 bit Byte_0.AbortIfError = FALSE; SDO List.Polarity Input 8 bit Byte_0.JumpToLine = FALSE; SDO List.Polarity Input 8 bit Byte_0.Line = 0; SDO List.Polarity Input 8 bit Byte_1.Index = 16#6002; SDO List.Polarity Input 8 bit Byte_1.Subindex = 16#02; SDO List.Polarity Input 8 bit Byte_1.Value = 0; SDO List.Polarity Input 8 bit Byte_1.Size = 8; SDO List.Polarity Input 8 bit Byte_1.AbortIfError = FALSE; SDO List.Polarity Input 8 bit Byte_1.JumpToLine = FALSE; SDO List.Polarity Input 8 bit Byte_1.Line = 0; SDO List.Polarity Input 8 bit Byte_2.Index = 16#6002; SDO List.Polarity Input 8 bit Byte_2.Subindex = 16#03; SDO List.Polarity Input 8 bit Byte_2.Value = 0; SDO List.Polarity Input 8 bit Byte_2.Size = 8; SDO List.Polarity Input 8 bit Byte_2.AbortIfError = FALSE; SDO List.Polarity Input 8 bit Byte_2.JumpToLine = FALSE; SDO List.Polarity Input 8 bit Byte_2.Line = 0; SDO List.Irq Mask Any Change Byte_1.Index = 16#6006; SDO List.Irq Mask Any Change Byte_1.Subindex = 16#01; SDO List.Irq Mask Any Change Byte_1.Value = 16#FF; SDO List.Irq Mask Any Change Byte_1.Size = 8; SDO List.Irq Mask Any Change Byte_1.AbortIfError = FALSE; SDO List.Irq Mask Any Change Byte_1.JumpToLine = FALSE; SDO List.Irq Mask Any Change Byte_1.Line = 0; SDO List.Irq Mask Any Change Byte_2.Index = 16#6006; SDO List.Irq Mask Any Change Byte_2.Subindex = 16#02; SDO List.Irq Mask Any Change Byte_2.Value = 16#FF; SDO List.Irq Mask Any Change Byte_2.Size = 8; SDO List.Irq Mask Any Change Byte_2.AbortIfError = FALSE; SDO List.Irq Mask Any Change Byte_2.JumpToLine = FALSE; SDO List.Irq Mask Any Change Byte_2.Line = 0; SDO List.Irq Mask Any Change Byte_3.Index = 16#6006; SDO List.Irq Mask Any Change Byte_3.Subindex = 16#03; SDO List.Irq Mask Any Change Byte_3.Value = 16#FF; SDO List.Irq Mask Any Change Byte_3.Size = 8; SDO List.Irq Mask Any Change Byte_3.AbortIfError = FALSE;
                  SDO List.Irq Mask Any Change Byte_3.JumpToLine = FALSE; SDO List.Irq Mask Any Change Byte_3.Line = 0; SDO List.Irq Mask Rising Edge Byte_1.Index = 16#6007; SDO List.Irq Mask Rising Edge Byte_1.Subindex = 16#01; SDO List.Irq Mask Rising Edge Byte_1.Value = 0; SDO List.Irq Mask Rising Edge Byte_1.Size = 8; SDO List.Irq Mask Rising Edge Byte_1.AbortIfError = FALSE; SDO List.Irq Mask Rising Edge Byte_1.JumpToLine = FALSE; SDO List.Irq Mask Rising Edge Byte_1.Line = 0; SDO List.Irq Mask Rising Edge Byte_2.Index = 16#6007; SDO List.Irq Mask Rising Edge Byte_2.Subindex = 16#02; SDO List.Irq Mask Rising Edge Byte_2.Value = 0; SDO List.Irq Mask Rising Edge Byte_2.Size = 8; SDO List.Irq Mask Rising Edge Byte_2.AbortIfError = FALSE; SDO List.Irq Mask Rising Edge Byte_2.JumpToLine = FALSE; SDO List.Irq Mask Rising Edge Byte_2.Line = 0; SDO List.Irq Mask Rising Edge Byte_3.Index = 16#6007; SDO List.Irq Mask Rising Edge Byte_3.Subindex = 16#03; SDO List.Irq Mask Rising Edge Byte_3.Value = 0; SDO List.Irq Mask Rising Edge Byte_3.Size = 8; SDO List.Irq Mask Rising Edge Byte_3.AbortIfError = FALSE; SDO List.Irq Mask Rising Edge Byte_3.JumpToLine = FALSE; SDO List.Irq Mask Rising Edge Byte_3.Line = 0; SDO List.Irq Mask Falling Edge Byte_1.Index = 16#6008; SDO List.Irq Mask Falling Edge Byte_1.Subindex = 16#01; SDO List.Irq Mask Falling Edge Byte_1.Value = 0; SDO List.Irq Mask Falling Edge Byte_1.Size = 8; SDO List.Irq Mask Falling Edge Byte_1.AbortIfError = FALSE; SDO List.Irq Mask Falling Edge Byte_1.JumpToLine = FALSE; SDO List.Irq Mask Falling Edge Byte_1.Line = 0; SDO List.Irq Mask Falling Edge Byte_2.Index = 16#6008; SDO List.Irq Mask Falling Edge Byte_2.Subindex = 16#02; SDO List.Irq Mask Falling Edge Byte_2.Value = 0; SDO List.Irq Mask Falling Edge Byte_2.Size = 8; SDO List.Irq Mask Falling Edge Byte_2.AbortIfError = FALSE; SDO List.Irq Mask Falling Edge Byte_2.JumpToLine = FALSE; SDO List.Irq Mask Falling Edge Byte_2.Line = 0; SDO List.Irq Mask Falling Edge Byte_3.Index = 16#6008; SDO List.Irq Mask Falling Edge Byte_3.Subindex = 16#03; SDO List.Irq Mask Falling Edge Byte_3.Value = 0;
                  SDO List.Irq Mask Falling Edge Byte_3.Size = 8; SDO List.Irq Mask Falling Edge Byte_3.AbortIfError = FALSE; SDO List.Irq Mask Falling Edge Byte_3.JumpToLine = FALSE; SDO List.Irq Mask Falling Edge Byte_3.Line = 0; SDO List.Change Polarity Output Byte_1.Index = 16#6202; SDO List.Change Polarity Output Byte_1.Subindex = 16#01; SDO List.Change Polarity Output Byte_1.Value = 0; SDO List.Change Polarity Output Byte_1.Size = 8; SDO List.Change Polarity Output Byte_1.AbortIfError = FALSE; SDO List.Change Polarity Output Byte_1.JumpToLine = FALSE; SDO List.Change Polarity Output Byte_1.Line = 0; SDO List.Error Mode Output Byte_1.Index = 16#6206; SDO List.Error Mode Output Byte_1.Subindex = 16#01; SDO List.Error Mode Output Byte_1.Value = 16#FF; SDO List.Error Mode Output Byte_1.Size = 8; SDO List.Error Mode Output Byte_1.AbortIfError = FALSE; SDO List.Error Mode Output Byte_1.JumpToLine = FALSE; SDO List.Error Mode Output Byte_1.Line = 0; SDO List.Error State Output Byte_1.Index = 16#6207; SDO List.Error State Output Byte_1.Subindex = 16#01; SDO List.Error State Output Byte_1.Value = 0; SDO List.Error State Output Byte_1.Size = 8; SDO List.Error State Output Byte_1.AbortIfError = FALSE; SDO List.Error State Output Byte_1.JumpToLine = FALSE; SDO List.Error State Output Byte_1.Line = 0; SDO List.Analog Input Trigger Selection1.Index = 16#6421; SDO List.Analog Input Trigger Selection1.Subindex = 16#01; SDO List.Analog Input Trigger Selection1.Value = 7; SDO List.Analog Input Trigger Selection1.Size = 8; SDO List.Analog Input Trigger Selection1.AbortIfError = FALSE; SDO List.Analog Input Trigger Selection1.JumpToLine = FALSE; SDO List.Analog Input Trigger Selection1.Line = 0; SDO List.Analog Input Trigger Selection2.Index = 16#6421; SDO List.Analog Input Trigger Selection2.Subindex = 16#02; SDO List.Analog Input Trigger Selection2.Value = 7; SDO List.Analog Input Trigger Selection2.Size = 8; SDO List.Analog Input Trigger Selection2.AbortIfError = FALSE; SDO List.Analog Input Trigger Selection2.JumpToLine = FALSE; SDO List.Analog Input Trigger Selection2.Line = 0; SDO List.Analog Input Trigger Selection3.Index = 16#6421;
                  SDO List.Analog Input Trigger Selection3.Subindex = 16#03; SDO List.Analog Input Trigger Selection3.Value = 7; SDO List.Analog Input Trigger Selection3.Size = 8; SDO List.Analog Input Trigger Selection3.AbortIfError = FALSE; SDO List.Analog Input Trigger Selection3.JumpToLine = FALSE; SDO List.Analog Input Trigger Selection3.Line = 0; SDO List.Analog Input Trigger Selection4.Index = 16#6421; SDO List.Analog Input Trigger Selection4.Subindex = 16#04; SDO List.Analog Input Trigger Selection4.Value = 7; SDO List.Analog Input Trigger Selection4.Size = 8; SDO List.Analog Input Trigger Selection4.AbortIfError = FALSE; SDO List.Analog Input Trigger Selection4.JumpToLine = FALSE; SDO List.Analog Input Trigger Selection4.Line = 0; SDO List.Analog Input Interrupt Upper Limit1.Index = 16#6424; SDO List.Analog Input Interrupt Upper Limit1.Subindex = 16#01; SDO List.Analog Input Interrupt Upper Limit1.Value = 16#00000000; SDO List.Analog Input Interrupt Upper Limit1.Size = 32; SDO List.Analog Input Interrupt Upper Limit1.AbortIfError = FALSE; SDO List.Analog Input Interrupt Upper Limit1.JumpToLine = FALSE; SDO List.Analog Input Interrupt Upper Limit1.Line = 0; SDO List.Analog Input Interrupt Upper Limit2.Index = 16#6424; SDO List.Analog Input Interrupt Upper Limit2.Subindex = 16#02; SDO List.Analog Input Interrupt Upper Limit2.Value = 16#00000000; SDO List.Analog Input Interrupt Upper Limit2.Size = 32; SDO List.Analog Input Interrupt Upper Limit2.AbortIfError = FALSE; SDO List.Analog Input Interrupt Upper Limit2.JumpToLine = FALSE; SDO List.Analog Input Interrupt Upper Limit2.Line = 0; SDO List.Analog Input Interrupt Upper Limit3.Index = 16#6424; SDO List.Analog Input Interrupt Upper Limit3.Subindex = 16#03; SDO List.Analog Input Interrupt Upper Limit3.Value = 16#00000000; SDO List.Analog Input Interrupt Upper Limit3.Size = 32; SDO List.Analog Input Interrupt Upper Limit3.AbortIfError = FALSE; SDO List.Analog Input Interrupt Upper Limit3.JumpToLine = FALSE; SDO List.Analog Input Interrupt Upper Limit3.Line = 0; SDO List.Analog Input Interrupt Upper Limit4.Index = 16#6424; SDO List.Analog Input Interrupt Upper Limit4.Subindex = 16#04; SDO List.Analog Input Interrupt Upper Limit4.Value = 16#00000000; SDO List.Analog Input Interrupt Upper Limit4.Size = 32; SDO List.Analog Input Interrupt Upper Limit4.AbortIfError = FALSE; SDO List.Analog Input Interrupt Upper Limit4.JumpToLine = FALSE;
                  SDO List.Analog Input Interrupt Upper Limit4.Line = 0; SDO List.Analog Input Interrupt Lower Limit1.Index = 16#6425; SDO List.Analog Input Interrupt Lower Limit1.Subindex = 16#01; SDO List.Analog Input Interrupt Lower Limit1.Value = 16#00000000; SDO List.Analog Input Interrupt Lower Limit1.Size = 32; SDO List.Analog Input Interrupt Lower Limit1.AbortIfError = FALSE; SDO List.Analog Input Interrupt Lower Limit1.JumpToLine = FALSE; SDO List.Analog Input Interrupt Lower Limit1.Line = 0; SDO List.Analog Input Interrupt Lower Limit2.Index = 16#6425; SDO List.Analog Input Interrupt Lower Limit2.Subindex = 16#02; SDO List.Analog Input Interrupt Lower Limit2.Value = 16#00000000; SDO List.Analog Input Interrupt Lower Limit2.Size = 32; SDO List.Analog Input Interrupt Lower Limit2.AbortIfError = FALSE; SDO List.Analog Input Interrupt Lower Limit2.JumpToLine = FALSE; SDO List.Analog Input Interrupt Lower Limit2.Line = 0; SDO List.Analog Input Interrupt Lower Limit3.Index = 16#6425; SDO List.Analog Input Interrupt Lower Limit3.Subindex = 16#03; SDO List.Analog Input Interrupt Lower Limit3.Value = 16#00000000; SDO List.Analog Input Interrupt Lower Limit3.Size = 32; SDO List.Analog Input Interrupt Lower Limit3.AbortIfError = FALSE; SDO List.Analog Input Interrupt Lower Limit3.JumpToLine = FALSE; SDO List.Analog Input Interrupt Lower Limit3.Line = 0; SDO List.Analog Input Interrupt Lower Limit4.Index = 16#6425; SDO List.Analog Input Interrupt Lower Limit4.Subindex = 16#04; SDO List.Analog Input Interrupt Lower Limit4.Value = 16#00000000; SDO List.Analog Input Interrupt Lower Limit4.Size = 32; SDO List.Analog Input Interrupt Lower Limit4.AbortIfError = FALSE; SDO List.Analog Input Interrupt Lower Limit4.JumpToLine = FALSE; SDO List.Analog Input Interrupt Lower Limit4.Line = 0; SDO List.Analog Input Interrupt Delta1.Index = 16#6426; SDO List.Analog Input Interrupt Delta1.Subindex = 16#01; SDO List.Analog Input Interrupt Delta1.Value = 16#00000000; SDO List.Analog Input Interrupt Delta1.Size = 32; SDO List.Analog Input Interrupt Delta1.AbortIfError = FALSE; SDO List.Analog Input Interrupt Delta1.JumpToLine = FALSE; SDO List.Analog Input Interrupt Delta1.Line = 0; SDO List.Analog Input Interrupt Delta2.Index = 16#6426; SDO List.Analog Input Interrupt Delta2.Subindex = 16#02; SDO List.Analog Input Interrupt Delta2.Value = 16#00000000; SDO List.Analog Input Interrupt Delta2.Size = 32;
                  SDO List.Analog Input Interrupt Delta2.AbortIfError = FALSE; SDO List.Analog Input Interrupt Delta2.JumpToLine = FALSE; SDO List.Analog Input Interrupt Delta2.Line = 0; SDO List.Analog Input Interrupt Delta3.Index = 16#6426; SDO List.Analog Input Interrupt Delta3.Subindex = 16#03; SDO List.Analog Input Interrupt Delta3.Value = 16#00000000; SDO List.Analog Input Interrupt Delta3.Size = 32; SDO List.Analog Input Interrupt Delta3.AbortIfError = FALSE; SDO List.Analog Input Interrupt Delta3.JumpToLine = FALSE; SDO List.Analog Input Interrupt Delta3.Line = 0; SDO List.Analog Input Interrupt Delta4.Index = 16#6426; SDO List.Analog Input Interrupt Delta4.Subindex = 16#04; SDO List.Analog Input Interrupt Delta4.Value = 16#00000000; SDO List.Analog Input Interrupt Delta4.Size = 32; SDO List.Analog Input Interrupt Delta4.AbortIfError = FALSE; SDO List.Analog Input Interrupt Delta4.JumpToLine = FALSE; SDO List.Analog Input Interrupt Delta4.Line = 0; SDO List.Analog Input Interrupt Negative Delta1.Index = 16#6427; SDO List.Analog Input Interrupt Negative Delta1.Subindex = 16#01; SDO List.Analog Input Interrupt Negative Delta1.Value = 16#00000000; SDO List.Analog Input Interrupt Negative Delta1.Size = 32; SDO List.Analog Input Interrupt Negative Delta1.AbortIfError = FALSE; SDO List.Analog Input Interrupt Negative Delta1.JumpToLine = FALSE; SDO List.Analog Input Interrupt Negative Delta1.Line = 0; SDO List.Analog Input Interrupt Negative Delta2.Index = 16#6427; SDO List.Analog Input Interrupt Negative Delta2.Subindex = 16#02; SDO List.Analog Input Interrupt Negative Delta2.Value = 16#00000000; SDO List.Analog Input Interrupt Negative Delta2.Size = 32; SDO List.Analog Input Interrupt Negative Delta2.AbortIfError = FALSE; SDO List.Analog Input Interrupt Negative Delta2.JumpToLine = FALSE; SDO List.Analog Input Interrupt Negative Delta2.Line = 0; SDO List.Analog Input Interrupt Negative Delta3.Index = 16#6427; SDO List.Analog Input Interrupt Negative Delta3.Subindex = 16#03; SDO List.Analog Input Interrupt Negative Delta3.Value = 16#00000000; SDO List.Analog Input Interrupt Negative Delta3.Size = 32; SDO List.Analog Input Interrupt Negative Delta3.AbortIfError = FALSE; SDO List.Analog Input Interrupt Negative Delta3.JumpToLine = FALSE; SDO List.Analog Input Interrupt Negative Delta3.Line = 0; SDO List.Analog Input Interrupt Negative Delta4.Index = 16#6427; SDO List.Analog Input Interrupt Negative Delta4.Subindex = 16#04;
                  SDO List.Analog Input Interrupt Negative Delta4.Value = 16#00000000; SDO List.Analog Input Interrupt Negative Delta4.Size = 32; SDO List.Analog Input Interrupt Negative Delta4.AbortIfError = FALSE; SDO List.Analog Input Interrupt Negative Delta4.JumpToLine = FALSE; SDO List.Analog Input Interrupt Negative Delta4.Line = 0; SDO List.Analog Input Interrupt Positive Delta1.Index = 16#6428; SDO List.Analog Input Interrupt Positive Delta1.Subindex = 16#01; SDO List.Analog Input Interrupt Positive Delta1.Value = 16#00000000; SDO List.Analog Input Interrupt Positive Delta1.Size = 32; SDO List.Analog Input Interrupt Positive Delta1.AbortIfError = FALSE; SDO List.Analog Input Interrupt Positive Delta1.JumpToLine = FALSE; SDO List.Analog Input Interrupt Positive Delta1.Line = 0; SDO List.Analog Input Interrupt Positive Delta2.Index = 16#6428; SDO List.Analog Input Interrupt Positive Delta2.Subindex = 16#02; SDO List.Analog Input Interrupt Positive Delta2.Value = 16#00000000; SDO List.Analog Input Interrupt Positive Delta2.Size = 32; SDO List.Analog Input Interrupt Positive Delta2.AbortIfError = FALSE; SDO List.Analog Input Interrupt Positive Delta2.JumpToLine = FALSE; SDO List.Analog Input Interrupt Positive Delta2.Line = 0; SDO List.Analog Input Interrupt Positive Delta3.Index = 16#6428; SDO List.Analog Input Interrupt Positive Delta3.Subindex = 16#03; SDO List.Analog Input Interrupt Positive Delta3.Value = 16#00000000; SDO List.Analog Input Interrupt Positive Delta3.Size = 32; SDO List.Analog Input Interrupt Positive Delta3.AbortIfError = FALSE; SDO List.Analog Input Interrupt Positive Delta3.JumpToLine = FALSE; SDO List.Analog Input Interrupt Positive Delta3.Line = 0; SDO List.Analog Input Interrupt Positive Delta4.Index = 16#6428; SDO List.Analog Input Interrupt Positive Delta4.Subindex = 16#04; SDO List.Analog Input Interrupt Positive Delta4.Value = 16#00000000; SDO List.Analog Input Interrupt Positive Delta4.Size = 32; SDO List.Analog Input Interrupt Positive Delta4.AbortIfError = FALSE; SDO List.Analog Input Interrupt Positive Delta4.JumpToLine = FALSE; SDO List.Analog Input Interrupt Positive Delta4.Line = 0; SDO List.Analog Input Offset1.Index = 16#6431; SDO List.Analog Input Offset1.Subindex = 16#01; SDO List.Analog Input Offset1.Value = 16#00000000; SDO List.Analog Input Offset1.Size = 32; SDO List.Analog Input Offset1.AbortIfError = FALSE; SDO List.Analog Input Offset1.JumpToLine = FALSE; SDO List.Analog Input Offset1.Line = 0;
                  SDO List.Analog Input Offset2.Index = 16#6431; SDO List.Analog Input Offset2.Subindex = 16#02; SDO List.Analog Input Offset2.Value = 16#00000000; SDO List.Analog Input Offset2.Size = 32; SDO List.Analog Input Offset2.AbortIfError = FALSE; SDO List.Analog Input Offset2.JumpToLine = FALSE; SDO List.Analog Input Offset2.Line = 0; SDO List.Analog Input Offset3.Index = 16#6431; SDO List.Analog Input Offset3.Subindex = 16#03; SDO List.Analog Input Offset3.Value = 16#00000000; SDO List.Analog Input Offset3.Size = 32; SDO List.Analog Input Offset3.AbortIfError = FALSE; SDO List.Analog Input Offset3.JumpToLine = FALSE; SDO List.Analog Input Offset3.Line = 0; SDO List.Analog Input Offset4.Index = 16#6431; SDO List.Analog Input Offset4.Subindex = 16#04; SDO List.Analog Input Offset4.Value = 16#00000000; SDO List.Analog Input Offset4.Size = 32; SDO List.Analog Input Offset4.AbortIfError = FALSE; SDO List.Analog Input Offset4.JumpToLine = FALSE; SDO List.Analog Input Offset4.Line = 0; ConfigVersion = 50659584
                input  Application.JOYSTICK_INPUT_MAPPING.xRawSwitch1 : BOOL  // DigInput8_2.Bit0
                input  Application.JOYSTICK_INPUT_MAPPING.xRawSwitch2 : BOOL  // DigInput8_2.Bit1
                input  Application.JOYSTICK_INPUT_MAPPING.xRawSwitch3 : BOOL  // DigInput8_2.Bit2
                input  Application.JOYSTICK_INPUT_MAPPING.xRawSwitch4 : BOOL  // DigInput8_2.Bit3
                input  Application.JOYSTICK_INPUT_MAPPING.xRawPersonPresent : BOOL  // DigInput8_2.Bit7
                input  Application.JOYSTICK_INPUT_MAPPING.iRawAxisX : INT  // Joystick X Axis
                input  Application.JOYSTICK_INPUT_MAPPING.iRawAxisY : INT  // Joystick Y Axis
                input  Application.JOYSTICK_INPUT_MAPPING.iRawAxisZ : INT  // Joystick Z Axis
                unmapped channels: Write Output Byte_1, DigInput8_0, DigInput8_1, DigInput8_2
            System_R360_I_O_CompactModule_CR2052_V020014 : System R360: I/O CompactModule CR2052_V020013, ifm electronic gmbh, order no. CR2052, version Revision=16#00000000, FileVersion=1.1
                settings: General Options.Create all SDOs = TRUE; General Options.Optional Device = TRUE; General Options.Reset Node = FALSE; NODEIDSAVED = 20; SDO Timeout = 1000000; PDO_Autoconfig = FALSE; EXPERTSETTINGS = True; Sync-General Parameters.Sync-COBID = 16#00000080; Sync-General Parameters.Communication Cycle Period = 16#000186A0 usec; Emergency-General Parameters.Emergency COBID = 16#00000094; Heartbeat-Producer Time = 200; PDO 16#1400.COBID = 16#00000214; PDO 16#1400.Transmission Type = 16#01; Process by CANopenManager = TRUE; PDO 16#1401.COBID = 16#00000314; PDO 16#1401.Transmission Type = 16#01; Process by CANopenManager = TRUE; PDO 16#1402.COBID = 16#00000414; PDO 16#1402.Transmission Type = 16#01; Process by CANopenManager = TRUE; PDO 16#1800.COBID = 16#00000194; PDO 16#1800.Transmission Type = 16#01; Process by CANopenManager = TRUE; PDO 16#1801.COBID = 16#00000294; PDO 16#1801.Transmission Type = 16#01; Process by CANopenManager = TRUE; PDO 16#1802.COBID = 16#00000394; PDO 16#1802.Transmission Type = 16#01; Process by CANopenManager = TRUE; PDO 16#1803.COBID = 16#00000494; PDO 16#1803.Transmission Type = 16#01; Process by CANopenManager = TRUE; PDO 16#1804.COBID = 16#00000195; PDO 16#1804.Transmission Type = 16#01; Process by CANopenManager = TRUE; PDO 16#1805.COBID = 16#00000295; PDO 16#1805.Transmission Type = 16#01; Process by CANopenManager = TRUE; PDO 16#1806.COBID = 16#00000395; PDO 16#1806.Transmission Type = 16#01;
                  Process by CANopenManager = TRUE; PDO 16#1807.COBID = 16#00000495; PDO 16#1807.Transmission Type = 16#01; Process by CANopenManager = TRUE; PDO 16#1808.COBID = 16#00000196; PDO 16#1808.Transmission Type = 16#01; Process by CANopenManager = TRUE; PDO 16#1809.COBID = 16#00000296; PDO 16#1809.Transmission Type = 16#01; Process by CANopenManager = TRUE; PDO 16#180a.COBID = 16#00000396; PDO 16#180a.Transmission Type = 16#01; Process by CANopenManager = TRUE; Heartbeat-Consuming1.Heartbeat-Time = 300 ms; Binary Outputs OUT 0 - OUT 7.Subindex = 16#01; Analog Output OUT 0.Subindex = 16#01; Analog Output OUT 1.Subindex = 16#02; Analog Output OUT 2.Subindex = 16#03; Analog Output OUT 3.Subindex = 16#04; Analog Output OUT 4.Subindex = 16#05; Analog Output OUT 5.Subindex = 16#06; Analog Output OUT 6.Subindex = 16#07; Analog Output OUT 7.Subindex = 16#08; Binary Inputs IN 0 - IN 7.Subindex = 16#01; BrakeShort Inputs IN 0 - IN 7.Subindex = 16#01; BrakeLoss Inputs IN 0 - IN 7.Subindex = 16#01; OverCurrent Inputs IN 0/IN 1/IN 4/IN 5.Subindex = 16#01; BrakeShort Outputs OUT 0 - OUT 7.Subindex = 16#01; BrakeLoss Outputs OUT 0 - OUT 7.Subindex = 16#01; Overload Outputs OUT 0 - OUT 7.Subindex = 16#01; Analog Input IN 0.Subindex = 16#01; Analog Input IN 1.Subindex = 16#02; Analog Input IN 4.Subindex = 16#03; Analog Input IN 5.Subindex = 16#04; Resistance Input IN 2.Subindex = 16#01; Resistance Input IN 3.Subindex = 16#02; Resistance Input IN 6.Subindex = 16#03; Resistance Input IN 7.Subindex = 16#04; Period Inputs IN 0.Subindex = 16#01; Period Inputs IN 1.Subindex = 16#02;
                  Period Inputs IN 4.Subindex = 16#03; Period Inputs IN 5.Subindex = 16#04; Ratio IN 0.Subindex = 16#01; Ratio IN 1.Subindex = 16#02; Ratio IN 4.Subindex = 16#03; Ratio IN 5.Subindex = 16#04; Frequency IN 0.Subindex = 16#01; Frequency IN 1.Subindex = 16#02; Frequency IN 4.Subindex = 16#03; Frequency IN 5.Subindex = 16#04; Current value OUT 0.Subindex = 16#01; Current value OUT 1.Subindex = 16#02; Current value OUT 2.Subindex = 16#03; Current value OUT 3.Subindex = 16#04; Current value OUT 4.Subindex = 16#05; Current value OUT 5.Subindex = 16#06; Current value OUT 6.Subindex = 16#07; Current value OUT 7.Subindex = 16#08; VBBS System voltage.Subindex = 16#01; VBB2 Supply voltage.Subindex = 16#01; Temperature.Subindex = 16#00; SDO List.Set COB-ID sync.Index = 16#1005; SDO List.Set COB-ID sync.Subindex = 16#00; SDO List.Set COB-ID sync.Value = 16#00000080; SDO List.Set COB-ID sync.Size = 32; SDO List.Set COB-ID sync.AbortIfError = FALSE; SDO List.Set COB-ID sync.JumpToLine = FALSE; SDO List.Set COB-ID sync.Line = 0; SDO List.Set communication cycle period.Index = 16#1006; SDO List.Set communication cycle period.Subindex = 16#00; SDO List.Set communication cycle period.Value = 16#000186A0; SDO List.Set communication cycle period.Size = 32; SDO List.Set communication cycle period.AbortIfError = FALSE; SDO List.Set communication cycle period.JumpToLine = FALSE; SDO List.Set communication cycle period.Line = 0; SDO List.Disable Emcy CobID.Index = 16#1014; SDO List.Disable Emcy CobID.Subindex = 16#00; SDO List.Disable Emcy CobID.Value = 16#80000094; SDO List.Disable Emcy CobID.Size = 32; SDO List.Disable Emcy CobID.AbortIfError = FALSE;
                  SDO List.Disable Emcy CobID.JumpToLine = FALSE; SDO List.Disable Emcy CobID.Line = 0; SDO List.Set Emcy CobID.Index = 16#1014; SDO List.Set Emcy CobID.Subindex = 16#00; SDO List.Set Emcy CobID.Value = 16#00000094; SDO List.Set Emcy CobID.Size = 32; SDO List.Set Emcy CobID.AbortIfError = FALSE; SDO List.Set Emcy CobID.JumpToLine = FALSE; SDO List.Set Emcy CobID.Line = 0; SDO List.Set Heartbeat Consumer.Index = 16#1016; SDO List.Set Heartbeat Consumer.Subindex = 16#01; SDO List.Set Heartbeat Consumer.Value = 16#0001012C; SDO List.Set Heartbeat Consumer.Size = 32; SDO List.Set Heartbeat Consumer.AbortIfError = FALSE; SDO List.Set Heartbeat Consumer.JumpToLine = FALSE; SDO List.Set Heartbeat Consumer.Line = 0; SDO List.Set Heartbeat Producer.Index = 16#1017; SDO List.Set Heartbeat Producer.Subindex = 16#00; SDO List.Set Heartbeat Producer.Value = 16#000000C8; SDO List.Set Heartbeat Producer.Size = 16; SDO List.Set Heartbeat Producer.AbortIfError = FALSE; SDO List.Set Heartbeat Producer.JumpToLine = FALSE; SDO List.Set Heartbeat Producer.Line = 0; SDO List.Disable PDO.Index = 16#1400; SDO List.Disable PDO.Subindex = 16#01; SDO List.Disable PDO.Value = 16#80000214; SDO List.Disable PDO.Size = 32; SDO List.Disable PDO.AbortIfError = FALSE; SDO List.Disable PDO.JumpToLine = FALSE; SDO List.Disable PDO.Line = 0; SDO List.Set transmission type.Index = 16#1400; SDO List.Set transmission type.Subindex = 16#02; SDO List.Set transmission type.Value = 16#01; SDO List.Set transmission type.Size = 8; SDO List.Set transmission type.AbortIfError = FALSE; SDO List.Set transmission type.JumpToLine = FALSE; SDO List.Set transmission type.Line = 0; SDO List.Set and enable COB-ID.Index = 16#1400; SDO List.Set and enable COB-ID.Subindex = 16#01; SDO List.Set and enable COB-ID.Value = 16#00000214;
                  SDO List.Set and enable COB-ID.Size = 32; SDO List.Set and enable COB-ID.AbortIfError = FALSE; SDO List.Set and enable COB-ID.JumpToLine = FALSE; SDO List.Set and enable COB-ID.Line = 0; SDO List.Disable PDO.Index = 16#1401; SDO List.Disable PDO.Subindex = 16#01; SDO List.Disable PDO.Value = 16#80000314; SDO List.Disable PDO.Size = 32; SDO List.Disable PDO.AbortIfError = FALSE; SDO List.Disable PDO.JumpToLine = FALSE; SDO List.Disable PDO.Line = 0; SDO List.Set transmission type.Index = 16#1401; SDO List.Set transmission type.Subindex = 16#02; SDO List.Set transmission type.Value = 16#01; SDO List.Set transmission type.Size = 8; SDO List.Set transmission type.AbortIfError = FALSE; SDO List.Set transmission type.JumpToLine = FALSE; SDO List.Set transmission type.Line = 0; SDO List.Set and enable COB-ID.Index = 16#1401; SDO List.Set and enable COB-ID.Subindex = 16#01; SDO List.Set and enable COB-ID.Value = 16#00000314; SDO List.Set and enable COB-ID.Size = 32; SDO List.Set and enable COB-ID.AbortIfError = FALSE; SDO List.Set and enable COB-ID.JumpToLine = FALSE; SDO List.Set and enable COB-ID.Line = 0; SDO List.Disable PDO.Index = 16#1402; SDO List.Disable PDO.Subindex = 16#01; SDO List.Disable PDO.Value = 16#80000414; SDO List.Disable PDO.Size = 32; SDO List.Disable PDO.AbortIfError = FALSE; SDO List.Disable PDO.JumpToLine = FALSE; SDO List.Disable PDO.Line = 0; SDO List.Set transmission type.Index = 16#1402; SDO List.Set transmission type.Subindex = 16#02; SDO List.Set transmission type.Value = 16#01; SDO List.Set transmission type.Size = 8; SDO List.Set transmission type.AbortIfError = FALSE; SDO List.Set transmission type.JumpToLine = FALSE; SDO List.Set transmission type.Line = 0; SDO List.Set and enable COB-ID.Index = 16#1402;
                  SDO List.Set and enable COB-ID.Subindex = 16#01; SDO List.Set and enable COB-ID.Value = 16#00000414; SDO List.Set and enable COB-ID.Size = 32; SDO List.Set and enable COB-ID.AbortIfError = FALSE; SDO List.Set and enable COB-ID.JumpToLine = FALSE; SDO List.Set and enable COB-ID.Line = 0; SDO List.Disable PDO.Index = 16#1800; SDO List.Disable PDO.Subindex = 16#01; SDO List.Disable PDO.Value = 16#80000194; SDO List.Disable PDO.Size = 32; SDO List.Disable PDO.AbortIfError = FALSE; SDO List.Disable PDO.JumpToLine = FALSE; SDO List.Disable PDO.Line = 0; SDO List.Set transmission type.Index = 16#1800; SDO List.Set transmission type.Subindex = 16#02; SDO List.Set transmission type.Value = 16#01; SDO List.Set transmission type.Size = 8; SDO List.Set transmission type.AbortIfError = FALSE; SDO List.Set transmission type.JumpToLine = FALSE; SDO List.Set transmission type.Line = 0; SDO List.Set inhibit time.Index = 16#1800; SDO List.Set inhibit time.Subindex = 16#03; SDO List.Set inhibit time.Value = 16#0000; SDO List.Set inhibit time.Size = 16; SDO List.Set inhibit time.AbortIfError = FALSE; SDO List.Set inhibit time.JumpToLine = FALSE; SDO List.Set inhibit time.Line = 0; SDO List.Set event time.Index = 16#1800; SDO List.Set event time.Subindex = 16#05; SDO List.Set event time.Value = 16#0000; SDO List.Set event time.Size = 16; SDO List.Set event time.AbortIfError = FALSE; SDO List.Set event time.JumpToLine = FALSE; SDO List.Set event time.Line = 0; SDO List.Set and enable COB-ID.Index = 16#1800; SDO List.Set and enable COB-ID.Subindex = 16#01; SDO List.Set and enable COB-ID.Value = 16#00000194; SDO List.Set and enable COB-ID.Size = 32; SDO List.Set and enable COB-ID.AbortIfError = FALSE; SDO List.Set and enable COB-ID.JumpToLine = FALSE;
                  SDO List.Set and enable COB-ID.Line = 0; SDO List.Disable PDO.Index = 16#1801; SDO List.Disable PDO.Subindex = 16#01; SDO List.Disable PDO.Value = 16#80000294; SDO List.Disable PDO.Size = 32; SDO List.Disable PDO.AbortIfError = FALSE; SDO List.Disable PDO.JumpToLine = FALSE; SDO List.Disable PDO.Line = 0; SDO List.Set transmission type.Index = 16#1801; SDO List.Set transmission type.Subindex = 16#02; SDO List.Set transmission type.Value = 16#01; SDO List.Set transmission type.Size = 8; SDO List.Set transmission type.AbortIfError = FALSE; SDO List.Set transmission type.JumpToLine = FALSE; SDO List.Set transmission type.Line = 0; SDO List.Set inhibit time.Index = 16#1801; SDO List.Set inhibit time.Subindex = 16#03; SDO List.Set inhibit time.Value = 16#0000; SDO List.Set inhibit time.Size = 16; SDO List.Set inhibit time.AbortIfError = FALSE; SDO List.Set inhibit time.JumpToLine = FALSE; SDO List.Set inhibit time.Line = 0; SDO List.Set event time.Index = 16#1801; SDO List.Set event time.Subindex = 16#05; SDO List.Set event time.Value = 16#0000; SDO List.Set event time.Size = 16; SDO List.Set event time.AbortIfError = FALSE; SDO List.Set event time.JumpToLine = FALSE; SDO List.Set event time.Line = 0; SDO List.Set and enable COB-ID.Index = 16#1801; SDO List.Set and enable COB-ID.Subindex = 16#01; SDO List.Set and enable COB-ID.Value = 16#00000294; SDO List.Set and enable COB-ID.Size = 32; SDO List.Set and enable COB-ID.AbortIfError = FALSE; SDO List.Set and enable COB-ID.JumpToLine = FALSE; SDO List.Set and enable COB-ID.Line = 0; SDO List.Disable PDO.Index = 16#1802; SDO List.Disable PDO.Subindex = 16#01; SDO List.Disable PDO.Value = 16#80000394; SDO List.Disable PDO.Size = 32;
                  SDO List.Disable PDO.AbortIfError = FALSE; SDO List.Disable PDO.JumpToLine = FALSE; SDO List.Disable PDO.Line = 0; SDO List.Set transmission type.Index = 16#1802; SDO List.Set transmission type.Subindex = 16#02; SDO List.Set transmission type.Value = 16#01; SDO List.Set transmission type.Size = 8; SDO List.Set transmission type.AbortIfError = FALSE; SDO List.Set transmission type.JumpToLine = FALSE; SDO List.Set transmission type.Line = 0; SDO List.Set inhibit time.Index = 16#1802; SDO List.Set inhibit time.Subindex = 16#03; SDO List.Set inhibit time.Value = 16#0000; SDO List.Set inhibit time.Size = 16; SDO List.Set inhibit time.AbortIfError = FALSE; SDO List.Set inhibit time.JumpToLine = FALSE; SDO List.Set inhibit time.Line = 0; SDO List.Set event time.Index = 16#1802; SDO List.Set event time.Subindex = 16#05; SDO List.Set event time.Value = 16#0000; SDO List.Set event time.Size = 16; SDO List.Set event time.AbortIfError = FALSE; SDO List.Set event time.JumpToLine = FALSE; SDO List.Set event time.Line = 0; SDO List.Set and enable COB-ID.Index = 16#1802; SDO List.Set and enable COB-ID.Subindex = 16#01; SDO List.Set and enable COB-ID.Value = 16#00000394; SDO List.Set and enable COB-ID.Size = 32; SDO List.Set and enable COB-ID.AbortIfError = FALSE; SDO List.Set and enable COB-ID.JumpToLine = FALSE; SDO List.Set and enable COB-ID.Line = 0; SDO List.Disable PDO.Index = 16#1803; SDO List.Disable PDO.Subindex = 16#01; SDO List.Disable PDO.Value = 16#80000494; SDO List.Disable PDO.Size = 32; SDO List.Disable PDO.AbortIfError = FALSE; SDO List.Disable PDO.JumpToLine = FALSE; SDO List.Disable PDO.Line = 0; SDO List.Set transmission type.Index = 16#1803; SDO List.Set transmission type.Subindex = 16#02;
                  SDO List.Set transmission type.Value = 16#01; SDO List.Set transmission type.Size = 8; SDO List.Set transmission type.AbortIfError = FALSE; SDO List.Set transmission type.JumpToLine = FALSE; SDO List.Set transmission type.Line = 0; SDO List.Set inhibit time.Index = 16#1803; SDO List.Set inhibit time.Subindex = 16#03; SDO List.Set inhibit time.Value = 16#0000; SDO List.Set inhibit time.Size = 16; SDO List.Set inhibit time.AbortIfError = FALSE; SDO List.Set inhibit time.JumpToLine = FALSE; SDO List.Set inhibit time.Line = 0; SDO List.Set event time.Index = 16#1803; SDO List.Set event time.Subindex = 16#05; SDO List.Set event time.Value = 16#0000; SDO List.Set event time.Size = 16; SDO List.Set event time.AbortIfError = FALSE; SDO List.Set event time.JumpToLine = FALSE; SDO List.Set event time.Line = 0; SDO List.Set and enable COB-ID.Index = 16#1803; SDO List.Set and enable COB-ID.Subindex = 16#01; SDO List.Set and enable COB-ID.Value = 16#00000494; SDO List.Set and enable COB-ID.Size = 32; SDO List.Set and enable COB-ID.AbortIfError = FALSE; SDO List.Set and enable COB-ID.JumpToLine = FALSE; SDO List.Set and enable COB-ID.Line = 0; SDO List.Disable PDO.Index = 16#1804; SDO List.Disable PDO.Subindex = 16#01; SDO List.Disable PDO.Value = 16#80000195; SDO List.Disable PDO.Size = 32; SDO List.Disable PDO.AbortIfError = FALSE; SDO List.Disable PDO.JumpToLine = FALSE; SDO List.Disable PDO.Line = 0; SDO List.Set transmission type.Index = 16#1804; SDO List.Set transmission type.Subindex = 16#02; SDO List.Set transmission type.Value = 16#01; SDO List.Set transmission type.Size = 8; SDO List.Set transmission type.AbortIfError = FALSE; SDO List.Set transmission type.JumpToLine = FALSE; SDO List.Set transmission type.Line = 0;
                  SDO List.Set inhibit time.Index = 16#1804; SDO List.Set inhibit time.Subindex = 16#03; SDO List.Set inhibit time.Value = 16#0000; SDO List.Set inhibit time.Size = 16; SDO List.Set inhibit time.AbortIfError = FALSE; SDO List.Set inhibit time.JumpToLine = FALSE; SDO List.Set inhibit time.Line = 0; SDO List.Set event time.Index = 16#1804; SDO List.Set event time.Subindex = 16#05; SDO List.Set event time.Value = 16#0000; SDO List.Set event time.Size = 16; SDO List.Set event time.AbortIfError = FALSE; SDO List.Set event time.JumpToLine = FALSE; SDO List.Set event time.Line = 0; SDO List.Set and enable COB-ID.Index = 16#1804; SDO List.Set and enable COB-ID.Subindex = 16#01; SDO List.Set and enable COB-ID.Value = 16#00000195; SDO List.Set and enable COB-ID.Size = 32; SDO List.Set and enable COB-ID.AbortIfError = FALSE; SDO List.Set and enable COB-ID.JumpToLine = FALSE; SDO List.Set and enable COB-ID.Line = 0; SDO List.Disable PDO.Index = 16#1805; SDO List.Disable PDO.Subindex = 16#01; SDO List.Disable PDO.Value = 16#80000295; SDO List.Disable PDO.Size = 32; SDO List.Disable PDO.AbortIfError = FALSE; SDO List.Disable PDO.JumpToLine = FALSE; SDO List.Disable PDO.Line = 0; SDO List.Set transmission type.Index = 16#1805; SDO List.Set transmission type.Subindex = 16#02; SDO List.Set transmission type.Value = 16#01; SDO List.Set transmission type.Size = 8; SDO List.Set transmission type.AbortIfError = FALSE; SDO List.Set transmission type.JumpToLine = FALSE; SDO List.Set transmission type.Line = 0; SDO List.Set inhibit time.Index = 16#1805; SDO List.Set inhibit time.Subindex = 16#03; SDO List.Set inhibit time.Value = 16#0000; SDO List.Set inhibit time.Size = 16; SDO List.Set inhibit time.AbortIfError = FALSE;
                  SDO List.Set inhibit time.JumpToLine = FALSE; SDO List.Set inhibit time.Line = 0; SDO List.Set event time.Index = 16#1805; SDO List.Set event time.Subindex = 16#05; SDO List.Set event time.Value = 16#0000; SDO List.Set event time.Size = 16; SDO List.Set event time.AbortIfError = FALSE; SDO List.Set event time.JumpToLine = FALSE; SDO List.Set event time.Line = 0; SDO List.Set and enable COB-ID.Index = 16#1805; SDO List.Set and enable COB-ID.Subindex = 16#01; SDO List.Set and enable COB-ID.Value = 16#00000295; SDO List.Set and enable COB-ID.Size = 32; SDO List.Set and enable COB-ID.AbortIfError = FALSE; SDO List.Set and enable COB-ID.JumpToLine = FALSE; SDO List.Set and enable COB-ID.Line = 0; SDO List.Disable PDO.Index = 16#1806; SDO List.Disable PDO.Subindex = 16#01; SDO List.Disable PDO.Value = 16#80000395; SDO List.Disable PDO.Size = 32; SDO List.Disable PDO.AbortIfError = FALSE; SDO List.Disable PDO.JumpToLine = FALSE; SDO List.Disable PDO.Line = 0; SDO List.Set transmission type.Index = 16#1806; SDO List.Set transmission type.Subindex = 16#02; SDO List.Set transmission type.Value = 16#01; SDO List.Set transmission type.Size = 8; SDO List.Set transmission type.AbortIfError = FALSE; SDO List.Set transmission type.JumpToLine = FALSE; SDO List.Set transmission type.Line = 0; SDO List.Set inhibit time.Index = 16#1806; SDO List.Set inhibit time.Subindex = 16#03; SDO List.Set inhibit time.Value = 16#0000; SDO List.Set inhibit time.Size = 16; SDO List.Set inhibit time.AbortIfError = FALSE; SDO List.Set inhibit time.JumpToLine = FALSE; SDO List.Set inhibit time.Line = 0; SDO List.Set event time.Index = 16#1806; SDO List.Set event time.Subindex = 16#05; SDO List.Set event time.Value = 16#0000;
                  SDO List.Set event time.Size = 16; SDO List.Set event time.AbortIfError = FALSE; SDO List.Set event time.JumpToLine = FALSE; SDO List.Set event time.Line = 0; SDO List.Set and enable COB-ID.Index = 16#1806; SDO List.Set and enable COB-ID.Subindex = 16#01; SDO List.Set and enable COB-ID.Value = 16#00000395; SDO List.Set and enable COB-ID.Size = 32; SDO List.Set and enable COB-ID.AbortIfError = FALSE; SDO List.Set and enable COB-ID.JumpToLine = FALSE; SDO List.Set and enable COB-ID.Line = 0; SDO List.Disable PDO.Index = 16#1807; SDO List.Disable PDO.Subindex = 16#01; SDO List.Disable PDO.Value = 16#80000495; SDO List.Disable PDO.Size = 32; SDO List.Disable PDO.AbortIfError = FALSE; SDO List.Disable PDO.JumpToLine = FALSE; SDO List.Disable PDO.Line = 0; SDO List.Set transmission type.Index = 16#1807; SDO List.Set transmission type.Subindex = 16#02; SDO List.Set transmission type.Value = 16#01; SDO List.Set transmission type.Size = 8; SDO List.Set transmission type.AbortIfError = FALSE; SDO List.Set transmission type.JumpToLine = FALSE; SDO List.Set transmission type.Line = 0; SDO List.Set inhibit time.Index = 16#1807; SDO List.Set inhibit time.Subindex = 16#03; SDO List.Set inhibit time.Value = 16#0000; SDO List.Set inhibit time.Size = 16; SDO List.Set inhibit time.AbortIfError = FALSE; SDO List.Set inhibit time.JumpToLine = FALSE; SDO List.Set inhibit time.Line = 0; SDO List.Set event time.Index = 16#1807; SDO List.Set event time.Subindex = 16#05; SDO List.Set event time.Value = 16#0000; SDO List.Set event time.Size = 16; SDO List.Set event time.AbortIfError = FALSE; SDO List.Set event time.JumpToLine = FALSE; SDO List.Set event time.Line = 0; SDO List.Set and enable COB-ID.Index = 16#1807;
                  SDO List.Set and enable COB-ID.Subindex = 16#01; SDO List.Set and enable COB-ID.Value = 16#00000495; SDO List.Set and enable COB-ID.Size = 32; SDO List.Set and enable COB-ID.AbortIfError = FALSE; SDO List.Set and enable COB-ID.JumpToLine = FALSE; SDO List.Set and enable COB-ID.Line = 0; SDO List.Disable PDO.Index = 16#1808; SDO List.Disable PDO.Subindex = 16#01; SDO List.Disable PDO.Value = 16#80000196; SDO List.Disable PDO.Size = 32; SDO List.Disable PDO.AbortIfError = FALSE; SDO List.Disable PDO.JumpToLine = FALSE; SDO List.Disable PDO.Line = 0; SDO List.Set transmission type.Index = 16#1808; SDO List.Set transmission type.Subindex = 16#02; SDO List.Set transmission type.Value = 16#01; SDO List.Set transmission type.Size = 8; SDO List.Set transmission type.AbortIfError = FALSE; SDO List.Set transmission type.JumpToLine = FALSE; SDO List.Set transmission type.Line = 0; SDO List.Set inhibit time.Index = 16#1808; SDO List.Set inhibit time.Subindex = 16#03; SDO List.Set inhibit time.Value = 16#0000; SDO List.Set inhibit time.Size = 16; SDO List.Set inhibit time.AbortIfError = FALSE; SDO List.Set inhibit time.JumpToLine = FALSE; SDO List.Set inhibit time.Line = 0; SDO List.Set event time.Index = 16#1808; SDO List.Set event time.Subindex = 16#05; SDO List.Set event time.Value = 16#0000; SDO List.Set event time.Size = 16; SDO List.Set event time.AbortIfError = FALSE; SDO List.Set event time.JumpToLine = FALSE; SDO List.Set event time.Line = 0; SDO List.Set and enable COB-ID.Index = 16#1808; SDO List.Set and enable COB-ID.Subindex = 16#01; SDO List.Set and enable COB-ID.Value = 16#00000196; SDO List.Set and enable COB-ID.Size = 32; SDO List.Set and enable COB-ID.AbortIfError = FALSE; SDO List.Set and enable COB-ID.JumpToLine = FALSE;
                  SDO List.Set and enable COB-ID.Line = 0; SDO List.Disable PDO.Index = 16#1809; SDO List.Disable PDO.Subindex = 16#01; SDO List.Disable PDO.Value = 16#80000296; SDO List.Disable PDO.Size = 32; SDO List.Disable PDO.AbortIfError = FALSE; SDO List.Disable PDO.JumpToLine = FALSE; SDO List.Disable PDO.Line = 0; SDO List.Set transmission type.Index = 16#1809; SDO List.Set transmission type.Subindex = 16#02; SDO List.Set transmission type.Value = 16#01; SDO List.Set transmission type.Size = 8; SDO List.Set transmission type.AbortIfError = FALSE; SDO List.Set transmission type.JumpToLine = FALSE; SDO List.Set transmission type.Line = 0; SDO List.Set inhibit time.Index = 16#1809; SDO List.Set inhibit time.Subindex = 16#03; SDO List.Set inhibit time.Value = 16#0000; SDO List.Set inhibit time.Size = 16; SDO List.Set inhibit time.AbortIfError = FALSE; SDO List.Set inhibit time.JumpToLine = FALSE; SDO List.Set inhibit time.Line = 0; SDO List.Set event time.Index = 16#1809; SDO List.Set event time.Subindex = 16#05; SDO List.Set event time.Value = 16#0000; SDO List.Set event time.Size = 16; SDO List.Set event time.AbortIfError = FALSE; SDO List.Set event time.JumpToLine = FALSE; SDO List.Set event time.Line = 0; SDO List.Set and enable COB-ID.Index = 16#1809; SDO List.Set and enable COB-ID.Subindex = 16#01; SDO List.Set and enable COB-ID.Value = 16#00000296; SDO List.Set and enable COB-ID.Size = 32; SDO List.Set and enable COB-ID.AbortIfError = FALSE; SDO List.Set and enable COB-ID.JumpToLine = FALSE; SDO List.Set and enable COB-ID.Line = 0; SDO List.Disable PDO.Index = 16#180A; SDO List.Disable PDO.Subindex = 16#01; SDO List.Disable PDO.Value = 16#80000396; SDO List.Disable PDO.Size = 32;
                  SDO List.Disable PDO.AbortIfError = FALSE; SDO List.Disable PDO.JumpToLine = FALSE; SDO List.Disable PDO.Line = 0; SDO List.Set transmission type.Index = 16#180A; SDO List.Set transmission type.Subindex = 16#02; SDO List.Set transmission type.Value = 16#01; SDO List.Set transmission type.Size = 8; SDO List.Set transmission type.AbortIfError = FALSE; SDO List.Set transmission type.JumpToLine = FALSE; SDO List.Set transmission type.Line = 0; SDO List.Set inhibit time.Index = 16#180A; SDO List.Set inhibit time.Subindex = 16#03; SDO List.Set inhibit time.Value = 16#0000; SDO List.Set inhibit time.Size = 16; SDO List.Set inhibit time.AbortIfError = FALSE; SDO List.Set inhibit time.JumpToLine = FALSE; SDO List.Set inhibit time.Line = 0; SDO List.Set event time.Index = 16#180A; SDO List.Set event time.Subindex = 16#05; SDO List.Set event time.Value = 16#0000; SDO List.Set event time.Size = 16; SDO List.Set event time.AbortIfError = FALSE; SDO List.Set event time.JumpToLine = FALSE; SDO List.Set event time.Line = 0; SDO List.Set and enable COB-ID.Index = 16#180A; SDO List.Set and enable COB-ID.Subindex = 16#01; SDO List.Set and enable COB-ID.Value = 16#00000396; SDO List.Set and enable COB-ID.Size = 32; SDO List.Set and enable COB-ID.AbortIfError = FALSE; SDO List.Set and enable COB-ID.JumpToLine = FALSE; SDO List.Set and enable COB-ID.Line = 0; SDO List.IO Configuration IN 00.Index = 16#2000; SDO List.IO Configuration IN 00.Subindex = 16#01; SDO List.IO Configuration IN 00.Value = 6; SDO List.IO Configuration IN 00.Size = 8; SDO List.IO Configuration IN 00.AbortIfError = FALSE; SDO List.IO Configuration IN 00.JumpToLine = FALSE; SDO List.IO Configuration IN 00.Line = 0; SDO List.IO Configuration IN 01.Index = 16#2000; SDO List.IO Configuration IN 01.Subindex = 16#02;
                  SDO List.IO Configuration IN 01.Value = 6; SDO List.IO Configuration IN 01.Size = 8; SDO List.IO Configuration IN 01.AbortIfError = FALSE; SDO List.IO Configuration IN 01.JumpToLine = FALSE; SDO List.IO Configuration IN 01.Line = 0; SDO List.IO Configuration IN 02.Index = 16#2000; SDO List.IO Configuration IN 02.Subindex = 16#03; SDO List.IO Configuration IN 02.Value = 10; SDO List.IO Configuration IN 02.Size = 8; SDO List.IO Configuration IN 02.AbortIfError = FALSE; SDO List.IO Configuration IN 02.JumpToLine = FALSE; SDO List.IO Configuration IN 02.Line = 0; SDO List.IO Configuration IN 03.Index = 16#2000; SDO List.IO Configuration IN 03.Subindex = 16#04; SDO List.IO Configuration IN 03.Value = 10; SDO List.IO Configuration IN 03.Size = 8; SDO List.IO Configuration IN 03.AbortIfError = FALSE; SDO List.IO Configuration IN 03.JumpToLine = FALSE; SDO List.IO Configuration IN 03.Line = 0; SDO List.IO Configuration IN 04.Index = 16#2000; SDO List.IO Configuration IN 04.Subindex = 16#05; SDO List.IO Configuration IN 04.Value = 10; SDO List.IO Configuration IN 04.Size = 8; SDO List.IO Configuration IN 04.AbortIfError = FALSE; SDO List.IO Configuration IN 04.JumpToLine = FALSE; SDO List.IO Configuration IN 04.Line = 0; SDO List.IO Configuration IN 05.Index = 16#2000; SDO List.IO Configuration IN 05.Subindex = 16#06; SDO List.IO Configuration IN 05.Value = 10; SDO List.IO Configuration IN 05.Size = 8; SDO List.IO Configuration IN 05.AbortIfError = FALSE; SDO List.IO Configuration IN 05.JumpToLine = FALSE; SDO List.IO Configuration IN 05.Line = 0; SDO List.IO Configuration IN 06.Index = 16#2000; SDO List.IO Configuration IN 06.Subindex = 16#07; SDO List.IO Configuration IN 06.Value = 10; SDO List.IO Configuration IN 06.Size = 8; SDO List.IO Configuration IN 06.AbortIfError = FALSE; SDO List.IO Configuration IN 06.JumpToLine = FALSE; SDO List.IO Configuration IN 06.Line = 0;
                  SDO List.IO Configuration IN 07.Index = 16#2000; SDO List.IO Configuration IN 07.Subindex = 16#08; SDO List.IO Configuration IN 07.Value = 10; SDO List.IO Configuration IN 07.Size = 8; SDO List.IO Configuration IN 07.AbortIfError = FALSE; SDO List.IO Configuration IN 07.JumpToLine = FALSE; SDO List.IO Configuration IN 07.Line = 0; SDO List.IO Configuration OUT 00.Index = 16#2000; SDO List.IO Configuration OUT 00.Subindex = 16#09; SDO List.IO Configuration OUT 00.Value = 2; SDO List.IO Configuration OUT 00.Size = 8; SDO List.IO Configuration OUT 00.AbortIfError = FALSE; SDO List.IO Configuration OUT 00.JumpToLine = FALSE; SDO List.IO Configuration OUT 00.Line = 0; SDO List.IO Configuration OUT 01.Index = 16#2000; SDO List.IO Configuration OUT 01.Subindex = 16#0A; SDO List.IO Configuration OUT 01.Value = 2; SDO List.IO Configuration OUT 01.Size = 8; SDO List.IO Configuration OUT 01.AbortIfError = FALSE; SDO List.IO Configuration OUT 01.JumpToLine = FALSE; SDO List.IO Configuration OUT 01.Line = 0; SDO List.IO Configuration OUT 02.Index = 16#2000; SDO List.IO Configuration OUT 02.Subindex = 16#0B; SDO List.IO Configuration OUT 02.Value = 2; SDO List.IO Configuration OUT 02.Size = 8; SDO List.IO Configuration OUT 02.AbortIfError = FALSE; SDO List.IO Configuration OUT 02.JumpToLine = FALSE; SDO List.IO Configuration OUT 02.Line = 0; SDO List.IO Configuration OUT 03.Index = 16#2000; SDO List.IO Configuration OUT 03.Subindex = 16#0C; SDO List.IO Configuration OUT 03.Value = 2; SDO List.IO Configuration OUT 03.Size = 8; SDO List.IO Configuration OUT 03.AbortIfError = FALSE; SDO List.IO Configuration OUT 03.JumpToLine = FALSE; SDO List.IO Configuration OUT 03.Line = 0; SDO List.IO Configuration OUT 04.Index = 16#2000; SDO List.IO Configuration OUT 04.Subindex = 16#0D; SDO List.IO Configuration OUT 04.Value = 2; SDO List.IO Configuration OUT 04.Size = 8; SDO List.IO Configuration OUT 04.AbortIfError = FALSE;
                  SDO List.IO Configuration OUT 04.JumpToLine = FALSE; SDO List.IO Configuration OUT 04.Line = 0; SDO List.IO Configuration OUT 05.Index = 16#2000; SDO List.IO Configuration OUT 05.Subindex = 16#0E; SDO List.IO Configuration OUT 05.Value = 2; SDO List.IO Configuration OUT 05.Size = 8; SDO List.IO Configuration OUT 05.AbortIfError = FALSE; SDO List.IO Configuration OUT 05.JumpToLine = FALSE; SDO List.IO Configuration OUT 05.Line = 0; SDO List.IO Configuration OUT 06.Index = 16#2000; SDO List.IO Configuration OUT 06.Subindex = 16#0F; SDO List.IO Configuration OUT 06.Value = 2; SDO List.IO Configuration OUT 06.Size = 8; SDO List.IO Configuration OUT 06.AbortIfError = FALSE; SDO List.IO Configuration OUT 06.JumpToLine = FALSE; SDO List.IO Configuration OUT 06.Line = 0; SDO List.IO Configuration OUT 07.Index = 16#2000; SDO List.IO Configuration OUT 07.Subindex = 16#10; SDO List.IO Configuration OUT 07.Value = 2; SDO List.IO Configuration OUT 07.Size = 8; SDO List.IO Configuration OUT 07.AbortIfError = FALSE; SDO List.IO Configuration OUT 07.JumpToLine = FALSE; SDO List.IO Configuration OUT 07.Line = 0; SDO List.PWM frequency OUT 00.Index = 16#2001; SDO List.PWM frequency OUT 00.Subindex = 16#01; SDO List.PWM frequency OUT 00.Value = 100; SDO List.PWM frequency OUT 00.Size = 16; SDO List.PWM frequency OUT 00.AbortIfError = FALSE; SDO List.PWM frequency OUT 00.JumpToLine = FALSE; SDO List.PWM frequency OUT 00.Line = 0; SDO List.PWM frequency OUT 01.Index = 16#2001; SDO List.PWM frequency OUT 01.Subindex = 16#02; SDO List.PWM frequency OUT 01.Value = 100; SDO List.PWM frequency OUT 01.Size = 16; SDO List.PWM frequency OUT 01.AbortIfError = FALSE; SDO List.PWM frequency OUT 01.JumpToLine = FALSE; SDO List.PWM frequency OUT 01.Line = 0; SDO List.PWM frequency OUT 02.Index = 16#2001; SDO List.PWM frequency OUT 02.Subindex = 16#03; SDO List.PWM frequency OUT 02.Value = 100;
                  SDO List.PWM frequency OUT 02.Size = 16; SDO List.PWM frequency OUT 02.AbortIfError = FALSE; SDO List.PWM frequency OUT 02.JumpToLine = FALSE; SDO List.PWM frequency OUT 02.Line = 0; SDO List.PWM frequency OUT 03.Index = 16#2001; SDO List.PWM frequency OUT 03.Subindex = 16#04; SDO List.PWM frequency OUT 03.Value = 100; SDO List.PWM frequency OUT 03.Size = 16; SDO List.PWM frequency OUT 03.AbortIfError = FALSE; SDO List.PWM frequency OUT 03.JumpToLine = FALSE; SDO List.PWM frequency OUT 03.Line = 0; SDO List.PWM frequency OUT 04.Index = 16#2001; SDO List.PWM frequency OUT 04.Subindex = 16#05; SDO List.PWM frequency OUT 04.Value = 100; SDO List.PWM frequency OUT 04.Size = 16; SDO List.PWM frequency OUT 04.AbortIfError = FALSE; SDO List.PWM frequency OUT 04.JumpToLine = FALSE; SDO List.PWM frequency OUT 04.Line = 0; SDO List.PWM frequency OUT 05.Index = 16#2001; SDO List.PWM frequency OUT 05.Subindex = 16#06; SDO List.PWM frequency OUT 05.Value = 100; SDO List.PWM frequency OUT 05.Size = 16; SDO List.PWM frequency OUT 05.AbortIfError = FALSE; SDO List.PWM frequency OUT 05.JumpToLine = FALSE; SDO List.PWM frequency OUT 05.Line = 0; SDO List.PWM frequency OUT 06.Index = 16#2001; SDO List.PWM frequency OUT 06.Subindex = 16#07; SDO List.PWM frequency OUT 06.Value = 100; SDO List.PWM frequency OUT 06.Size = 16; SDO List.PWM frequency OUT 06.AbortIfError = FALSE; SDO List.PWM frequency OUT 06.JumpToLine = FALSE; SDO List.PWM frequency OUT 06.Line = 0; SDO List.PWM frequency OUT 07.Index = 16#2001; SDO List.PWM frequency OUT 07.Subindex = 16#08; SDO List.PWM frequency OUT 07.Value = 100; SDO List.PWM frequency OUT 07.Size = 16; SDO List.PWM frequency OUT 07.AbortIfError = FALSE; SDO List.PWM frequency OUT 07.JumpToLine = FALSE; SDO List.PWM frequency OUT 07.Line = 0; SDO List.Current control OUT 0 KP.Index = 16#2004;
                  SDO List.Current control OUT 0 KP.Subindex = 16#01; SDO List.Current control OUT 0 KP.Value = 30; SDO List.Current control OUT 0 KP.Size = 8; SDO List.Current control OUT 0 KP.AbortIfError = FALSE; SDO List.Current control OUT 0 KP.JumpToLine = FALSE; SDO List.Current control OUT 0 KP.Line = 0; SDO List.Current control OUT 1 KP.Index = 16#2004; SDO List.Current control OUT 1 KP.Subindex = 16#02; SDO List.Current control OUT 1 KP.Value = 30; SDO List.Current control OUT 1 KP.Size = 8; SDO List.Current control OUT 1 KP.AbortIfError = FALSE; SDO List.Current control OUT 1 KP.JumpToLine = FALSE; SDO List.Current control OUT 1 KP.Line = 0; SDO List.Current control OUT 2 KP.Index = 16#2004; SDO List.Current control OUT 2 KP.Subindex = 16#03; SDO List.Current control OUT 2 KP.Value = 30; SDO List.Current control OUT 2 KP.Size = 8; SDO List.Current control OUT 2 KP.AbortIfError = FALSE; SDO List.Current control OUT 2 KP.JumpToLine = FALSE; SDO List.Current control OUT 2 KP.Line = 0; SDO List.Current control OUT 3 KP.Index = 16#2004; SDO List.Current control OUT 3 KP.Subindex = 16#04; SDO List.Current control OUT 3 KP.Value = 30; SDO List.Current control OUT 3 KP.Size = 8; SDO List.Current control OUT 3 KP.AbortIfError = FALSE; SDO List.Current control OUT 3 KP.JumpToLine = FALSE; SDO List.Current control OUT 3 KP.Line = 0; SDO List.Current control OUT 4 KP.Index = 16#2004; SDO List.Current control OUT 4 KP.Subindex = 16#05; SDO List.Current control OUT 4 KP.Value = 30; SDO List.Current control OUT 4 KP.Size = 8; SDO List.Current control OUT 4 KP.AbortIfError = FALSE; SDO List.Current control OUT 4 KP.JumpToLine = FALSE; SDO List.Current control OUT 4 KP.Line = 0; SDO List.Current control OUT 5 KP.Index = 16#2004; SDO List.Current control OUT 5 KP.Subindex = 16#06; SDO List.Current control OUT 5 KP.Value = 30; SDO List.Current control OUT 5 KP.Size = 8; SDO List.Current control OUT 5 KP.AbortIfError = FALSE; SDO List.Current control OUT 5 KP.JumpToLine = FALSE;
                  SDO List.Current control OUT 5 KP.Line = 0; SDO List.Current control OUT 6 KP.Index = 16#2004; SDO List.Current control OUT 6 KP.Subindex = 16#07; SDO List.Current control OUT 6 KP.Value = 30; SDO List.Current control OUT 6 KP.Size = 8; SDO List.Current control OUT 6 KP.AbortIfError = FALSE; SDO List.Current control OUT 6 KP.JumpToLine = FALSE; SDO List.Current control OUT 6 KP.Line = 0; SDO List.Current control OUT 7 KP.Index = 16#2004; SDO List.Current control OUT 7 KP.Subindex = 16#08; SDO List.Current control OUT 7 KP.Value = 30; SDO List.Current control OUT 7 KP.Size = 8; SDO List.Current control OUT 7 KP.AbortIfError = FALSE; SDO List.Current control OUT 7 KP.JumpToLine = FALSE; SDO List.Current control OUT 7 KP.Line = 0; SDO List.Current control OUT 0 KI.Index = 16#2005; SDO List.Current control OUT 0 KI.Subindex = 16#01; SDO List.Current control OUT 0 KI.Value = 20; SDO List.Current control OUT 0 KI.Size = 8; SDO List.Current control OUT 0 KI.AbortIfError = FALSE; SDO List.Current control OUT 0 KI.JumpToLine = FALSE; SDO List.Current control OUT 0 KI.Line = 0; SDO List.Current control OUT 1 KI.Index = 16#2005; SDO List.Current control OUT 1 KI.Subindex = 16#02; SDO List.Current control OUT 1 KI.Value = 20; SDO List.Current control OUT 1 KI.Size = 8; SDO List.Current control OUT 1 KI.AbortIfError = FALSE; SDO List.Current control OUT 1 KI.JumpToLine = FALSE; SDO List.Current control OUT 1 KI.Line = 0; SDO List.Current control OUT 2 KI.Index = 16#2005; SDO List.Current control OUT 2 KI.Subindex = 16#03; SDO List.Current control OUT 2 KI.Value = 20; SDO List.Current control OUT 2 KI.Size = 8; SDO List.Current control OUT 2 KI.AbortIfError = FALSE; SDO List.Current control OUT 2 KI.JumpToLine = FALSE; SDO List.Current control OUT 2 KI.Line = 0; SDO List.Current control OUT 3 KI.Index = 16#2005; SDO List.Current control OUT 3 KI.Subindex = 16#04; SDO List.Current control OUT 3 KI.Value = 20; SDO List.Current control OUT 3 KI.Size = 8;
                  SDO List.Current control OUT 3 KI.AbortIfError = FALSE; SDO List.Current control OUT 3 KI.JumpToLine = FALSE; SDO List.Current control OUT 3 KI.Line = 0; SDO List.Current control OUT 4 KI.Index = 16#2005; SDO List.Current control OUT 4 KI.Subindex = 16#05; SDO List.Current control OUT 4 KI.Value = 20; SDO List.Current control OUT 4 KI.Size = 8; SDO List.Current control OUT 4 KI.AbortIfError = FALSE; SDO List.Current control OUT 4 KI.JumpToLine = FALSE; SDO List.Current control OUT 4 KI.Line = 0; SDO List.Current control OUT 5 KI.Index = 16#2005; SDO List.Current control OUT 5 KI.Subindex = 16#06; SDO List.Current control OUT 5 KI.Value = 20; SDO List.Current control OUT 5 KI.Size = 8; SDO List.Current control OUT 5 KI.AbortIfError = FALSE; SDO List.Current control OUT 5 KI.JumpToLine = FALSE; SDO List.Current control OUT 5 KI.Line = 0; SDO List.Current control OUT 6 KI.Index = 16#2005; SDO List.Current control OUT 6 KI.Subindex = 16#07; SDO List.Current control OUT 6 KI.Value = 20; SDO List.Current control OUT 6 KI.Size = 8; SDO List.Current control OUT 6 KI.AbortIfError = FALSE; SDO List.Current control OUT 6 KI.JumpToLine = FALSE; SDO List.Current control OUT 6 KI.Line = 0; SDO List.Current control OUT 7 KI.Index = 16#2005; SDO List.Current control OUT 7 KI.Subindex = 16#08; SDO List.Current control OUT 7 KI.Value = 20; SDO List.Current control OUT 7 KI.Size = 8; SDO List.Current control OUT 7 KI.AbortIfError = FALSE; SDO List.Current control OUT 7 KI.JumpToLine = FALSE; SDO List.Current control OUT 7 KI.Line = 0; SDO List.Current control OUT 0 Ditherfreq.Index = 16#2006; SDO List.Current control OUT 0 Ditherfreq.Subindex = 16#01; SDO List.Current control OUT 0 Ditherfreq.Value = 0; SDO List.Current control OUT 0 Ditherfreq.Size = 16; SDO List.Current control OUT 0 Ditherfreq.AbortIfError = FALSE; SDO List.Current control OUT 0 Ditherfreq.JumpToLine = FALSE; SDO List.Current control OUT 0 Ditherfreq.Line = 0; SDO List.Current control OUT 1 Ditherfreq.Index = 16#2006; SDO List.Current control OUT 1 Ditherfreq.Subindex = 16#02;
                  SDO List.Current control OUT 1 Ditherfreq.Value = 0; SDO List.Current control OUT 1 Ditherfreq.Size = 16; SDO List.Current control OUT 1 Ditherfreq.AbortIfError = FALSE; SDO List.Current control OUT 1 Ditherfreq.JumpToLine = FALSE; SDO List.Current control OUT 1 Ditherfreq.Line = 0; SDO List.Current control OUT 2 Ditherfreq.Index = 16#2006; SDO List.Current control OUT 2 Ditherfreq.Subindex = 16#03; SDO List.Current control OUT 2 Ditherfreq.Value = 0; SDO List.Current control OUT 2 Ditherfreq.Size = 16; SDO List.Current control OUT 2 Ditherfreq.AbortIfError = FALSE; SDO List.Current control OUT 2 Ditherfreq.JumpToLine = FALSE; SDO List.Current control OUT 2 Ditherfreq.Line = 0; SDO List.Current control OUT 3 Ditherfreq.Index = 16#2006; SDO List.Current control OUT 3 Ditherfreq.Subindex = 16#04; SDO List.Current control OUT 3 Ditherfreq.Value = 0; SDO List.Current control OUT 3 Ditherfreq.Size = 16; SDO List.Current control OUT 3 Ditherfreq.AbortIfError = FALSE; SDO List.Current control OUT 3 Ditherfreq.JumpToLine = FALSE; SDO List.Current control OUT 3 Ditherfreq.Line = 0; SDO List.Current control OUT 4 Ditherfreq.Index = 16#2006; SDO List.Current control OUT 4 Ditherfreq.Subindex = 16#05; SDO List.Current control OUT 4 Ditherfreq.Value = 0; SDO List.Current control OUT 4 Ditherfreq.Size = 16; SDO List.Current control OUT 4 Ditherfreq.AbortIfError = FALSE; SDO List.Current control OUT 4 Ditherfreq.JumpToLine = FALSE; SDO List.Current control OUT 4 Ditherfreq.Line = 0; SDO List.Current control OUT 5 Ditherfreq.Index = 16#2006; SDO List.Current control OUT 5 Ditherfreq.Subindex = 16#06; SDO List.Current control OUT 5 Ditherfreq.Value = 0; SDO List.Current control OUT 5 Ditherfreq.Size = 16; SDO List.Current control OUT 5 Ditherfreq.AbortIfError = FALSE; SDO List.Current control OUT 5 Ditherfreq.JumpToLine = FALSE; SDO List.Current control OUT 5 Ditherfreq.Line = 0; SDO List.Current control OUT 6 Ditherfreq.Index = 16#2006; SDO List.Current control OUT 6 Ditherfreq.Subindex = 16#07; SDO List.Current control OUT 6 Ditherfreq.Value = 0; SDO List.Current control OUT 6 Ditherfreq.Size = 16; SDO List.Current control OUT 6 Ditherfreq.AbortIfError = FALSE; SDO List.Current control OUT 6 Ditherfreq.JumpToLine = FALSE; SDO List.Current control OUT 6 Ditherfreq.Line = 0;
                  SDO List.Current control OUT 7 Ditherfreq.Index = 16#2006; SDO List.Current control OUT 7 Ditherfreq.Subindex = 16#08; SDO List.Current control OUT 7 Ditherfreq.Value = 0; SDO List.Current control OUT 7 Ditherfreq.Size = 16; SDO List.Current control OUT 7 Ditherfreq.AbortIfError = FALSE; SDO List.Current control OUT 7 Ditherfreq.JumpToLine = FALSE; SDO List.Current control OUT 7 Ditherfreq.Line = 0; SDO List.Current control OUT 0 Dithervalue.Index = 16#2007; SDO List.Current control OUT 0 Dithervalue.Subindex = 16#01; SDO List.Current control OUT 0 Dithervalue.Value = 0; SDO List.Current control OUT 0 Dithervalue.Size = 16; SDO List.Current control OUT 0 Dithervalue.AbortIfError = FALSE; SDO List.Current control OUT 0 Dithervalue.JumpToLine = FALSE; SDO List.Current control OUT 0 Dithervalue.Line = 0; SDO List.Current control OUT 1 Dithervalue.Index = 16#2007; SDO List.Current control OUT 1 Dithervalue.Subindex = 16#02; SDO List.Current control OUT 1 Dithervalue.Value = 0; SDO List.Current control OUT 1 Dithervalue.Size = 16; SDO List.Current control OUT 1 Dithervalue.AbortIfError = FALSE; SDO List.Current control OUT 1 Dithervalue.JumpToLine = FALSE; SDO List.Current control OUT 1 Dithervalue.Line = 0; SDO List.Current control OUT 2 Dithervalue.Index = 16#2007; SDO List.Current control OUT 2 Dithervalue.Subindex = 16#03; SDO List.Current control OUT 2 Dithervalue.Value = 0; SDO List.Current control OUT 2 Dithervalue.Size = 16; SDO List.Current control OUT 2 Dithervalue.AbortIfError = FALSE; SDO List.Current control OUT 2 Dithervalue.JumpToLine = FALSE; SDO List.Current control OUT 2 Dithervalue.Line = 0; SDO List.Current control OUT 3 Dithervalue.Index = 16#2007; SDO List.Current control OUT 3 Dithervalue.Subindex = 16#04; SDO List.Current control OUT 3 Dithervalue.Value = 0; SDO List.Current control OUT 3 Dithervalue.Size = 16; SDO List.Current control OUT 3 Dithervalue.AbortIfError = FALSE; SDO List.Current control OUT 3 Dithervalue.JumpToLine = FALSE; SDO List.Current control OUT 3 Dithervalue.Line = 0; SDO List.Current control OUT 4 Dithervalue.Index = 16#2007; SDO List.Current control OUT 4 Dithervalue.Subindex = 16#05; SDO List.Current control OUT 4 Dithervalue.Value = 0; SDO List.Current control OUT 4 Dithervalue.Size = 16; SDO List.Current control OUT 4 Dithervalue.AbortIfError = FALSE;
                  SDO List.Current control OUT 4 Dithervalue.JumpToLine = FALSE; SDO List.Current control OUT 4 Dithervalue.Line = 0; SDO List.Current control OUT 5 Dithervalue.Index = 16#2007; SDO List.Current control OUT 5 Dithervalue.Subindex = 16#06; SDO List.Current control OUT 5 Dithervalue.Value = 0; SDO List.Current control OUT 5 Dithervalue.Size = 16; SDO List.Current control OUT 5 Dithervalue.AbortIfError = FALSE; SDO List.Current control OUT 5 Dithervalue.JumpToLine = FALSE; SDO List.Current control OUT 5 Dithervalue.Line = 0; SDO List.Current control OUT 6 Dithervalue.Index = 16#2007; SDO List.Current control OUT 6 Dithervalue.Subindex = 16#07; SDO List.Current control OUT 6 Dithervalue.Value = 0; SDO List.Current control OUT 6 Dithervalue.Size = 16; SDO List.Current control OUT 6 Dithervalue.AbortIfError = FALSE; SDO List.Current control OUT 6 Dithervalue.JumpToLine = FALSE; SDO List.Current control OUT 6 Dithervalue.Line = 0; SDO List.Current control OUT 7 Dithervalue.Index = 16#2007; SDO List.Current control OUT 7 Dithervalue.Subindex = 16#08; SDO List.Current control OUT 7 Dithervalue.Value = 0; SDO List.Current control OUT 7 Dithervalue.Size = 16; SDO List.Current control OUT 7 Dithervalue.AbortIfError = FALSE; SDO List.Current control OUT 7 Dithervalue.JumpToLine = FALSE; SDO List.Current control OUT 7 Dithervalue.Line = 0; SDO List.Period count average IN 0.Index = 16#2013; SDO List.Period count average IN 0.Subindex = 16#01; SDO List.Period count average IN 0.Value = 4; SDO List.Period count average IN 0.Size = 8; SDO List.Period count average IN 0.AbortIfError = FALSE; SDO List.Period count average IN 0.JumpToLine = FALSE; SDO List.Period count average IN 0.Line = 0; SDO List.Period count average IN 1.Index = 16#2013; SDO List.Period count average IN 1.Subindex = 16#02; SDO List.Period count average IN 1.Value = 4; SDO List.Period count average IN 1.Size = 8; SDO List.Period count average IN 1.AbortIfError = FALSE; SDO List.Period count average IN 1.JumpToLine = FALSE; SDO List.Period count average IN 1.Line = 0; SDO List.Period count average IN 4.Index = 16#2013; SDO List.Period count average IN 4.Subindex = 16#03; SDO List.Period count average IN 4.Value = 4;
                  SDO List.Period count average IN 4.Size = 8; SDO List.Period count average IN 4.AbortIfError = FALSE; SDO List.Period count average IN 4.JumpToLine = FALSE; SDO List.Period count average IN 4.Line = 0; SDO List.Period count average IN 5.Index = 16#2013; SDO List.Period count average IN 5.Subindex = 16#04; SDO List.Period count average IN 5.Value = 4; SDO List.Period count average IN 5.Size = 8; SDO List.Period count average IN 5.AbortIfError = FALSE; SDO List.Period count average IN 5.JumpToLine = FALSE; SDO List.Period count average IN 5.Line = 0; SDO List.Frequency timebase IN 0.Index = 16#2016; SDO List.Frequency timebase IN 0.Subindex = 16#01; SDO List.Frequency timebase IN 0.Value = 50; SDO List.Frequency timebase IN 0.Size = 16; SDO List.Frequency timebase IN 0.AbortIfError = FALSE; SDO List.Frequency timebase IN 0.JumpToLine = FALSE; SDO List.Frequency timebase IN 0.Line = 0; SDO List.Frequency timebase IN 1.Index = 16#2016; SDO List.Frequency timebase IN 1.Subindex = 16#02; SDO List.Frequency timebase IN 1.Value = 50; SDO List.Frequency timebase IN 1.Size = 16; SDO List.Frequency timebase IN 1.AbortIfError = FALSE; SDO List.Frequency timebase IN 1.JumpToLine = FALSE; SDO List.Frequency timebase IN 1.Line = 0; SDO List.Frequency timebase IN 4.Index = 16#2016; SDO List.Frequency timebase IN 4.Subindex = 16#03; SDO List.Frequency timebase IN 4.Value = 50; SDO List.Frequency timebase IN 4.Size = 16; SDO List.Frequency timebase IN 4.AbortIfError = FALSE; SDO List.Frequency timebase IN 4.JumpToLine = FALSE; SDO List.Frequency timebase IN 4.Line = 0; SDO List.Frequency timebase IN 5.Index = 16#2016; SDO List.Frequency timebase IN 5.Subindex = 16#04; SDO List.Frequency timebase IN 5.Value = 50; SDO List.Frequency timebase IN 5.Size = 16; SDO List.Frequency timebase IN 5.AbortIfError = FALSE; SDO List.Frequency timebase IN 5.JumpToLine = FALSE; SDO List.Frequency timebase IN 5.Line = 0; SDO List.Node id switch a.Index = 16#20F0;
                  SDO List.Node id switch a.Subindex = 16#00; SDO List.Node id switch a.Value = 20; SDO List.Node id switch a.Size = 8; SDO List.Node id switch a.AbortIfError = FALSE; SDO List.Node id switch a.JumpToLine = FALSE; SDO List.Node id switch a.Line = 0; SDO List.Node id switch b.Index = 16#20F1; SDO List.Node id switch b.Subindex = 16#00; SDO List.Node id switch b.Value = 20; SDO List.Node id switch b.Size = 8; SDO List.Node id switch b.AbortIfError = FALSE; SDO List.Node id switch b.JumpToLine = FALSE; SDO List.Node id switch b.Line = 0; SDO List.Bit rate switch a.Index = 16#20F2; SDO List.Bit rate switch a.Subindex = 16#00; SDO List.Bit rate switch a.Value = 3; SDO List.Bit rate switch a.Size = 8; SDO List.Bit rate switch a.AbortIfError = FALSE; SDO List.Bit rate switch a.JumpToLine = FALSE; SDO List.Bit rate switch a.Line = 0; SDO List.Bit rate switch b.Index = 16#20F3; SDO List.Bit rate switch b.Subindex = 16#00; SDO List.Bit rate switch b.Value = 3; SDO List.Bit rate switch b.Size = 8; SDO List.Bit rate switch b.AbortIfError = FALSE; SDO List.Bit rate switch b.JumpToLine = FALSE; SDO List.Bit rate switch b.Line = 0; SDO List.Autostart.Index = 16#20F4; SDO List.Autostart.Subindex = 16#00; SDO List.Autostart.Value = 0; SDO List.Autostart.Size = 16; SDO List.Autostart.AbortIfError = FALSE; SDO List.Autostart.JumpToLine = FALSE; SDO List.Autostart.Line = 0; SDO List.Lock edit parameters.Index = 16#20F5; SDO List.Lock edit parameters.Subindex = 16#00; SDO List.Lock edit parameters.Value = 0; SDO List.Lock edit parameters.Size = 8; SDO List.Lock edit parameters.AbortIfError = FALSE; SDO List.Lock edit parameters.JumpToLine = FALSE;
                  SDO List.Lock edit parameters.Line = 0; SDO List.CANopen interface a.Index = 16#20F6; SDO List.CANopen interface a.Subindex = 16#00; SDO List.CANopen interface a.Value = 1; SDO List.CANopen interface a.Size = 8; SDO List.CANopen interface a.AbortIfError = FALSE; SDO List.CANopen interface a.JumpToLine = FALSE; SDO List.CANopen interface a.Line = 0; SDO List.CANopen interface b.Index = 16#20F7; SDO List.CANopen interface b.Subindex = 16#00; SDO List.CANopen interface b.Value = 1; SDO List.CANopen interface b.Size = 8; SDO List.CANopen interface b.AbortIfError = FALSE; SDO List.CANopen interface b.JumpToLine = FALSE; SDO List.CANopen interface b.Line = 0; SDO List.Binary Outputs OUT 0 - OUT 7.Index = 16#6200; SDO List.Binary Outputs OUT 0 - OUT 7.Subindex = 16#01; SDO List.Binary Outputs OUT 0 - OUT 7.Value = 0; SDO List.Binary Outputs OUT 0 - OUT 7.Size = 8; SDO List.Binary Outputs OUT 0 - OUT 7.AbortIfError = FALSE; SDO List.Binary Outputs OUT 0 - OUT 7.JumpToLine = FALSE; SDO List.Binary Outputs OUT 0 - OUT 7.Line = 0; SDO List.Analog Output OUT 0.Index = 16#6414; SDO List.Analog Output OUT 0.Subindex = 16#01; SDO List.Analog Output OUT 0.Value = 1; SDO List.Analog Output OUT 0.Size = 16; SDO List.Analog Output OUT 0.AbortIfError = FALSE; SDO List.Analog Output OUT 0.JumpToLine = FALSE; SDO List.Analog Output OUT 0.Line = 0; SDO List.Analog Output OUT 1.Index = 16#6414; SDO List.Analog Output OUT 1.Subindex = 16#02; SDO List.Analog Output OUT 1.Value = 0; SDO List.Analog Output OUT 1.Size = 16; SDO List.Analog Output OUT 1.AbortIfError = FALSE; SDO List.Analog Output OUT 1.JumpToLine = FALSE; SDO List.Analog Output OUT 1.Line = 0; SDO List.Analog Output OUT 2.Index = 16#6414; SDO List.Analog Output OUT 2.Subindex = 16#03; SDO List.Analog Output OUT 2.Value = 0; SDO List.Analog Output OUT 2.Size = 16;
                  SDO List.Analog Output OUT 2.AbortIfError = FALSE; SDO List.Analog Output OUT 2.JumpToLine = FALSE; SDO List.Analog Output OUT 2.Line = 0; SDO List.Analog Output OUT 3.Index = 16#6414; SDO List.Analog Output OUT 3.Subindex = 16#04; SDO List.Analog Output OUT 3.Value = 0; SDO List.Analog Output OUT 3.Size = 16; SDO List.Analog Output OUT 3.AbortIfError = FALSE; SDO List.Analog Output OUT 3.JumpToLine = FALSE; SDO List.Analog Output OUT 3.Line = 0; SDO List.Analog Output OUT 4.Index = 16#6414; SDO List.Analog Output OUT 4.Subindex = 16#05; SDO List.Analog Output OUT 4.Value = 0; SDO List.Analog Output OUT 4.Size = 16; SDO List.Analog Output OUT 4.AbortIfError = FALSE; SDO List.Analog Output OUT 4.JumpToLine = FALSE; SDO List.Analog Output OUT 4.Line = 0; SDO List.Analog Output OUT 5.Index = 16#6414; SDO List.Analog Output OUT 5.Subindex = 16#06; SDO List.Analog Output OUT 5.Value = 0; SDO List.Analog Output OUT 5.Size = 16; SDO List.Analog Output OUT 5.AbortIfError = FALSE; SDO List.Analog Output OUT 5.JumpToLine = FALSE; SDO List.Analog Output OUT 5.Line = 0; SDO List.Analog Output OUT 6.Index = 16#6414; SDO List.Analog Output OUT 6.Subindex = 16#07; SDO List.Analog Output OUT 6.Value = 0; SDO List.Analog Output OUT 6.Size = 16; SDO List.Analog Output OUT 6.AbortIfError = FALSE; SDO List.Analog Output OUT 6.JumpToLine = FALSE; SDO List.Analog Output OUT 6.Line = 0; SDO List.Analog Output OUT 7.Index = 16#6414; SDO List.Analog Output OUT 7.Subindex = 16#08; SDO List.Analog Output OUT 7.Value = 0; SDO List.Analog Output OUT 7.Size = 16; SDO List.Analog Output OUT 7.AbortIfError = FALSE; SDO List.Analog Output OUT 7.JumpToLine = FALSE; SDO List.Analog Output OUT 7.Line = 0; SDO List.Communication cycle period.Index = 16#1006; SDO List.Communication cycle period.Subindex = 16#00;
                  SDO List.Communication cycle period.Value = 150000; SDO List.Communication cycle period.Size = 32; SDO List.Communication cycle period.AbortIfError = FALSE; SDO List.Communication cycle period.JumpToLine = FALSE; SDO List.Communication cycle period.Line = 0; ConfigVersion = 50659584
                output Application.GVL_STRUCT.gstCR2052n20o.xCabAlarm : BOOL  // Binary Outputs OUT 0 - OUT 7.Bit3
                input  Application.GVL_STRUCT.gstCR2052n20i.xGpsAutoMode : BOOL  // Binary Inputs IN 0 - IN 7.Bit1
                input  Application.GVL_STRUCT.gstCR2052n20i.xArmrestDown : BOOL  // Binary Inputs IN 0 - IN 7.Bit2
                input  Application.GVL_STRUCT.gstCR2052n20i.xLoadSense : BOOL  // Binary Inputs IN 0 - IN 7.Bit4
                input  Application.GVL_STRUCT.gstCR2052n20i.xReverse : BOOL  // Binary Inputs IN 0 - IN 7.Bit6
                input  Application.GVL_STRUCT.gstHarvCR711SiDiag.xGPSHeightShort : BOOL  // BrakeShort Inputs IN 0 - IN 7.Bit0
                input  Application.GVL_STRUCT.gstHarvCR711SiDiag.xGPSTiltShort : BOOL  // BrakeShort Inputs IN 0 - IN 7.Bit1
                input  Application.GVL_STRUCT.gstHarvCR711SiDiag.xArmrestDownShort : BOOL  // BrakeShort Inputs IN 0 - IN 7.Bit2
                input  Application.GVL_STRUCT.gstHarvCR711SiDiag.xLoadSenseShort : BOOL  // BrakeShort Inputs IN 0 - IN 7.Bit3
                input  Application.GVL_STRUCT.gstHarvCR711SiDiag.xReverseShort : BOOL  // BrakeShort Inputs IN 0 - IN 7.Bit5
                input  Application.GVL_STRUCT.gstHarvCR711SiDiag.xGpsAutoModeShort : BOOL  // BrakeShort Inputs IN 0 - IN 7.Bit6
                input  Application.GVL_STRUCT.gstHarvCR711SiDiag.xGpsHeightLoss : BOOL  // BrakeLoss Inputs IN 0 - IN 7.Bit0
                input  Application.GVL_STRUCT.gstHarvCR711SiDiag.xGPSTiltLoss : BOOL  // BrakeLoss Inputs IN 0 - IN 7.Bit1
                input  Application.GVL_STRUCT.gstHarvCR711SiDiag.xArmrestDownLoss : BOOL  // BrakeLoss Inputs IN 0 - IN 7.Bit2
                input  Application.GVL_STRUCT.gstHarvCR711SiDiag.xLoadSenseLoss : BOOL  // BrakeLoss Inputs IN 0 - IN 7.Bit3
                input  Application.GVL_STRUCT.gstHarvCR711SiDiag.xReverseLoss : BOOL  // BrakeLoss Inputs IN 0 - IN 7.Bit5
                input  Application.GVL_STRUCT.gstHarvCR711SiDiag.xGpsAutoModeLoss : BOOL  // BrakeLoss Inputs IN 0 - IN 7.Bit6
                input  Application.GVL_STRUCT.gstHarvCR711SoDiag.xCabAlarmShort : BOOL  // BrakeShort Outputs OUT 0 - OUT 7.Bit3
                input  Application.GVL_STRUCT.gstHarvCR711SoDiag.xCabAlarmLoss : BOOL  // BrakeLoss Outputs OUT 0 - OUT 7.Bit3
                input  Application.GVL_STRUCT.gstCR2052n20i.uiGpsRaiseLower : UINT  // Analog Input IN 0
                input  Application.GVL_STRUCT.gstCR2052n20i.uiGpsTiltLeftRight : UINT  // Analog Input IN 1
                input  Application.GVL.uiNode20VBBSTx : UINT  // VBBS System voltage
                input  Application.GVL.uiNode20VBB2Tx : UINT  // VBB2 Supply voltage
                input  Application.GVL.iNode20TempTx : INT  // Temperature
                unmapped channels: Binary Outputs OUT 0 - OUT 7, Analog Output OUT 0, Analog Output OUT 1, Analog Output OUT 2, Analog Output OUT 3, Analog Output OUT 4, Analog Output OUT 5, Analog Output OUT 6, Analog Output OUT 7, Binary Inputs IN 0 - IN 7, BrakeShort Inputs IN 0 - IN 7, BrakeLoss Inputs IN 0 - IN 7, OverCurrent Inputs IN 0/IN 1/IN 4/IN 5, BrakeShort Outputs OUT 0 - OUT 7, BrakeLoss Outputs OUT 0 - OUT 7, Overload Outputs OUT 0 - OUT 7, Analog Input IN 4, Analog Input IN 5, Resistance Input IN 2, Resistance Input IN 3, Resistance Input IN 6, Resistance Input IN 7, Period Inputs IN 0, Period Inputs IN 1, Period Inputs IN 4, Period Inputs IN 5, Ratio IN 0, Ratio IN 1, Ratio IN 4, Ratio IN 5, Frequency IN 0, Frequency IN 1, Frequency IN 4, Frequency IN 5, Current value OUT 0, Current value OUT 1, Current value OUT 2, Current value OUT 3, Current value OUT 4, Current value OUT 5,
                  Current value OUT 6, Current value OUT 7
      Ethernet : Ethernet, ifm electronic, version 3.2.0.0
    HMI : HMI, ifm electronic, version 3.2.0.0
      User_LEDs : User_LEDs, ifm electronic, version 3.2.0.0
          input  UserLED0_I : LED_IEC_B_INPUT_MAPPING_TYPE  // UserLED0_I
          input  UserLED1_I : LED_IEC_B_INPUT_MAPPING_TYPE  // UserLED1_I
          input  UserLED2_I : LED_IEC_B_INPUT_MAPPING_TYPE  // UserLED2_I
          input  UserLED3_I : LED_IEC_B_INPUT_MAPPING_TYPE  // UserLED3_I
          output UserLED0_Q : LED_IEC_B_OUTPUT_MAPPING_TYPE  // User LED 0
          output UserLED1_Q : LED_IEC_B_OUTPUT_MAPPING_TYPE  // User LED 1
          output UserLED2_Q : LED_IEC_B_OUTPUT_MAPPING_TYPE  // User LED 2
          output UserLED3_Q : LED_IEC_B_OUTPUT_MAPPING_TYPE  // User LED 3
    Local_IO : Local_IO, ifm electronic, version 3.2.0.0
      Inputs : Inputs, ifm electronic, version 3.2.0.0
          input  IN0100_I : IN_MULTIFUNCTION_A_INPUT_MAPPING_TYPE  // IN0100_I
          input  IN0101_I : IN_MULTIFUNCTION_A_INPUT_MAPPING_TYPE  // IN0101_I
          input  IN0102_I : IN_MULTIFUNCTION_A_INPUT_MAPPING_TYPE  // IN0102_I
          input  IN0103_I : IN_MULTIFUNCTION_A_INPUT_MAPPING_TYPE  // IN0103_I
          input  IN0200_I : IN_MULTIFUNCTION_A_INPUT_MAPPING_TYPE  // IN0200_I
          input  IN0201_I : IN_MULTIFUNCTION_A_INPUT_MAPPING_TYPE  // IN0201_I
          input  IN0202_I : IN_MULTIFUNCTION_A_INPUT_MAPPING_TYPE  // IN0202_I
          input  IN0203_I : IN_MULTIFUNCTION_A_INPUT_MAPPING_TYPE  // IN0203_I
          input  IN0600_I : IN_MULTIFUNCTION_A_INPUT_MAPPING_TYPE  // IN0600_I
          input  IN0601_I : IN_MULTIFUNCTION_A_INPUT_MAPPING_TYPE  // IN0601_I
          input  IN0602_I : IN_MULTIFUNCTION_A_INPUT_MAPPING_TYPE  // IN0602_I
          input  IN0603_I : IN_MULTIFUNCTION_A_INPUT_MAPPING_TYPE  // IN0603_I
          input  IN0700_I : IN_MULTIFUNCTION_A_INPUT_MAPPING_TYPE  // IN0700_I
          input  IN0701_I : IN_MULTIFUNCTION_A_INPUT_MAPPING_TYPE  // IN0701_I
          input  IN0702_I : IN_MULTIFUNCTION_A_INPUT_MAPPING_TYPE  // IN0702_I
          input  IN0703_I : IN_MULTIFUNCTION_A_INPUT_MAPPING_TYPE  // IN0703_I
          input  IN0400_I : IN_RESISTOR_A_INPUT_MAPPING_TYPE  // IN0400_I
          input  IN0401_I : IN_RESISTOR_A_INPUT_MAPPING_TYPE  // IN0401_I
          input  IN0900_I : IN_RESISTOR_A_INPUT_MAPPING_TYPE  // IN0900_I
          input  IN0901_I : IN_RESISTOR_A_INPUT_MAPPING_TYPE  // IN0901_I
          input  IN0300_I : IN_DIGITAL_B_INPUT_MAPPING_TYPE  // IN0300_I
          input  IN0301_I : IN_DIGITAL_B_INPUT_MAPPING_TYPE  // IN0301_I
          input  IN0800_I : IN_DIGITAL_B_INPUT_MAPPING_TYPE  // IN0800_I
          input  IN0801_I : IN_DIGITAL_B_INPUT_MAPPING_TYPE  // IN0801_I
          input  COM_RESET_I : IN_COMMUNICATION_RESET_INPUT_MAPPING_TYPE  // COM_RESET_I
          input  IN0000_I : IN_FREQUENCY_B_CHANNEL_A_INPUT_MAPPING_TYPE  // IN0000_I
          input  IN0002_I : IN_FREQUENCY_B_CHANNEL_A_INPUT_MAPPING_TYPE  // IN0002_I
          input  IN0500_I : IN_FREQUENCY_B_CHANNEL_A_INPUT_MAPPING_TYPE  // IN0500_I
          input  IN0502_I : IN_FREQUENCY_B_CHANNEL_A_INPUT_MAPPING_TYPE  // IN0502_I
          input  IN0001_I : IN_FREQUENCY_B_CHANNEL_B_INPUT_MAPPING_TYPE  // IN0001_I
          input  IN0003_I : IN_FREQUENCY_B_CHANNEL_B_INPUT_MAPPING_TYPE  // IN0003_I
          input  IN0501_I : IN_FREQUENCY_B_CHANNEL_B_INPUT_MAPPING_TYPE  // IN0501_I
          input  IN0503_I : IN_FREQUENCY_B_CHANNEL_B_INPUT_MAPPING_TYPE  // IN0503_I
      Outputs : Outputs, ifm electronic, version 3.2.0.0
          input  OUT0006_I : OUT_PWM_40_BRIDGE_A_INPUT_MAPPING_TYPE  // OUT0006_I
          input  OUT0106_I : OUT_PWM_40_BRIDGE_A_INPUT_MAPPING_TYPE  // OUT0106_I
          input  OUT0206_I : OUT_PWM_40_BRIDGE_A_INPUT_MAPPING_TYPE  // OUT0206_I
          input  OUT0008_I : OUT_PWM_40_A_INPUT_MAPPING_TYPE  // OUT0008_I
          input  OUT0108_I : OUT_PWM_40_A_INPUT_MAPPING_TYPE  // OUT0108_I
          input  OUT0208_I : OUT_PWM_40_A_INPUT_MAPPING_TYPE  // OUT0208_I
          input  OUT0000_I : OUT_PWM_25_A_INPUT_MAPPING_TYPE  // OUT0000_I
          input  OUT0002_I : OUT_PWM_25_A_INPUT_MAPPING_TYPE  // OUT0002_I
          input  OUT0004_I : OUT_PWM_25_A_INPUT_MAPPING_TYPE  // OUT0004_I
          input  OUT0100_I : OUT_PWM_25_A_INPUT_MAPPING_TYPE  // OUT0100_I
          input  OUT0102_I : OUT_PWM_25_A_INPUT_MAPPING_TYPE  // OUT0102_I
          input  OUT0104_I : OUT_PWM_25_A_INPUT_MAPPING_TYPE  // OUT0104_I
          input  OUT0200_I : OUT_PWM_25_A_INPUT_MAPPING_TYPE  // OUT0200_I
          input  OUT0202_I : OUT_PWM_25_A_INPUT_MAPPING_TYPE  // OUT0202_I
          input  OUT0204_I : OUT_PWM_25_A_INPUT_MAPPING_TYPE  // OUT0204_I
          input  OUT3001_I : OUT_VOLTAGE_A_INPUT_MAPPING_TYPE  // OUT3001_I
          input  OUT3000_I : OUT_SUPPLY_A_INPUT_MAPPING_TYPE  // OUT3000_I
          input  OUT0001_I : OUT_PWM_25_B_INPUT_MAPPING_TYPE  // OUT0001_I
          input  OUT0003_I : OUT_PWM_25_B_INPUT_MAPPING_TYPE  // OUT0003_I
          input  OUT0005_I : OUT_PWM_25_B_INPUT_MAPPING_TYPE  // OUT0005_I
          input  OUT0101_I : OUT_PWM_25_B_INPUT_MAPPING_TYPE  // OUT0101_I
          input  OUT0103_I : OUT_PWM_25_B_INPUT_MAPPING_TYPE  // OUT0103_I
          input  OUT0105_I : OUT_PWM_25_B_INPUT_MAPPING_TYPE  // OUT0105_I
          input  OUT0201_I : OUT_PWM_25_B_INPUT_MAPPING_TYPE  // OUT0201_I
          input  OUT0203_I : OUT_PWM_25_B_INPUT_MAPPING_TYPE  // OUT0203_I
          input  OUT0205_I : OUT_PWM_25_B_INPUT_MAPPING_TYPE  // OUT0205_I
          input  OUT0007_I : OUT_PWM_40_BRIDGE_A_INPUT_MAPPING_TYPE  // OUT0007_I
          input  OUT0107_I : OUT_PWM_40_BRIDGE_A_INPUT_MAPPING_TYPE  // OUT0107_I
          input  OUT0207_I : OUT_PWM_40_BRIDGE_A_INPUT_MAPPING_TYPE  // OUT0207_I
          output OUT0006_Q : OUT_PWM_40_BRIDGE_A_OUTPUT_MAPPING_TYPE  // OUT0006_Q
          output OUT0106_Q : OUT_PWM_40_BRIDGE_A_OUTPUT_MAPPING_TYPE  // OUT0106_Q
          output OUT0206_Q : OUT_PWM_40_BRIDGE_A_OUTPUT_MAPPING_TYPE  // OUT0206_Q
          output OUT0008_Q : OUT_PWM_40_A_OUTPUT_MAPPING_TYPE  // OUT0008_Q
          output OUT0108_Q : OUT_PWM_40_A_OUTPUT_MAPPING_TYPE  // OUT0108_Q
          output OUT0208_Q : OUT_PWM_40_A_OUTPUT_MAPPING_TYPE  // OUT0208_Q
          output OUT0000_Q : OUT_PWM_25_A_OUTPUT_MAPPING_TYPE  // OUT0000_Q
          output OUT0002_Q : OUT_PWM_25_A_OUTPUT_MAPPING_TYPE  // OUT0002_Q
          output OUT0004_Q : OUT_PWM_25_A_OUTPUT_MAPPING_TYPE  // OUT0004_Q
          output OUT0100_Q : OUT_PWM_25_A_OUTPUT_MAPPING_TYPE  // OUT0100_Q
          output OUT0102_Q : OUT_PWM_25_A_OUTPUT_MAPPING_TYPE  // OUT0102_Q
          output OUT0104_Q : OUT_PWM_25_A_OUTPUT_MAPPING_TYPE  // OUT0104_Q
          output OUT0200_Q : OUT_PWM_25_A_OUTPUT_MAPPING_TYPE  // OUT0200_Q
          output OUT0202_Q : OUT_PWM_25_A_OUTPUT_MAPPING_TYPE  // OUT0202_Q
          output OUT0204_Q : OUT_PWM_25_A_OUTPUT_MAPPING_TYPE  // OUT0204_Q
          output OUT3001_Q : OUT_VOLTAGE_A_OUTPUT_MAPPING_TYPE  // OUT3001_Q
          output OUT3000_Q : OUT_SUPPLY_A_OUTPUT_MAPPING_TYPE  // OUT3000_Q
          output OUT0001_Q : OUT_PWM_25_B_OUTPUT_MAPPING_TYPE  // OUT0001_Q
          output OUT0003_Q : OUT_PWM_25_B_OUTPUT_MAPPING_TYPE  // OUT0003_Q
          output OUT0005_Q : OUT_PWM_25_B_OUTPUT_MAPPING_TYPE  // OUT0005_Q
          output OUT0101_Q : OUT_PWM_25_B_OUTPUT_MAPPING_TYPE  // OUT0101_Q
          output OUT0103_Q : OUT_PWM_25_B_OUTPUT_MAPPING_TYPE  // OUT0103_Q
          output OUT0105_Q : OUT_PWM_25_B_OUTPUT_MAPPING_TYPE  // OUT0105_Q
          output OUT0201_Q : OUT_PWM_25_B_OUTPUT_MAPPING_TYPE  // OUT0201_Q
          output OUT0203_Q : OUT_PWM_25_B_OUTPUT_MAPPING_TYPE  // OUT0203_Q
          output OUT0205_Q : OUT_PWM_25_B_OUTPUT_MAPPING_TYPE  // OUT0205_Q
          output OUT0007_Q : OUT_PWM_40_BRIDGE_A_OUTPUT_MAPPING_TYPE  // OUT0007_Q
          output OUT0107_Q : OUT_PWM_40_BRIDGE_A_OUTPUT_MAPPING_TYPE  // OUT0107_Q
          output OUT0207_Q : OUT_PWM_40_BRIDGE_A_OUTPUT_MAPPING_TYPE  // OUT0207_Q
      System_Inputs : System_Inputs, ifm electronic, version 3.2.0.0
          input  VBB30 : IN_SYSTEM_VOLTAGE_INPUT_MAPPING_TYPE  // VBB30
          input  Application.GVL.uiPlcVBB30Tx : UINT  // VBB30.VBBx
          input  VBB15 : IN_SYSTEM_VOLTAGE_INPUT_MAPPING_TYPE  // VBB15
          input  Application.GVL.uiPlcVBB15Tx : UINT  // VBB15.VBBx
          input  TemperatureBoard0 : IN_TEMPERATURE_INPUT_MAPPING_TYPE  // TemperatureBoard0
          input  Application.GVL.iPlcTempBTx : INT  // TemperatureBoard0.Temperature
          input  TemperatureChip0 : IN_TEMPERATURE_INPUT_MAPPING_TYPE  // TemperatureChip0
          input  Application.GVL.iPlcTempCTx : INT  // TemperatureChip0.Temperature
      System_Outputs : System_Outputs, ifm electronic, version 3.2.0.0
          input  VBB0_SW_I : OUT_GROUP_SWITCH_INPUT_MAPPING_TYPE  // VBB0_SW_I
          input  VBB1_SW_I : OUT_GROUP_SWITCH_INPUT_MAPPING_TYPE  // VBB1_SW_I
          input  VBB2_SW_I : OUT_GROUP_SWITCH_INPUT_MAPPING_TYPE  // VBB2_SW_I
          output VBB0_SW_Q : OUT_GROUP_SWITCH_OUTPUT_MAPPING_TYPE  // VBB0_SW_Q
          output VBB1_SW_Q : OUT_GROUP_SWITCH_OUTPUT_MAPPING_TYPE  // VBB1_SW_Q
          output VBB2_SW_Q : OUT_GROUP_SWITCH_OUTPUT_MAPPING_TYPE  // VBB2_SW_Q
          output SUPPLY_SWITCH_Q : OUT_SYS_SWITCH_OUTPUT_MAPPING_TYPE  // SUPPLY_SWITCH_Q
  CR711S : CR711S, ifm electronic, order no. CR711S, version 3.2.0.0
  text list GlobalTextList
*)

// StandardPLC/Application/PersistentVars
{attribute 'qualified_only'}
VAR_GLOBAL PERSISTENT RETAIN

wEngineOnCount		:WORD;	//Count OF times Engine is turned ON
wGpsOnCount			:WORD;	//Count OF times GPS Activated
wAutoOnCount		:WORD;	//Count OF times Auto Harvest Activated
wFlightOnCount		:WORD;	//Count OF times Flight Converyor is turned ON
wTotalMaintCount	:WORD;	//Count of times Maintenance Mode Activated
wTotalFilterCount	:WORD;	//Count of Filter Bypass Alarms
wTotalPressCount	:WORD;	//Count of Pressure Alarms
wTotalTempCount		:WORD;	//Count OF Temperature Alarms
wTotalEstopCount	:WORD;	//Count of times E-Stop is Activated
wTotalStallCount	:WORD;	//Count of Machine Stalls
wTotalDerateCount	:WORD;	//Count of De-rate Events
wTotalVoltageCount	:WORD;	//Count of Voltage Alarms

wHarvPlcVoltCount  : WORD;    // Total count of Trailer PLC Voltage Alarms
wHarvDispVoltCount : WORD;    // Total count of Trailer Display Voltage Alarms
wTracDispVoltCount : WORD;    // Total count of Prime Mover Display Voltage Alarms

wNode20VoltCount   : WORD;    // Total count of IO module Node 20 Module Voltage Alarm
wNode0VoltCount   : WORD;    // Total count of Engine Node 50 Voltage Alarm

	
END_VAR

// SafetyPLC/Application/EVL
(* THIS EVL IS AUTOGENERATED. DO NOT MODIFY THESE ATTRIBUTES. *)
{attribute 'location' := '16#800' }
{attribute 'linkalways'}
{attribute 'qualified_only'}
VAR_GLOBAL

END_VAR

// SafetyPLC/Application/PLC_PRG
PROGRAM PLC_PRG
VAR

END_VAR

END_PROGRAM

// StandardPLC/Application/SFC_TEST
PROGRAM SFC_TEST
VAR
	SensorA: BOOL;
	SensorB: BOOL;
END_VAR

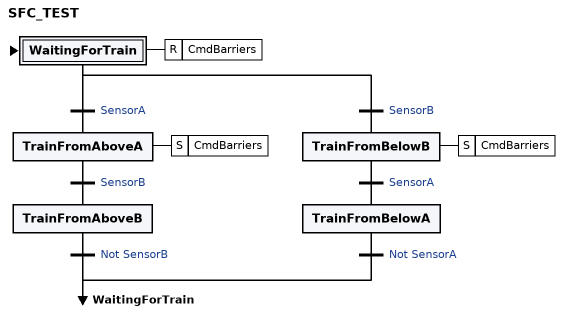
INITIAL_STEP WaitingForTrain:
    CmdBarriers(R);
END_STEP
TRANSITION FROM WaitingForTrain TO TrainFromAboveA
    := SensorA;
END_TRANSITION
STEP TrainFromAboveA:
    CmdBarriers(S);
END_STEP
TRANSITION FROM TrainFromAboveA TO TrainFromAboveB
    := SensorB;
END_TRANSITION
STEP TrainFromAboveB:
END_STEP
TRANSITION FROM TrainFromAboveB TO WaitingForTrain
    := Not SensorB;
END_TRANSITION
TRANSITION FROM WaitingForTrain TO TrainFromBelowB
    := SensorB;
END_TRANSITION
STEP TrainFromBelowB:
    CmdBarriers(S);
END_STEP
TRANSITION FROM TrainFromBelowB TO TrainFromBelowA
    := SensorA;
END_TRANSITION
STEP TrainFromBelowA:
END_STEP
TRANSITION FROM TrainFromBelowA TO WaitingForTrain
    := Not SensorA;
END_TRANSITION

END_PROGRAM

// StandardPLC/Application/FB_TESTING
PROGRAM FB_TESTING
(***********************************************************************************************
Object Name	: PLC_SUPPLY
Descrition	: Program to control the System Supply Switch to ensure the PLC turns OFF when the ignition turns OFF.
Author		: KP
Date		: 17/06/25
Rev			: P1
***********************************************************************************************)
VAR CONSTANT
	uiMinVoltage 		: UINT := 5000;    // Minimum Voltage in mV
END_VAR
VAR
	fbSystemSupply 	: ifmIOcommon.SystemSupply; // Function Block to monitor supply voltage on VBB15 (from ignition)
	fbSupplySwitch 	: ifmIOcommon.SupplySwitch; // Function Block to turn ON/OFF latching switch on VBB15 supply (from ignition)
	uiCurrSupplyVolt	: UINT ;    // Operating Voltage in mV
	TOF_0: TOF;
	Test: BOOL;
	dude: BOOL;
END_VAR

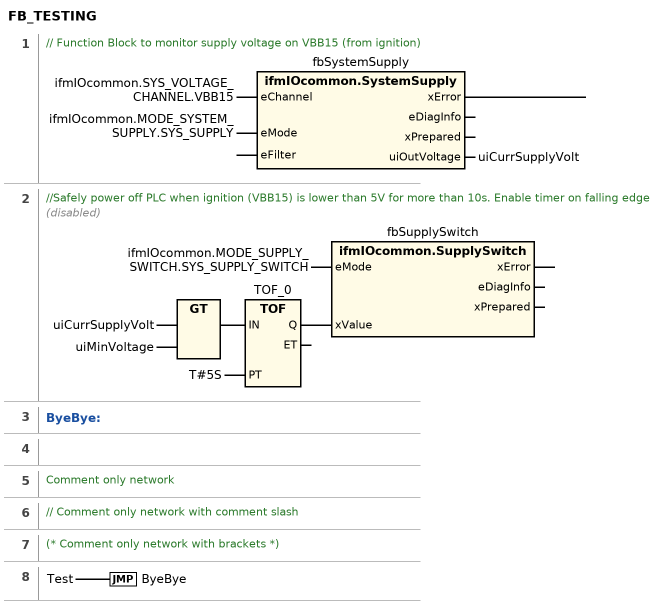
// NETWORK 1
// // Function Block to monitor supply voltage on VBB15 (from ignition)
fbSystemSupply(
    eChannel := ifmIOcommon.SYS_VOLTAGE_CHANNEL.VBB15,
    eMode := ifmIOcommon.MODE_SYSTEM_SUPPLY.SYS_SUPPLY,
    uiOutVoltage => uiCurrSupplyVolt); // ifmIOcommon.SystemSupply

// NETWORK 2 (disabled)
// //Safely power off PLC when ignition (VBB15) is lower than 5V for more than 10s. Enable timer on falling edge
// TOF_0(IN := uiCurrSupplyVolt > uiMinVoltage, PT := T#5S); // TOF
// fbSupplySwitch(eMode := ifmIOcommon.MODE_SUPPLY_SWITCH.SYS_SUPPLY_SWITCH, xValue := TOF_0.Q); // ifmIOcommon.SupplySwitch

// NETWORK 3
ByeBye: ;

// NETWORK 4

// NETWORK 5
// Comment only network

// NETWORK 6
// // Comment only network with comment slash

// NETWORK 7
// (* Comment only network with brackets *)

// NETWORK 8
IF Test THEN JMP ByeBye; END_IF

ACTION PleaseIhaveKids:
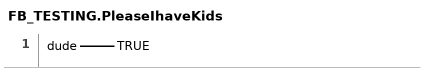
// NETWORK 1
TRUE := dude;
END_ACTION

END_PROGRAM

// StandardPLC/Application/LD_TEST
PROGRAM LD_TEST
VAR
	Sensor1: BOOL;
	Sensor2: BOOL;
	sensor3: BOOL;
	PowerOn: BOOL;
	TON_0: TON;
	CTU_0: CTU;
	PowerOff: BOOL;
END_VAR

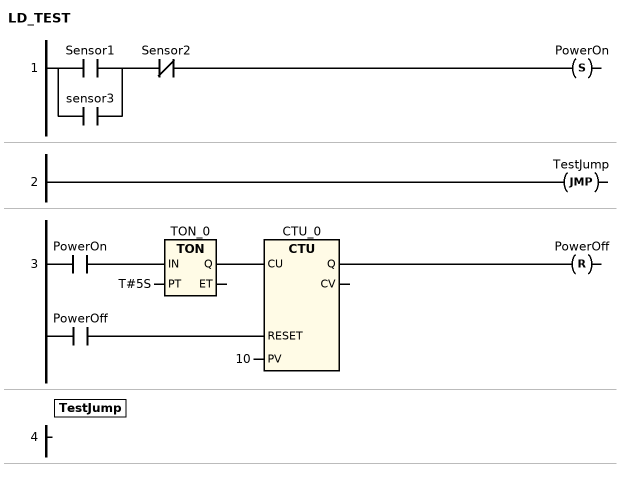
// NETWORK 1
PowerOn S= (Sensor1 OR sensor3) AND NOT Sensor2;

// NETWORK 2
JMP TestJump;

// NETWORK 3
TON_0(IN := PowerOn, PT := T#5S); // TON
CTU_0(CU := TON_0.Q, RESET := PowerOff, PV := 10); // CTU
PowerOff R= CTU_0.Q;

// NETWORK 4
TestJump: ;

END_PROGRAM

// StandardPLC/Application/Visualization
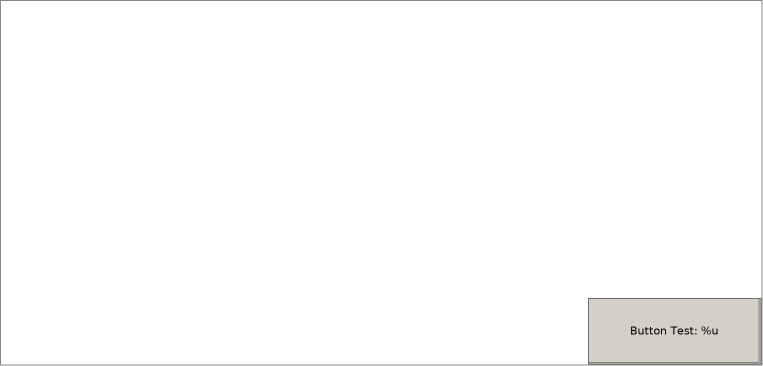
VISUALIZATION Visualization  // 763x366
    Button (588,298 173x66), "Button Test: %u", text variable: FB_TESTING.uiCurrSupplyVolt
END_VISUALIZATION
